// TIA Portal V20 export
// export: Created 2025-12-01T14:57:30.8490755Z, ExportSetting None, DisplayName Totally Integrated Automation Portal, DisplayVersion V20 Update 3, DisplayName TIA Portal Openness, DisplayVersion V20 Update 3, DisplayName TIA Portal Version Control Interface, DisplayVersion V20 Update 3, DisplayName STEP 7 Professional, DisplayVersion V20 Update 3, DisplayName STEP 7 Safety, DisplayVersion V20 Update 2, DisplayName WinCC Basic/Comfort/Advanced, DisplayVersion V20 Update 3, DisplayName WinCC Professional, DisplayVersion V20 Update 3, DisplayName WinCC Unified, DisplayVersion V20 Update 3
FUNCTION_BLOCK "FB271_FSS_Carga_Congelado"   // FB271, LAD
{ S7_Optimized_Access := 'FALSE' }
// NO sube los topes hasta
// stored: AutoNumber false, SetENOAutomatically false
   VAR_INPUT
      Mesa : UInt;   // Mesa de la FB
      Error_Tx : Bool;
      EnTension : Bool;   // Existe Tension en la Mesa
      Termico_Tx : Bool;
      pHsMx_1 : Bool;
      pHsMx_2 : Bool;
      EnMovimiento_Tx : Bool;
      Termico_TRx : Bool;
      Termico_TRxE : Bool;
      TRx_Arriba : Bool;
      TRx_Abajo { ExternalAccessible := 'False'; ExternalVisible := 'False'; ExternalWritable := 'False'} : Bool;
      EnMovimiento_TRx : Bool;
      EnMovimiento_TRxE : Bool;
      TP1_Arriba : Bool;
      TP1_Abajo { ExternalAccessible := 'False'; ExternalVisible := 'False'; ExternalWritable := 'False'} : Bool;
      TP2_Arriba : Bool;
      TP2_Abajo { ExternalAccessible := 'False'; ExternalVisible := 'False'; ExternalWritable := 'False'} : Bool;
      EnMovimiento_TP1 : Bool;
      EnMovimiento_TP2 : Bool;
      MAnt_E2_DesCarga_Act : Bool;
      AVTF_MAnt_E2_Mx : Bool;
      P_Mens_MAnt_E2_Mx : Bool;
      Arrival_S3 : Bool;
      Rotative_S3 : Bool;
      Complete_S3 : Bool;
      PTF_Mx_MSig_S4 : Bool;
      FTF_Mx_MSig_S4 : Bool;
      Mx_NoEntrar_E2 : Bool;
      Mx_Simul_E2S4 : Bool;
      F_EnvMens_PMx : Bool;
      F_EnvMens_AMx : Bool;
      OrdSal_S3 : Bool;
      OrdSal_S4 : Bool;
      MSig_Ocupada : Bool;
      IN_Bandeja_Peq_1 : Bool;
      IN_Bandeja_Peq_2 : Bool;
      IN_Bandeja_grande : Bool;
      V_SubirTP : Int := 20;
      V_CNT_pHsMx_E2 : Int := 500;
      V_CNT_pHsMx_FTF_E2 : Int := 0;
      V_CNTSeg_Pres : Int := 10;
      V_TIM_ApHsMx : Time := T#100ms;
      V_CNTSeg_Aus : Int := 10;
      V_TIM_VeloRapida_E2 : Time := T#1s;
      V_CNTSimul : Int := 999;
      V_Simul_Inicio : Int := 0;
      V_Simul_Fin : Int := 0;
      V_TOut_Entrada : Time := T#5s;
      V_TOut_TP : Time := T#2s;
      V_TOut_TR : Time := T#2s;
      V_TOut_Interlock : Time := T#10s;
      V_CNT_Perdida_pHs : Int := 10;
   END_VAR
   VAR_OUTPUT
      P_EnvMens_PMx : Bool;
      P_EnvMens_AMx : Bool;
      P_RecepOK_Mx : Bool;
      PTF_MAnt_E2_Mx : Bool;
      FTF_MAnt_E2_Mx : Bool;
      AVTF_Mx_MSig_S4 : Bool;
      P_Mens_Mx_MSig_S4 : Bool;
   END_VAR
   VAR
      TOut_Entrada_E2 { ExternalAccessible := 'False'; ExternalVisible := 'False'; ExternalWritable := 'False'; S7_SetPoint := 'True'} : TON_TIME;
      TOut_TP1 { ExternalAccessible := 'False'; ExternalVisible := 'False'; ExternalWritable := 'False'; S7_SetPoint := 'True'} : TON_TIME;
      TOut_TP2 { ExternalAccessible := 'False'; ExternalVisible := 'False'; ExternalWritable := 'False'; S7_SetPoint := 'True'} : TON_TIME;
      TOut_TRx { ExternalAccessible := 'False'; ExternalVisible := 'False'; ExternalWritable := 'False'; S7_SetPoint := 'True'} : TON_TIME;
      TOut_Interlock { S7_SetPoint := 'True'} : TON_TIME;
      CNTPerdida_pHs { ExternalAccessible := 'False'; ExternalVisible := 'False'; ExternalWritable := 'False'; S7_SetPoint := 'True'} : CTU_INT;
      TIM_VeloRapida_E2 { ExternalAccessible := 'False'; ExternalVisible := 'False'; ExternalWritable := 'False'; S7_SetPoint := 'True'} : TON_TIME;
      TIM_ApHsMx { S7_SetPoint := 'True'} : TON_TIME;
      CNT_pHsMx_E2 { ExternalAccessible := 'False'; ExternalVisible := 'False'; ExternalWritable := 'False'; S7_SetPoint := 'True'} : "FB910_CNT_UHS";
      CNTSeg_Pres { ExternalAccessible := 'False'; ExternalVisible := 'False'; ExternalWritable := 'False'; S7_SetPoint := 'True'} : CTU_INT;
      CNTSeg_Aus { ExternalAccessible := 'False'; ExternalVisible := 'False'; ExternalWritable := 'False'; S7_SetPoint := 'True'} : CTU_INT;
      CNTSimul { S7_SetPoint := 'True'} : CTD_INT;
      CNT_Inactividad { S7_SetPoint := 'True'} : "FB910_CNT_UHS";
      Tim_Marcha_Ina { S7_SetPoint := 'True'} : TON_TIME;
      CNTSimul_CV : Int;
      Simul_Mx_E2S4 : Bool;
      Protoc_Ini_Mx : Bool;
      FTF_Entrada_E2_OK : Bool;
      AVTF_Salida_S4_OK : Bool;
      MA_Avanzar_Tx : Bool;
      MA_Retroceder_Tx : Bool;
      MA_VeloRapida_Tx : Bool;
      MA_Subir_TP1 : Bool;
      MA_Bajar_TP1 : Bool;
      MA_Subir_TP2 : Bool;
      MA_Bajar_TP2 : Bool;
      MA_Avanzar_TRx : Bool;
      MA_Retroceder_TRx : Bool;
      MA_VeloRapida_TRx : Bool;
      MA_Subir_TRx : Bool;
      MA_Bajar_TRx : Bool;
      MA_PickUpOK_S3 : Bool;
      Selec_Entrada_E2 : Bool;
      Selec_Salida_S3 : Bool;
      Selec_Salida_S4 : Bool;
      Mx_ET00 : Bool;
      Mx_ET01 : Bool;
      Mx_ET02 : Bool;
      Mx_RES01 : Bool;
      Mx_RES02 : Bool;
      Mx_RES03 : Bool;
      Mx_RES09 : Bool;
      Mx_ET20 : Bool;
      Mx_ET21 : Bool;
      Mx_ET22 : Bool;
      Mx_ET23 : Bool;
      Mx_ET50 : Bool;
      Mx_ET51 : Bool;
      Mx_ET52 : Bool;
      Mx_ET60 : Bool;
      Mx_ET61 : Bool;
      Mx_ET90 : Bool;
      Mx_ET91 : Bool;
      Mx_ET120 : Bool;
      Mx_ET121 : Bool;
      Mx_ET150 : Bool;
      Mx_ET151 : Bool;
      Mx_ET160 : Bool;
      Mx_ET161 : Bool;
      Mx_ET250 : Bool;
      Mx_ET260 : Bool;
      STAT_EnvMens_PMx : Bool;
      STAT_EnvMens_AMx : Bool;
      STAT_FTF_MAnt_E2_Mx : Bool;
      STAT_AVTF_Mx_MSig_S4 : Bool;
   END_VAR
   VAR_TEMP
      EstadoZona : "EstadoZona";   // Estado de Zona de la Mesa
      EstadoVI : "EstadosMesa";   // Estado del Vehiculo Inteliguente de la Mesa
      ConfigFB : "UDT_ConfigFB";   // Configuracion de la FB de la Mesa
      BaseUnidades_ms : DInt;
      Aux_ET00 : Bool;
      FinCargaFSS_Auto_S3 : Bool;
      AutoArranque : Bool;
      EnResetPresMulti : Bool;
      EliminaErrores : Bool;
   END_VAR
BEGIN

REGION Network 1: INICIALIZAR - Recoger las Variables de Estado de la Mesa
   // Se recoge - Estado_CBx
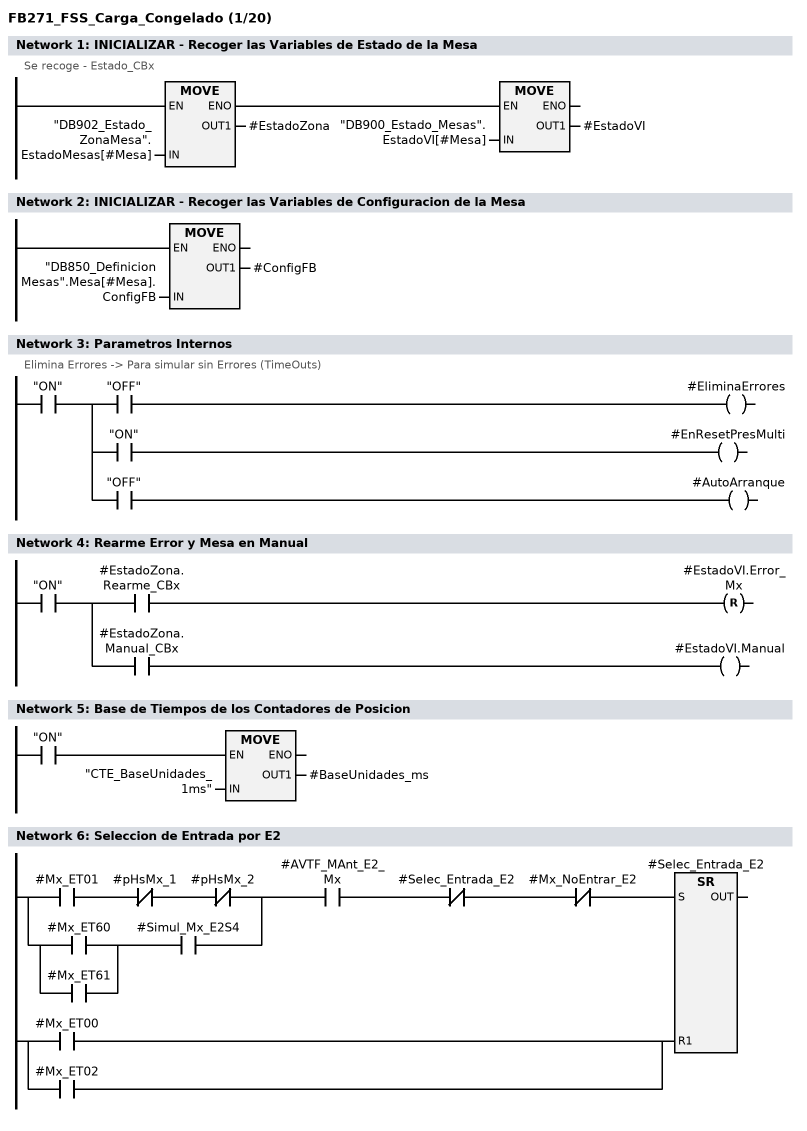
   RUNG wire#powerrail
      Move(in := "DB902_Estado_ZonaMesa".EstadoMesas[#Mesa], out1 => #EstadoZona)
      Move(in := "DB900_Estado_Mesas".EstadoVI[#Mesa], out1 => #EstadoVI)
   END_RUNG
   // the same network as SCL:
   #EstadoZona := "DB902_Estado_ZonaMesa".EstadoMesas[#Mesa];
   #EstadoVI := "DB900_Estado_Mesas".EstadoVI[#Mesa];
END_REGION

REGION Network 2: INICIALIZAR - Recoger las Variables de Configuracion de la Mesa
   RUNG wire#powerrail
      Move(in := "DB850_DefinicionMesas".Mesa[#Mesa].ConfigFB, out1 => #ConfigFB)
   END_RUNG
   // the same network as SCL:
   #ConfigFB := "DB850_DefinicionMesas".Mesa[#Mesa].ConfigFB;
END_REGION

REGION Network 3: Parametros Internos
   // Elimina Errores -> Para simular sin Errores (TimeOuts)
   RUNG wire#powerrail
      Contact( "ON" )
      wire#w1
      Contact( "OFF" )
      Coil( #EliminaErrores )
   END_RUNG
   RUNG wire#w1
      Contact( "ON" )
      Coil( #EnResetPresMulti )
   END_RUNG
   RUNG wire#w1
      Contact( "OFF" )
      Coil( #AutoArranque )
   END_RUNG
   // the same network as SCL:
   #EliminaErrores := "ON" AND "OFF";
   #EnResetPresMulti := "ON" AND "ON";
   #AutoArranque := "ON" AND "OFF";
END_REGION

REGION Network 4: Rearme Error y Mesa en Manual
   RUNG wire#powerrail
      Contact( "ON" )
      wire#w1
      Contact( #EstadoZona.Rearme_CBx )
      R_Coil( #EstadoVI.Error_Mx )
   END_RUNG
   RUNG wire#w1
      Contact( #EstadoZona.Manual_CBx )
      Coil( #EstadoVI.Manual )
   END_RUNG
   // the same network as SCL:
   IF "ON" AND #EstadoZona.Rearme_CBx THEN #EstadoVI.Error_Mx := FALSE; END_IF;
   #EstadoVI.Manual := "ON" AND #EstadoZona.Manual_CBx;
END_REGION

REGION Network 5: Base de Tiempos de los Contadores de Posicion
   RUNG wire#powerrail
      Contact( "ON" )
      Move(in := "CTE_BaseUnidades_1ms", out1 => #BaseUnidades_ms)
   END_RUNG
   // the same network as SCL:
   IF "ON" THEN #BaseUnidades_ms := "CTE_BaseUnidades_1ms"; END_IF;
END_REGION

REGION Network 6: Seleccion de Entrada por E2
   RUNG wire#powerrail
      Contact( #Mx_ET01 )
      I_Contact( #pHsMx_1 )
      I_Contact( #pHsMx_2 )
      wire#w1
      Contact( #AVTF_MAnt_E2_Mx )
      I_Contact( #Selec_Entrada_E2 )
      I_Contact( #Mx_NoEntrar_E2 )
      S_SR(operand := #Selec_Entrada_E2, r1 := wire#w3)
   END_RUNG
   RUNG wire#powerrail
      Contact( #Mx_ET60 )
      wire#w2
      Contact( #Simul_Mx_E2S4 )
   END_RUNG wire#w1
   RUNG wire#powerrail
      Contact( #Mx_ET61 )
   END_RUNG wire#w2
   RUNG wire#powerrail
      Contact( #Mx_ET00 )
   END_RUNG wire#w3
   RUNG wire#powerrail
      Contact( #Mx_ET02 )
   END_RUNG wire#w3
   // the same network as SCL:
   IF ((#Mx_ET01 AND NOT #pHsMx_1 AND NOT #pHsMx_2) OR ((#Mx_ET60 OR #Mx_ET61) AND #Simul_Mx_E2S4)) AND #AVTF_MAnt_E2_Mx AND NOT #Selec_Entrada_E2 AND NOT #Mx_NoEntrar_E2 THEN
       #Selec_Entrada_E2 := TRUE;   // SR flip-flop
   END_IF;
   IF #Mx_ET00 OR #Mx_ET02 THEN #Selec_Entrada_E2 := FALSE; END_IF;
END_REGION

REGION Network 7: Seleccion de Salida por S3 -Carga del FSS
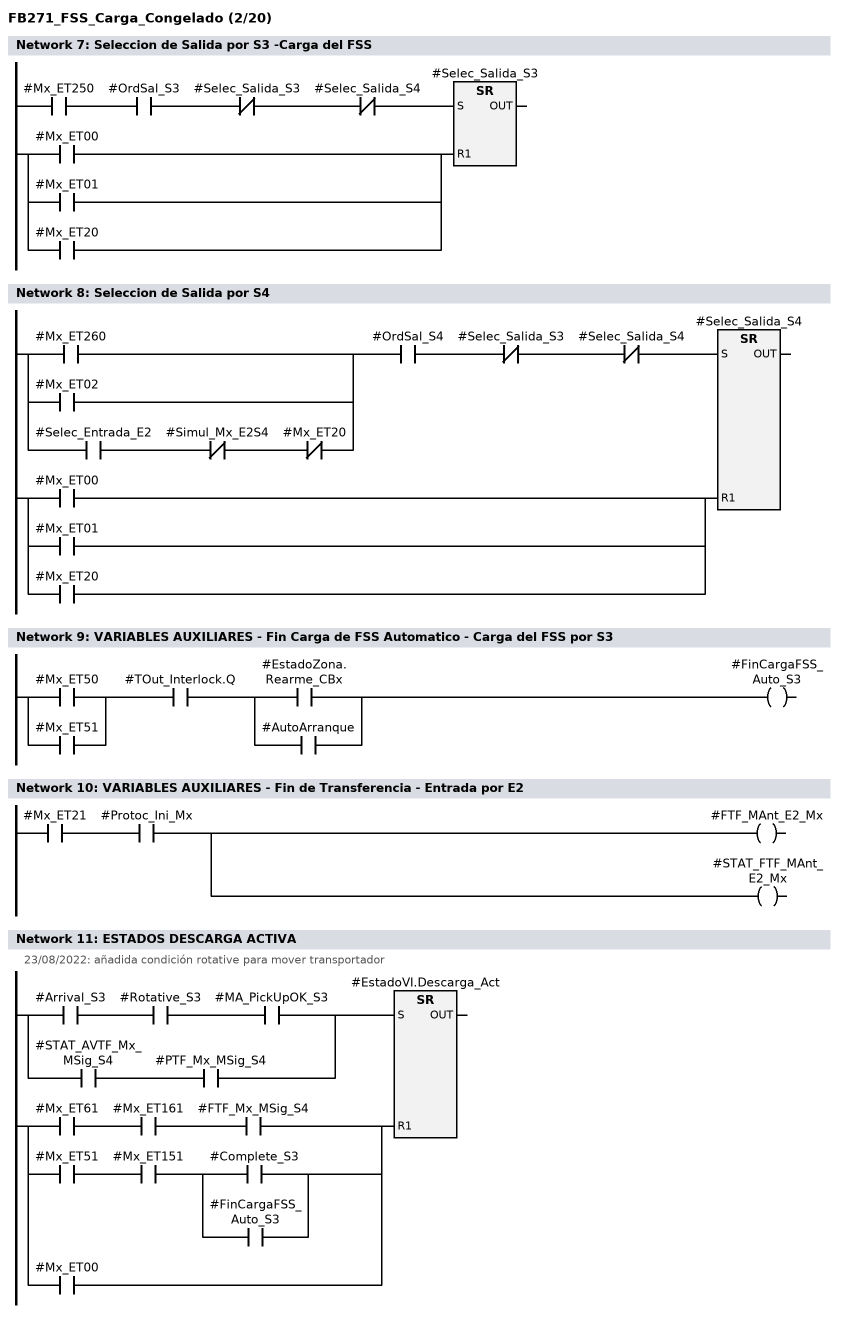
   RUNG wire#powerrail
      Contact( #Mx_ET250 )
      Contact( #OrdSal_S3 )
      I_Contact( #Selec_Salida_S3 )
      I_Contact( #Selec_Salida_S4 )
      S_SR(operand := #Selec_Salida_S3, r1 := wire#w1)
   END_RUNG
   RUNG wire#powerrail
      Contact( #Mx_ET00 )
   END_RUNG wire#w1
   RUNG wire#powerrail
      Contact( #Mx_ET01 )
   END_RUNG wire#w1
   RUNG wire#powerrail
      Contact( #Mx_ET20 )
   END_RUNG wire#w1
   // the same network as SCL:
   IF #Mx_ET250 AND #OrdSal_S3 AND NOT #Selec_Salida_S3 AND NOT #Selec_Salida_S4 THEN
       #Selec_Salida_S3 := TRUE;   // SR flip-flop
   END_IF;
   IF #Mx_ET00 OR #Mx_ET01 OR #Mx_ET20 THEN #Selec_Salida_S3 := FALSE; END_IF;
END_REGION

REGION Network 8: Seleccion de Salida por S4
   RUNG wire#powerrail
      Contact( #Mx_ET260 )
      wire#w1
      Contact( #OrdSal_S4 )
      I_Contact( #Selec_Salida_S3 )
      I_Contact( #Selec_Salida_S4 )
      S_SR(operand := #Selec_Salida_S4, r1 := wire#w2)
   END_RUNG
   RUNG wire#powerrail
      Contact( #Mx_ET02 )
   END_RUNG wire#w1
   RUNG wire#powerrail
      Contact( #Selec_Entrada_E2 )
      I_Contact( #Simul_Mx_E2S4 )
      I_Contact( #Mx_ET20 )
   END_RUNG wire#w1
   RUNG wire#powerrail
      Contact( #Mx_ET00 )
   END_RUNG wire#w2
   RUNG wire#powerrail
      Contact( #Mx_ET01 )
   END_RUNG wire#w2
   RUNG wire#powerrail
      Contact( #Mx_ET20 )
   END_RUNG wire#w2
   // the same network as SCL:
   IF (#Mx_ET260 OR #Mx_ET02 OR (#Selec_Entrada_E2 AND NOT #Simul_Mx_E2S4 AND NOT #Mx_ET20)) AND #OrdSal_S4 AND NOT #Selec_Salida_S3 AND NOT #Selec_Salida_S4 THEN
       #Selec_Salida_S4 := TRUE;   // SR flip-flop
   END_IF;
   IF #Mx_ET00 OR #Mx_ET01 OR #Mx_ET20 THEN #Selec_Salida_S4 := FALSE; END_IF;
END_REGION

REGION Network 9: VARIABLES AUXILIARES - Fin Carga de FSS Automatico - Carga del FSS por S3
   RUNG wire#powerrail
      Contact( #Mx_ET50 )
      wire#w1
      Contact( #TOut_Interlock.Q )
      wire#w2
      Contact( #EstadoZona.Rearme_CBx )
      wire#w3
      Coil( #FinCargaFSS_Auto_S3 )
   END_RUNG
   RUNG wire#powerrail
      Contact( #Mx_ET51 )
   END_RUNG wire#w1
   RUNG wire#w2
      Contact( #AutoArranque )
   END_RUNG wire#w3
   // the same network as SCL:
   #FinCargaFSS_Auto_S3 := (#Mx_ET50 OR #Mx_ET51) AND #TOut_Interlock.Q AND (#EstadoZona.Rearme_CBx OR #AutoArranque);
END_REGION

REGION Network 10: VARIABLES AUXILIARES - Fin de Transferencia - Entrada por E2
   RUNG wire#powerrail
      Contact( #Mx_ET21 )
      Contact( #Protoc_Ini_Mx )
      wire#w1
      Coil( #FTF_MAnt_E2_Mx )
   END_RUNG
   RUNG wire#w1
      Coil( #STAT_FTF_MAnt_E2_Mx )
   END_RUNG
   // the same network as SCL:
   #FTF_MAnt_E2_Mx := #Mx_ET21 AND #Protoc_Ini_Mx;
   #STAT_FTF_MAnt_E2_Mx := #FTF_MAnt_E2_Mx;
END_REGION

REGION Network 11: ESTADOS DESCARGA ACTIVA
   // 23/08/2022: añadida condición rotative para mover transportador
   RUNG wire#powerrail
      Contact( #Arrival_S3 )
      Contact( #Rotative_S3 )
      Contact( #MA_PickUpOK_S3 )
      wire#w1
      S_SR(operand := #EstadoVI.Descarga_Act, r1 := wire#w3)
   END_RUNG
   RUNG wire#powerrail
      Contact( #STAT_AVTF_Mx_MSig_S4 )
      Contact( #PTF_Mx_MSig_S4 )
   END_RUNG wire#w1
   RUNG wire#powerrail
      Contact( #Mx_ET61 )
      Contact( #Mx_ET161 )
      Contact( #FTF_Mx_MSig_S4 )
   END_RUNG wire#w3
   RUNG wire#powerrail
      Contact( #Mx_ET51 )
      Contact( #Mx_ET151 )
      wire#w2
      Contact( #Complete_S3 )
   END_RUNG wire#w3
   RUNG wire#w2
      Contact( #FinCargaFSS_Auto_S3 )
   END_RUNG wire#w3
   RUNG wire#powerrail
      Contact( #Mx_ET00 )
   END_RUNG wire#w3
   // the same network as SCL:
   IF (#Arrival_S3 AND #Rotative_S3 AND #MA_PickUpOK_S3) OR (#STAT_AVTF_Mx_MSig_S4 AND #PTF_Mx_MSig_S4) THEN
       #EstadoVI.Descarga_Act := TRUE;   // SR flip-flop
   END_IF;
   IF (#Mx_ET61 AND #Mx_ET161 AND #FTF_Mx_MSig_S4) OR (#Mx_ET51 AND #Mx_ET151 AND (#Complete_S3 OR #FinCargaFSS_Auto_S3)) OR #Mx_ET00 THEN
       #EstadoVI.Descarga_Act := FALSE;
   END_IF;
END_REGION

REGION Network 12: ET91
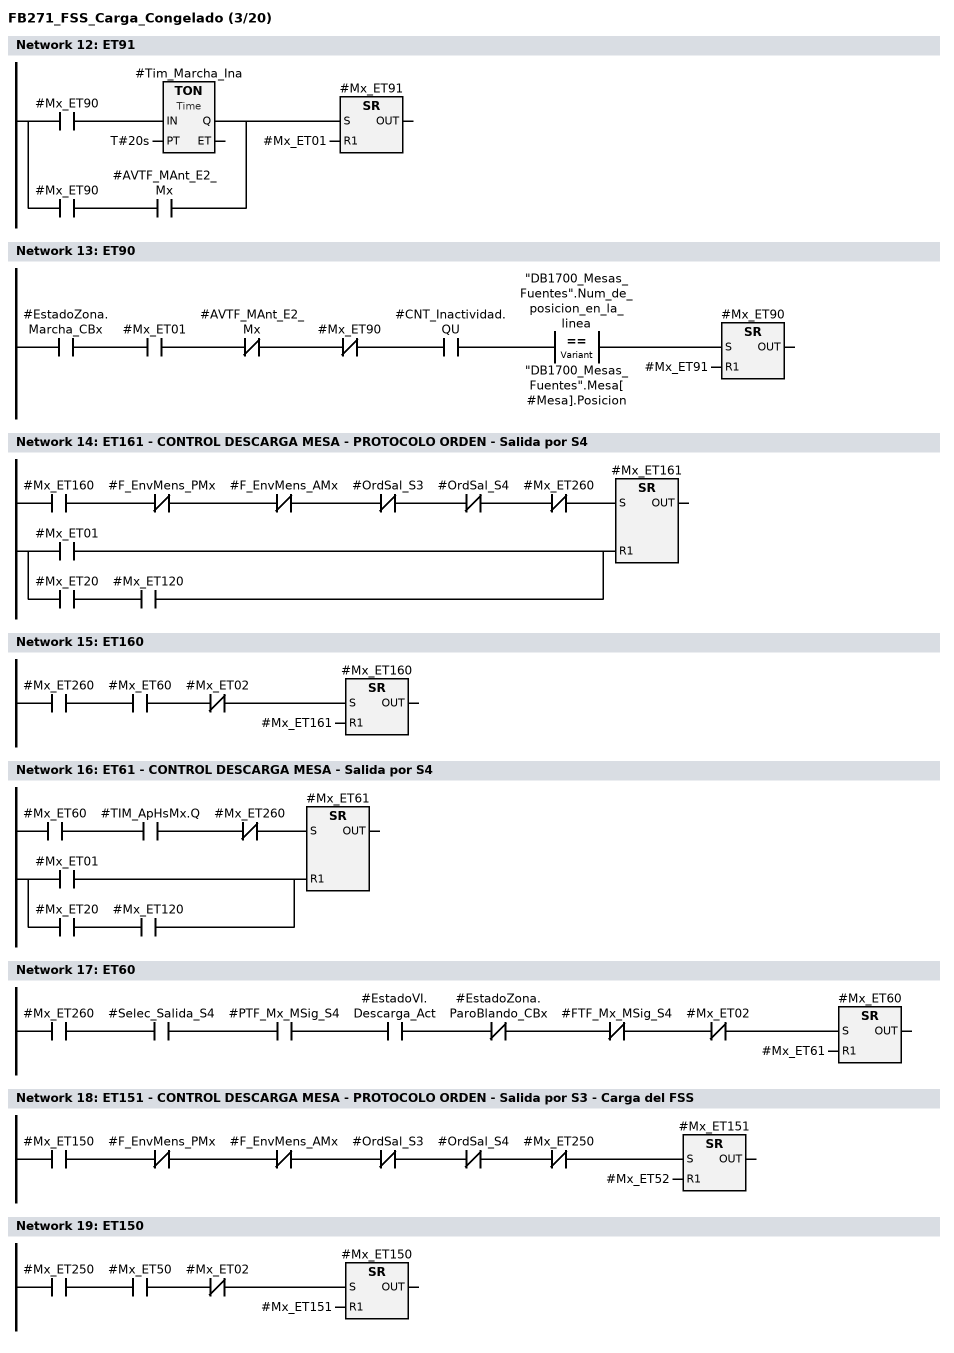
   RUNG wire#powerrail
      Contact( #Mx_ET90 )
      { S7_Templates := "time_type := Time" } #Tim_Marcha_Ina.TON(pt := T#20s, et =>)
      wire#w1
      S_SR(operand := #Mx_ET91, r1 := #Mx_ET01)
   END_RUNG
   RUNG wire#powerrail
      Contact( #Mx_ET90 )
      Contact( #AVTF_MAnt_E2_Mx )
   END_RUNG wire#w1
   // the same network as SCL:
   #Tim_Marcha_Ina(IN := #Mx_ET90, PT := T#20s);   // TON
   IF #Tim_Marcha_Ina.Q OR (#Mx_ET90 AND #AVTF_MAnt_E2_Mx) THEN
       #Mx_ET91 := TRUE;   // SR flip-flop
   END_IF;
   IF #Mx_ET01 THEN #Mx_ET91 := FALSE; END_IF;
END_REGION

REGION Network 13: ET90
   RUNG wire#powerrail
      Contact( #EstadoZona.Marcha_CBx )
      Contact( #Mx_ET01 )
      I_Contact( #AVTF_MAnt_E2_Mx )
      I_Contact( #Mx_ET90 )
      Contact( #CNT_Inactividad.QU )
      { S7_Templates := "SrcType := Variant" } EQ_Contact(in1 := "DB1700_Mesas_Fuentes".Num_de_posicion_en_la_linea, in2 := "DB1700_Mesas_Fuentes".Mesa[#Mesa].Posicion)
      S_SR(operand := #Mx_ET90, r1 := #Mx_ET91)
   END_RUNG
   // the same network as SCL:
   IF #EstadoZona.Marcha_CBx AND #Mx_ET01 AND NOT #AVTF_MAnt_E2_Mx AND NOT #Mx_ET90 AND #CNT_Inactividad.QU AND ("DB1700_Mesas_Fuentes".Num_de_posicion_en_la_linea = "DB1700_Mesas_Fuentes".Mesa[#Mesa].Posicion) THEN
       #Mx_ET90 := TRUE;   // SR flip-flop
   END_IF;
   IF #Mx_ET91 THEN #Mx_ET90 := FALSE; END_IF;
END_REGION

REGION Network 14: ET161 - CONTROL DESCARGA MESA - PROTOCOLO ORDEN - Salida por S4
   RUNG wire#powerrail
      Contact( #Mx_ET160 )
      I_Contact( #F_EnvMens_PMx )
      I_Contact( #F_EnvMens_AMx )
      I_Contact( #OrdSal_S3 )
      I_Contact( #OrdSal_S4 )
      I_Contact( #Mx_ET260 )
      S_SR(operand := #Mx_ET161, r1 := wire#w1)
   END_RUNG
   RUNG wire#powerrail
      Contact( #Mx_ET01 )
   END_RUNG wire#w1
   RUNG wire#powerrail
      Contact( #Mx_ET20 )
      Contact( #Mx_ET120 )
   END_RUNG wire#w1
   // the same network as SCL:
   IF #Mx_ET160 AND NOT #F_EnvMens_PMx AND NOT #F_EnvMens_AMx AND NOT #OrdSal_S3 AND NOT #OrdSal_S4 AND NOT #Mx_ET260 THEN
       #Mx_ET161 := TRUE;   // SR flip-flop
   END_IF;
   IF #Mx_ET01 OR (#Mx_ET20 AND #Mx_ET120) THEN #Mx_ET161 := FALSE; END_IF;
END_REGION

REGION Network 15: ET160
   RUNG wire#powerrail
      Contact( #Mx_ET260 )
      Contact( #Mx_ET60 )
      I_Contact( #Mx_ET02 )
      S_SR(operand := #Mx_ET160, r1 := #Mx_ET161)
   END_RUNG
   // the same network as SCL:
   IF #Mx_ET260 AND #Mx_ET60 AND NOT #Mx_ET02 THEN
       #Mx_ET160 := TRUE;   // SR flip-flop
   END_IF;
   IF #Mx_ET161 THEN #Mx_ET160 := FALSE; END_IF;
END_REGION

REGION Network 16: ET61 - CONTROL DESCARGA MESA - Salida por S4
   RUNG wire#powerrail
      Contact( #Mx_ET60 )
      Contact( #TIM_ApHsMx.Q )
      I_Contact( #Mx_ET260 )
      S_SR(operand := #Mx_ET61, r1 := wire#w1)
   END_RUNG
   RUNG wire#powerrail
      Contact( #Mx_ET01 )
   END_RUNG wire#w1
   RUNG wire#powerrail
      Contact( #Mx_ET20 )
      Contact( #Mx_ET120 )
   END_RUNG wire#w1
   // the same network as SCL:
   IF #Mx_ET60 AND #TIM_ApHsMx.Q AND NOT #Mx_ET260 THEN
       #Mx_ET61 := TRUE;   // SR flip-flop
   END_IF;
   IF #Mx_ET01 OR (#Mx_ET20 AND #Mx_ET120) THEN #Mx_ET61 := FALSE; END_IF;
END_REGION

REGION Network 17: ET60
   RUNG wire#powerrail
      Contact( #Mx_ET260 )
      Contact( #Selec_Salida_S4 )
      Contact( #PTF_Mx_MSig_S4 )
      Contact( #EstadoVI.Descarga_Act )
      I_Contact( #EstadoZona.ParoBlando_CBx )
      I_Contact( #FTF_Mx_MSig_S4 )
      I_Contact( #Mx_ET02 )
      S_SR(operand := #Mx_ET60, r1 := #Mx_ET61)
   END_RUNG
   // the same network as SCL:
   IF #Mx_ET260 AND #Selec_Salida_S4 AND #PTF_Mx_MSig_S4 AND #EstadoVI.Descarga_Act AND NOT #EstadoZona.ParoBlando_CBx AND NOT #FTF_Mx_MSig_S4 AND NOT #Mx_ET02 THEN
       #Mx_ET60 := TRUE;   // SR flip-flop
   END_IF;
   IF #Mx_ET61 THEN #Mx_ET60 := FALSE; END_IF;
END_REGION

REGION Network 18: ET151 - CONTROL DESCARGA MESA - PROTOCOLO ORDEN - Salida por S3 - Carga del FSS
   RUNG wire#powerrail
      Contact( #Mx_ET150 )
      I_Contact( #F_EnvMens_PMx )
      I_Contact( #F_EnvMens_AMx )
      I_Contact( #OrdSal_S3 )
      I_Contact( #OrdSal_S4 )
      I_Contact( #Mx_ET250 )
      S_SR(operand := #Mx_ET151, r1 := #Mx_ET52)
   END_RUNG
   // the same network as SCL:
   IF #Mx_ET150 AND NOT #F_EnvMens_PMx AND NOT #F_EnvMens_AMx AND NOT #OrdSal_S3 AND NOT #OrdSal_S4 AND NOT #Mx_ET250 THEN
       #Mx_ET151 := TRUE;   // SR flip-flop
   END_IF;
   IF #Mx_ET52 THEN #Mx_ET151 := FALSE; END_IF;
END_REGION

REGION Network 19: ET150
   RUNG wire#powerrail
      Contact( #Mx_ET250 )
      Contact( #Mx_ET50 )
      I_Contact( #Mx_ET02 )
      S_SR(operand := #Mx_ET150, r1 := #Mx_ET151)
   END_RUNG
   // the same network as SCL:
   IF #Mx_ET250 AND #Mx_ET50 AND NOT #Mx_ET02 THEN
       #Mx_ET150 := TRUE;   // SR flip-flop
   END_IF;
   IF #Mx_ET151 THEN #Mx_ET150 := FALSE; END_IF;
END_REGION

REGION Network 20: ET52 - CONTROL DESCARGA MESA - Salida por S3 - Carga del FSS
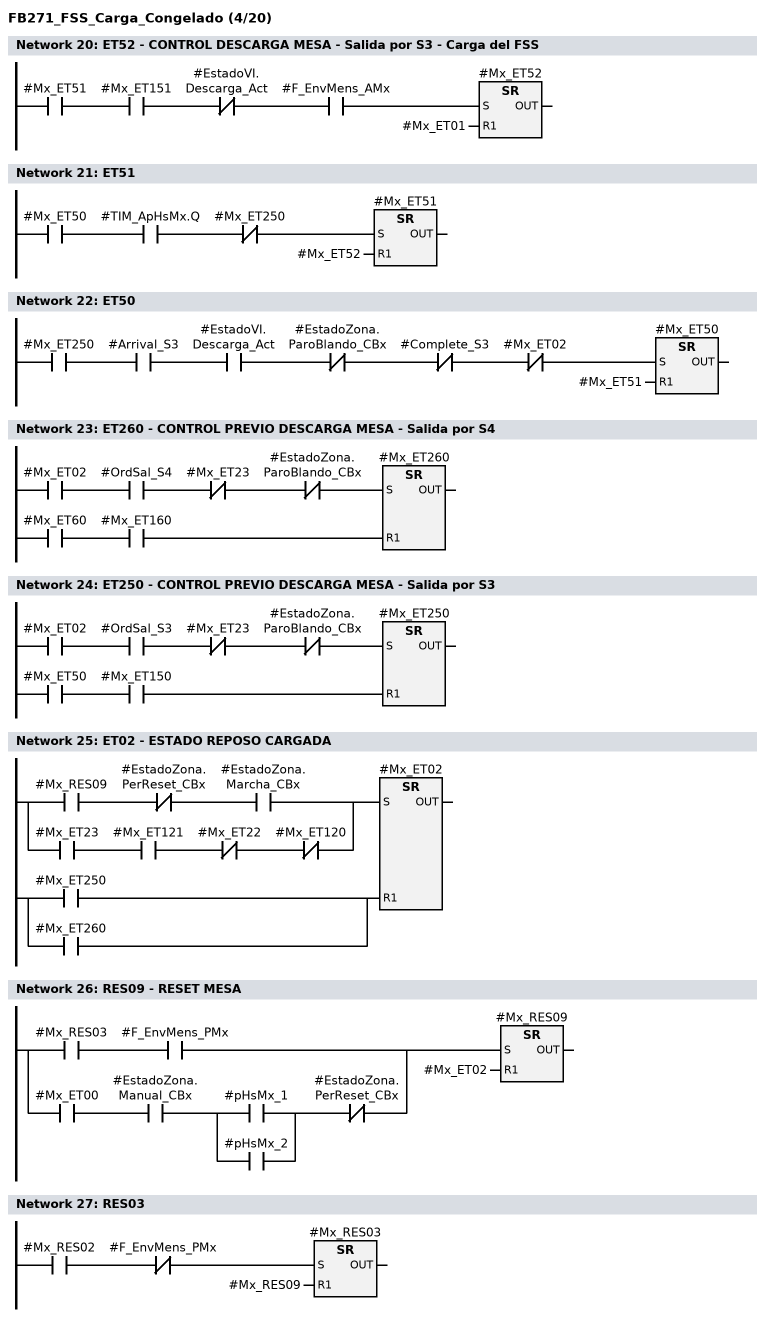
   RUNG wire#powerrail
      Contact( #Mx_ET51 )
      Contact( #Mx_ET151 )
      I_Contact( #EstadoVI.Descarga_Act )
      Contact( #F_EnvMens_AMx )
      S_SR(operand := #Mx_ET52, r1 := #Mx_ET01)
   END_RUNG
   // the same network as SCL:
   IF #Mx_ET51 AND #Mx_ET151 AND NOT #EstadoVI.Descarga_Act AND #F_EnvMens_AMx THEN
       #Mx_ET52 := TRUE;   // SR flip-flop
   END_IF;
   IF #Mx_ET01 THEN #Mx_ET52 := FALSE; END_IF;
END_REGION

REGION Network 21: ET51
   RUNG wire#powerrail
      Contact( #Mx_ET50 )
      Contact( #TIM_ApHsMx.Q )
      I_Contact( #Mx_ET250 )
      S_SR(operand := #Mx_ET51, r1 := #Mx_ET52)
   END_RUNG
   // the same network as SCL:
   IF #Mx_ET50 AND #TIM_ApHsMx.Q AND NOT #Mx_ET250 THEN
       #Mx_ET51 := TRUE;   // SR flip-flop
   END_IF;
   IF #Mx_ET52 THEN #Mx_ET51 := FALSE; END_IF;
END_REGION

REGION Network 22: ET50
   RUNG wire#powerrail
      Contact( #Mx_ET250 )
      Contact( #Arrival_S3 )
      Contact( #EstadoVI.Descarga_Act )
      I_Contact( #EstadoZona.ParoBlando_CBx )
      I_Contact( #Complete_S3 )
      I_Contact( #Mx_ET02 )
      S_SR(operand := #Mx_ET50, r1 := #Mx_ET51)
   END_RUNG
   // the same network as SCL:
   IF #Mx_ET250 AND #Arrival_S3 AND #EstadoVI.Descarga_Act AND NOT #EstadoZona.ParoBlando_CBx AND NOT #Complete_S3 AND NOT #Mx_ET02 THEN
       #Mx_ET50 := TRUE;   // SR flip-flop
   END_IF;
   IF #Mx_ET51 THEN #Mx_ET50 := FALSE; END_IF;
END_REGION

REGION Network 23: ET260 - CONTROL PREVIO DESCARGA MESA - Salida por S4
   RUNG wire#powerrail
      Contact( #Mx_ET02 )
      Contact( #OrdSal_S4 )
      I_Contact( #Mx_ET23 )
      I_Contact( #EstadoZona.ParoBlando_CBx )
      S_SR(operand := #Mx_ET260, r1 := wire#w1)
   END_RUNG
   RUNG wire#powerrail
      Contact( #Mx_ET60 )
      Contact( #Mx_ET160 )
   END_RUNG wire#w1
   // the same network as SCL:
   IF #Mx_ET02 AND #OrdSal_S4 AND NOT #Mx_ET23 AND NOT #EstadoZona.ParoBlando_CBx THEN
       #Mx_ET260 := TRUE;   // SR flip-flop
   END_IF;
   IF #Mx_ET60 AND #Mx_ET160 THEN #Mx_ET260 := FALSE; END_IF;
END_REGION

REGION Network 24: ET250 - CONTROL PREVIO DESCARGA MESA - Salida por S3
   RUNG wire#powerrail
      Contact( #Mx_ET02 )
      Contact( #OrdSal_S3 )
      I_Contact( #Mx_ET23 )
      I_Contact( #EstadoZona.ParoBlando_CBx )
      S_SR(operand := #Mx_ET250, r1 := wire#w1)
   END_RUNG
   RUNG wire#powerrail
      Contact( #Mx_ET50 )
      Contact( #Mx_ET150 )
   END_RUNG wire#w1
   // the same network as SCL:
   IF #Mx_ET02 AND #OrdSal_S3 AND NOT #Mx_ET23 AND NOT #EstadoZona.ParoBlando_CBx THEN
       #Mx_ET250 := TRUE;   // SR flip-flop
   END_IF;
   IF #Mx_ET50 AND #Mx_ET150 THEN #Mx_ET250 := FALSE; END_IF;
END_REGION

REGION Network 25: ET02 - ESTADO REPOSO CARGADA
   RUNG wire#powerrail
      Contact( #Mx_RES09 )
      I_Contact( #EstadoZona.PerReset_CBx )
      Contact( #EstadoZona.Marcha_CBx )
      wire#w1
      S_SR(operand := #Mx_ET02, r1 := wire#w2)
   END_RUNG
   RUNG wire#powerrail
      Contact( #Mx_ET23 )
      Contact( #Mx_ET121 )
      I_Contact( #Mx_ET22 )
      I_Contact( #Mx_ET120 )
   END_RUNG wire#w1
   RUNG wire#powerrail
      Contact( #Mx_ET250 )
   END_RUNG wire#w2
   RUNG wire#powerrail
      Contact( #Mx_ET260 )
   END_RUNG wire#w2
   // the same network as SCL:
   IF (#Mx_RES09 AND NOT #EstadoZona.PerReset_CBx AND #EstadoZona.Marcha_CBx) OR (#Mx_ET23 AND #Mx_ET121 AND NOT #Mx_ET22 AND NOT #Mx_ET120) THEN
       #Mx_ET02 := TRUE;   // SR flip-flop
   END_IF;
   IF #Mx_ET250 OR #Mx_ET260 THEN #Mx_ET02 := FALSE; END_IF;
END_REGION

REGION Network 26: RES09 - RESET MESA
   RUNG wire#powerrail
      Contact( #Mx_RES03 )
      Contact( #F_EnvMens_PMx )
      wire#w1
      S_SR(operand := #Mx_RES09, r1 := #Mx_ET02)
   END_RUNG
   RUNG wire#powerrail
      Contact( #Mx_ET00 )
      Contact( #EstadoZona.Manual_CBx )
      wire#w2
      Contact( #pHsMx_1 )
      wire#w3
      I_Contact( #EstadoZona.PerReset_CBx )
   END_RUNG wire#w1
   RUNG wire#w2
      Contact( #pHsMx_2 )
   END_RUNG wire#w3
   // the same network as SCL:
   IF (#Mx_RES03 AND #F_EnvMens_PMx) OR (#Mx_ET00 AND #EstadoZona.Manual_CBx AND (#pHsMx_1 OR #pHsMx_2) AND NOT #EstadoZona.PerReset_CBx) THEN
       #Mx_RES09 := TRUE;   // SR flip-flop
   END_IF;
   IF #Mx_ET02 THEN #Mx_RES09 := FALSE; END_IF;
END_REGION

REGION Network 27: RES03
   RUNG wire#powerrail
      Contact( #Mx_RES02 )
      I_Contact( #F_EnvMens_PMx )
      S_SR(operand := #Mx_RES03, r1 := #Mx_RES09)
   END_RUNG
   // the same network as SCL:
   IF #Mx_RES02 AND NOT #F_EnvMens_PMx THEN
       #Mx_RES03 := TRUE;   // SR flip-flop
   END_IF;
   IF #Mx_RES09 THEN #Mx_RES03 := FALSE; END_IF;
END_REGION

REGION Network 28: RES02
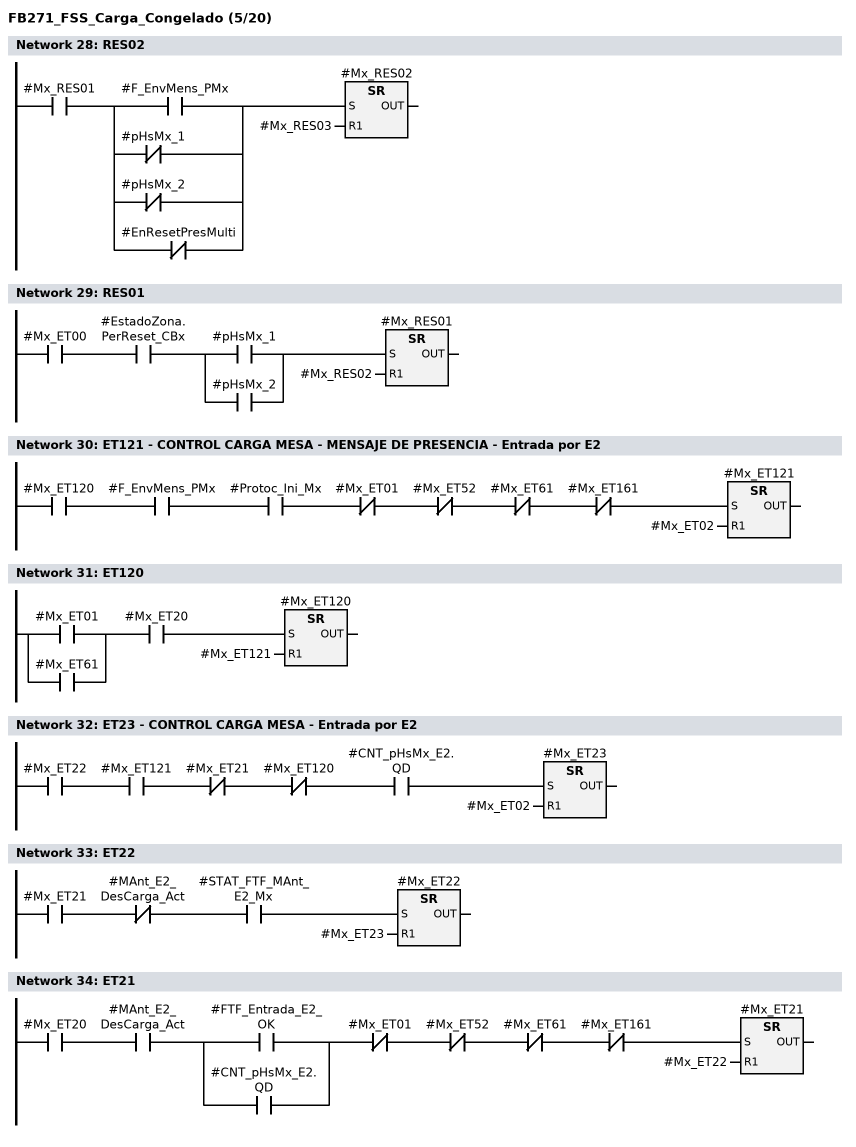
   RUNG wire#powerrail
      Contact( #Mx_RES01 )
      wire#w1
      Contact( #F_EnvMens_PMx )
      wire#w2
      S_SR(operand := #Mx_RES02, r1 := #Mx_RES03)
   END_RUNG
   RUNG wire#w1
      I_Contact( #pHsMx_1 )
   END_RUNG wire#w2
   RUNG wire#w1
      I_Contact( #pHsMx_2 )
   END_RUNG wire#w2
   RUNG wire#w1
      I_Contact( #EnResetPresMulti )
   END_RUNG wire#w2
   // the same network as SCL:
   IF #Mx_RES01 AND (#F_EnvMens_PMx OR NOT #pHsMx_1 OR NOT #pHsMx_2 OR NOT #EnResetPresMulti) THEN
       #Mx_RES02 := TRUE;   // SR flip-flop
   END_IF;
   IF #Mx_RES03 THEN #Mx_RES02 := FALSE; END_IF;
END_REGION

REGION Network 29: RES01
   RUNG wire#powerrail
      Contact( #Mx_ET00 )
      Contact( #EstadoZona.PerReset_CBx )
      wire#w1
      Contact( #pHsMx_1 )
      wire#w2
      S_SR(operand := #Mx_RES01, r1 := #Mx_RES02)
   END_RUNG
   RUNG wire#w1
      Contact( #pHsMx_2 )
   END_RUNG wire#w2
   // the same network as SCL:
   IF #Mx_ET00 AND #EstadoZona.PerReset_CBx AND (#pHsMx_1 OR #pHsMx_2) THEN
       #Mx_RES01 := TRUE;   // SR flip-flop
   END_IF;
   IF #Mx_RES02 THEN #Mx_RES01 := FALSE; END_IF;
END_REGION

REGION Network 30: ET121 - CONTROL CARGA MESA - MENSAJE DE PRESENCIA - Entrada por E2
   RUNG wire#powerrail
      Contact( #Mx_ET120 )
      Contact( #F_EnvMens_PMx )
      Contact( #Protoc_Ini_Mx )
      I_Contact( #Mx_ET01 )
      I_Contact( #Mx_ET52 )
      I_Contact( #Mx_ET61 )
      I_Contact( #Mx_ET161 )
      S_SR(operand := #Mx_ET121, r1 := #Mx_ET02)
   END_RUNG
   // the same network as SCL:
   IF #Mx_ET120 AND #F_EnvMens_PMx AND #Protoc_Ini_Mx AND NOT #Mx_ET01 AND NOT #Mx_ET52 AND NOT #Mx_ET61 AND NOT #Mx_ET161 THEN
       #Mx_ET121 := TRUE;   // SR flip-flop
   END_IF;
   IF #Mx_ET02 THEN #Mx_ET121 := FALSE; END_IF;
END_REGION

REGION Network 31: ET120
   RUNG wire#powerrail
      Contact( #Mx_ET01 )
      wire#w1
      Contact( #Mx_ET20 )
      S_SR(operand := #Mx_ET120, r1 := #Mx_ET121)
   END_RUNG
   RUNG wire#powerrail
      Contact( #Mx_ET61 )
   END_RUNG wire#w1
   // the same network as SCL:
   IF (#Mx_ET01 OR #Mx_ET61) AND #Mx_ET20 THEN
       #Mx_ET120 := TRUE;   // SR flip-flop
   END_IF;
   IF #Mx_ET121 THEN #Mx_ET120 := FALSE; END_IF;
END_REGION

REGION Network 32: ET23 - CONTROL CARGA MESA - Entrada por E2
   RUNG wire#powerrail
      Contact( #Mx_ET22 )
      Contact( #Mx_ET121 )
      I_Contact( #Mx_ET21 )
      I_Contact( #Mx_ET120 )
      Contact( #CNT_pHsMx_E2.QD )
      S_SR(operand := #Mx_ET23, r1 := #Mx_ET02)
   END_RUNG
   // the same network as SCL:
   IF #Mx_ET22 AND #Mx_ET121 AND NOT #Mx_ET21 AND NOT #Mx_ET120 AND #CNT_pHsMx_E2.QD THEN
       #Mx_ET23 := TRUE;   // SR flip-flop
   END_IF;
   IF #Mx_ET02 THEN #Mx_ET23 := FALSE; END_IF;
END_REGION

REGION Network 33: ET22
   RUNG wire#powerrail
      Contact( #Mx_ET21 )
      I_Contact( #MAnt_E2_DesCarga_Act )
      Contact( #STAT_FTF_MAnt_E2_Mx )
      S_SR(operand := #Mx_ET22, r1 := #Mx_ET23)
   END_RUNG
   // the same network as SCL:
   IF #Mx_ET21 AND NOT #MAnt_E2_DesCarga_Act AND #STAT_FTF_MAnt_E2_Mx THEN
       #Mx_ET22 := TRUE;   // SR flip-flop
   END_IF;
   IF #Mx_ET23 THEN #Mx_ET22 := FALSE; END_IF;
END_REGION

REGION Network 34: ET21
   RUNG wire#powerrail
      Contact( #Mx_ET20 )
      Contact( #MAnt_E2_DesCarga_Act )
      wire#w1
      Contact( #FTF_Entrada_E2_OK )
      wire#w2
      I_Contact( #Mx_ET01 )
      I_Contact( #Mx_ET52 )
      I_Contact( #Mx_ET61 )
      I_Contact( #Mx_ET161 )
      S_SR(operand := #Mx_ET21, r1 := #Mx_ET22)
   END_RUNG
   RUNG wire#w1
      Contact( #CNT_pHsMx_E2.QD )
   END_RUNG wire#w2
   // the same network as SCL:
   IF #Mx_ET20 AND #MAnt_E2_DesCarga_Act AND (#FTF_Entrada_E2_OK OR #CNT_pHsMx_E2.QD) AND NOT #Mx_ET01 AND NOT #Mx_ET52 AND NOT #Mx_ET61 AND NOT #Mx_ET161 THEN
       #Mx_ET21 := TRUE;   // SR flip-flop
   END_IF;
   IF #Mx_ET22 THEN #Mx_ET21 := FALSE; END_IF;
END_REGION

REGION Network 35: ET20
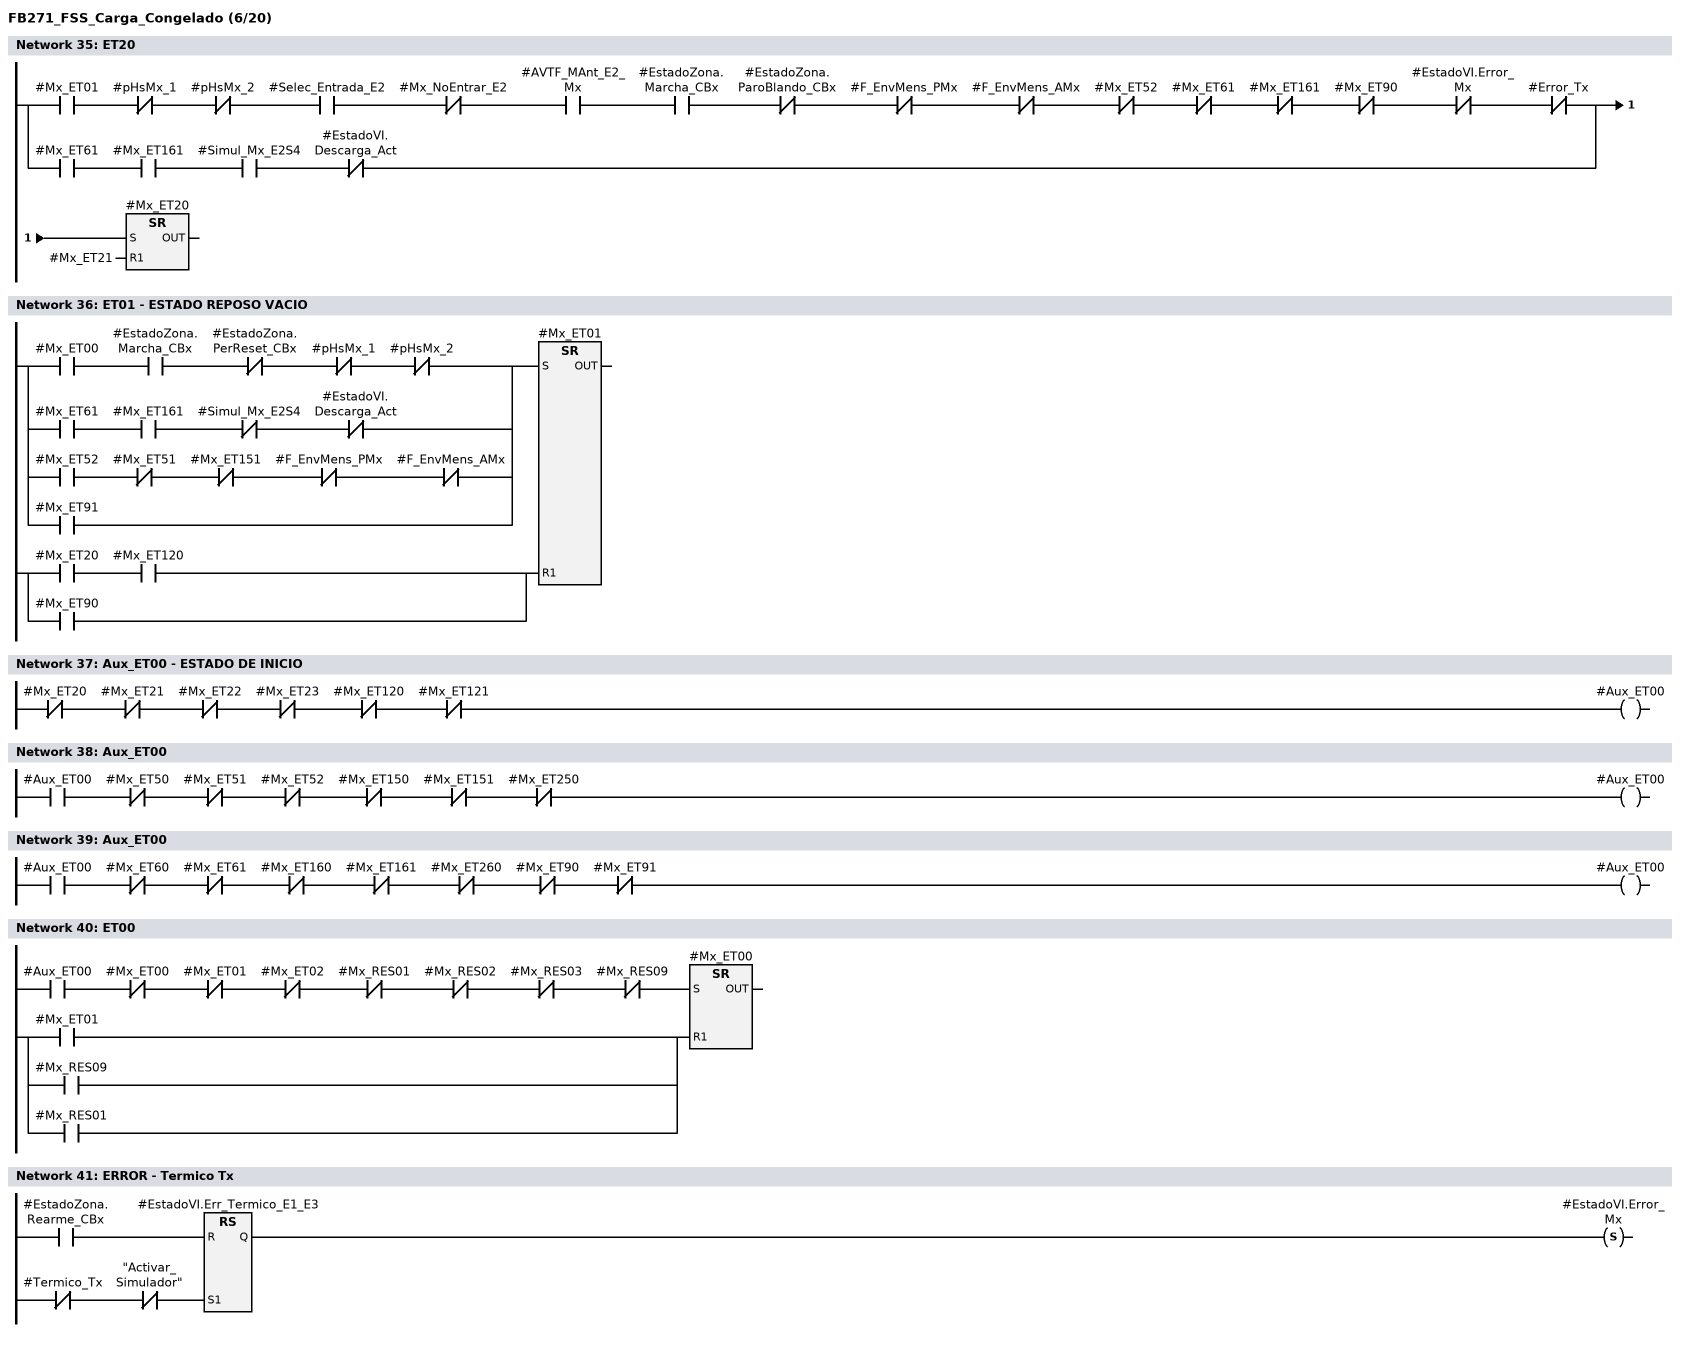
   RUNG wire#powerrail
      Contact( #Mx_ET01 )
      I_Contact( #pHsMx_1 )
      I_Contact( #pHsMx_2 )
      Contact( #Selec_Entrada_E2 )
      I_Contact( #Mx_NoEntrar_E2 )
      Contact( #AVTF_MAnt_E2_Mx )
      Contact( #EstadoZona.Marcha_CBx )
      I_Contact( #EstadoZona.ParoBlando_CBx )
      I_Contact( #F_EnvMens_PMx )
      I_Contact( #F_EnvMens_AMx )
      I_Contact( #Mx_ET52 )
      I_Contact( #Mx_ET61 )
      I_Contact( #Mx_ET161 )
      I_Contact( #Mx_ET90 )
      I_Contact( #EstadoVI.Error_Mx )
      I_Contact( #Error_Tx )
      wire#w1
      S_SR(operand := #Mx_ET20, r1 := #Mx_ET21)
   END_RUNG
   RUNG wire#powerrail
      Contact( #Mx_ET61 )
      Contact( #Mx_ET161 )
      Contact( #Simul_Mx_E2S4 )
      I_Contact( #EstadoVI.Descarga_Act )
   END_RUNG wire#w1
   // the same network as SCL:
   IF (#Mx_ET01 AND NOT #pHsMx_1 AND NOT #pHsMx_2 AND #Selec_Entrada_E2 AND NOT #Mx_NoEntrar_E2 AND #AVTF_MAnt_E2_Mx AND #EstadoZona.Marcha_CBx AND NOT #EstadoZona.ParoBlando_CBx AND NOT #F_EnvMens_PMx AND NOT #F_EnvMens_AMx AND NOT #Mx_ET52 AND NOT #Mx_ET61 AND NOT #Mx_ET161 AND NOT #Mx_ET90 AND NOT #EstadoVI.Error_Mx AND NOT #Error_Tx) OR (#Mx_ET61 AND #Mx_ET161 AND #Simul_Mx_E2S4 AND NOT #EstadoVI.Descarga_Act) THEN
       #Mx_ET20 := TRUE;   // SR flip-flop
   END_IF;
   IF #Mx_ET21 THEN #Mx_ET20 := FALSE; END_IF;
END_REGION

REGION Network 36: ET01 - ESTADO REPOSO VACIO
   RUNG wire#powerrail
      Contact( #Mx_ET00 )
      Contact( #EstadoZona.Marcha_CBx )
      I_Contact( #EstadoZona.PerReset_CBx )
      I_Contact( #pHsMx_1 )
      I_Contact( #pHsMx_2 )
      wire#w1
      S_SR(operand := #Mx_ET01, r1 := wire#w2)
   END_RUNG
   RUNG wire#powerrail
      Contact( #Mx_ET61 )
      Contact( #Mx_ET161 )
      I_Contact( #Simul_Mx_E2S4 )
      I_Contact( #EstadoVI.Descarga_Act )
   END_RUNG wire#w1
   RUNG wire#powerrail
      Contact( #Mx_ET52 )
      I_Contact( #Mx_ET51 )
      I_Contact( #Mx_ET151 )
      I_Contact( #F_EnvMens_PMx )
      I_Contact( #F_EnvMens_AMx )
   END_RUNG wire#w1
   RUNG wire#powerrail
      Contact( #Mx_ET91 )
   END_RUNG wire#w1
   RUNG wire#powerrail
      Contact( #Mx_ET20 )
      Contact( #Mx_ET120 )
   END_RUNG wire#w2
   RUNG wire#powerrail
      Contact( #Mx_ET90 )
   END_RUNG wire#w2
   // the same network as SCL:
   IF (#Mx_ET00 AND #EstadoZona.Marcha_CBx AND NOT #EstadoZona.PerReset_CBx AND NOT #pHsMx_1 AND NOT #pHsMx_2) OR (#Mx_ET61 AND #Mx_ET161 AND NOT #Simul_Mx_E2S4 AND NOT #EstadoVI.Descarga_Act) OR (#Mx_ET52 AND NOT #Mx_ET51 AND NOT #Mx_ET151 AND NOT #F_EnvMens_PMx AND NOT #F_EnvMens_AMx) OR #Mx_ET91 THEN
       #Mx_ET01 := TRUE;   // SR flip-flop
   END_IF;
   IF (#Mx_ET20 AND #Mx_ET120) OR #Mx_ET90 THEN #Mx_ET01 := FALSE; END_IF;
END_REGION

REGION Network 37: Aux_ET00 - ESTADO DE INICIO
   RUNG wire#powerrail
      I_Contact( #Mx_ET20 )
      I_Contact( #Mx_ET21 )
      I_Contact( #Mx_ET22 )
      I_Contact( #Mx_ET23 )
      I_Contact( #Mx_ET120 )
      I_Contact( #Mx_ET121 )
      Coil( #Aux_ET00 )
   END_RUNG
   // the same network as SCL:
   #Aux_ET00 := NOT #Mx_ET20 AND NOT #Mx_ET21 AND NOT #Mx_ET22 AND NOT #Mx_ET23 AND NOT #Mx_ET120 AND NOT #Mx_ET121;
END_REGION

REGION Network 38: Aux_ET00
   RUNG wire#powerrail
      Contact( #Aux_ET00 )
      I_Contact( #Mx_ET50 )
      I_Contact( #Mx_ET51 )
      I_Contact( #Mx_ET52 )
      I_Contact( #Mx_ET150 )
      I_Contact( #Mx_ET151 )
      I_Contact( #Mx_ET250 )
      Coil( #Aux_ET00 )
   END_RUNG
   // the same network as SCL:
   #Aux_ET00 := #Aux_ET00 AND NOT #Mx_ET50 AND NOT #Mx_ET51 AND NOT #Mx_ET52 AND NOT #Mx_ET150 AND NOT #Mx_ET151 AND NOT #Mx_ET250;
END_REGION

REGION Network 39: Aux_ET00
   RUNG wire#powerrail
      Contact( #Aux_ET00 )
      I_Contact( #Mx_ET60 )
      I_Contact( #Mx_ET61 )
      I_Contact( #Mx_ET160 )
      I_Contact( #Mx_ET161 )
      I_Contact( #Mx_ET260 )
      I_Contact( #Mx_ET90 )
      I_Contact( #Mx_ET91 )
      Coil( #Aux_ET00 )
   END_RUNG
   // the same network as SCL:
   #Aux_ET00 := #Aux_ET00 AND NOT #Mx_ET60 AND NOT #Mx_ET61 AND NOT #Mx_ET160 AND NOT #Mx_ET161 AND NOT #Mx_ET260 AND NOT #Mx_ET90 AND NOT #Mx_ET91;
END_REGION

REGION Network 40: ET00
   RUNG wire#powerrail
      Contact( #Aux_ET00 )
      I_Contact( #Mx_ET00 )
      I_Contact( #Mx_ET01 )
      I_Contact( #Mx_ET02 )
      I_Contact( #Mx_RES01 )
      I_Contact( #Mx_RES02 )
      I_Contact( #Mx_RES03 )
      I_Contact( #Mx_RES09 )
      S_SR(operand := #Mx_ET00, r1 := wire#w1)
   END_RUNG
   RUNG wire#powerrail
      Contact( #Mx_ET01 )
   END_RUNG wire#w1
   RUNG wire#powerrail
      Contact( #Mx_RES09 )
   END_RUNG wire#w1
   RUNG wire#powerrail
      Contact( #Mx_RES01 )
   END_RUNG wire#w1
   // the same network as SCL:
   IF #Aux_ET00 AND NOT #Mx_ET00 AND NOT #Mx_ET01 AND NOT #Mx_ET02 AND NOT #Mx_RES01 AND NOT #Mx_RES02 AND NOT #Mx_RES03 AND NOT #Mx_RES09 THEN
       #Mx_ET00 := TRUE;   // SR flip-flop
   END_IF;
   IF #Mx_ET01 OR #Mx_RES09 OR #Mx_RES01 THEN #Mx_ET00 := FALSE; END_IF;
END_REGION

REGION Network 41: ERROR - Termico Tx
   RUNG wire#powerrail
      Contact( #EstadoZona.Rearme_CBx )
      S_RS(operand := #EstadoVI.Err_Termico_E1_E3, s1 := wire#w1)
      S_Coil( #EstadoVI.Error_Mx )
   END_RUNG
   RUNG wire#powerrail
      I_Contact( #Termico_Tx )
      I_Contact( "Activar_Simulador" )
   END_RUNG wire#w1
   // the same network as SCL:
   IF #EstadoZona.Rearme_CBx THEN
       #EstadoVI.Err_Termico_E1_E3 := FALSE;   // RS flip-flop
   END_IF;
   IF NOT #Termico_Tx AND NOT "Activar_Simulador" THEN #EstadoVI.Err_Termico_E1_E3 := TRUE; END_IF;
   IF #EstadoVI.Err_Termico_E1_E3 THEN #EstadoVI.Error_Mx := TRUE; END_IF;
END_REGION

REGION Network 42: ERROR - Termico TRx
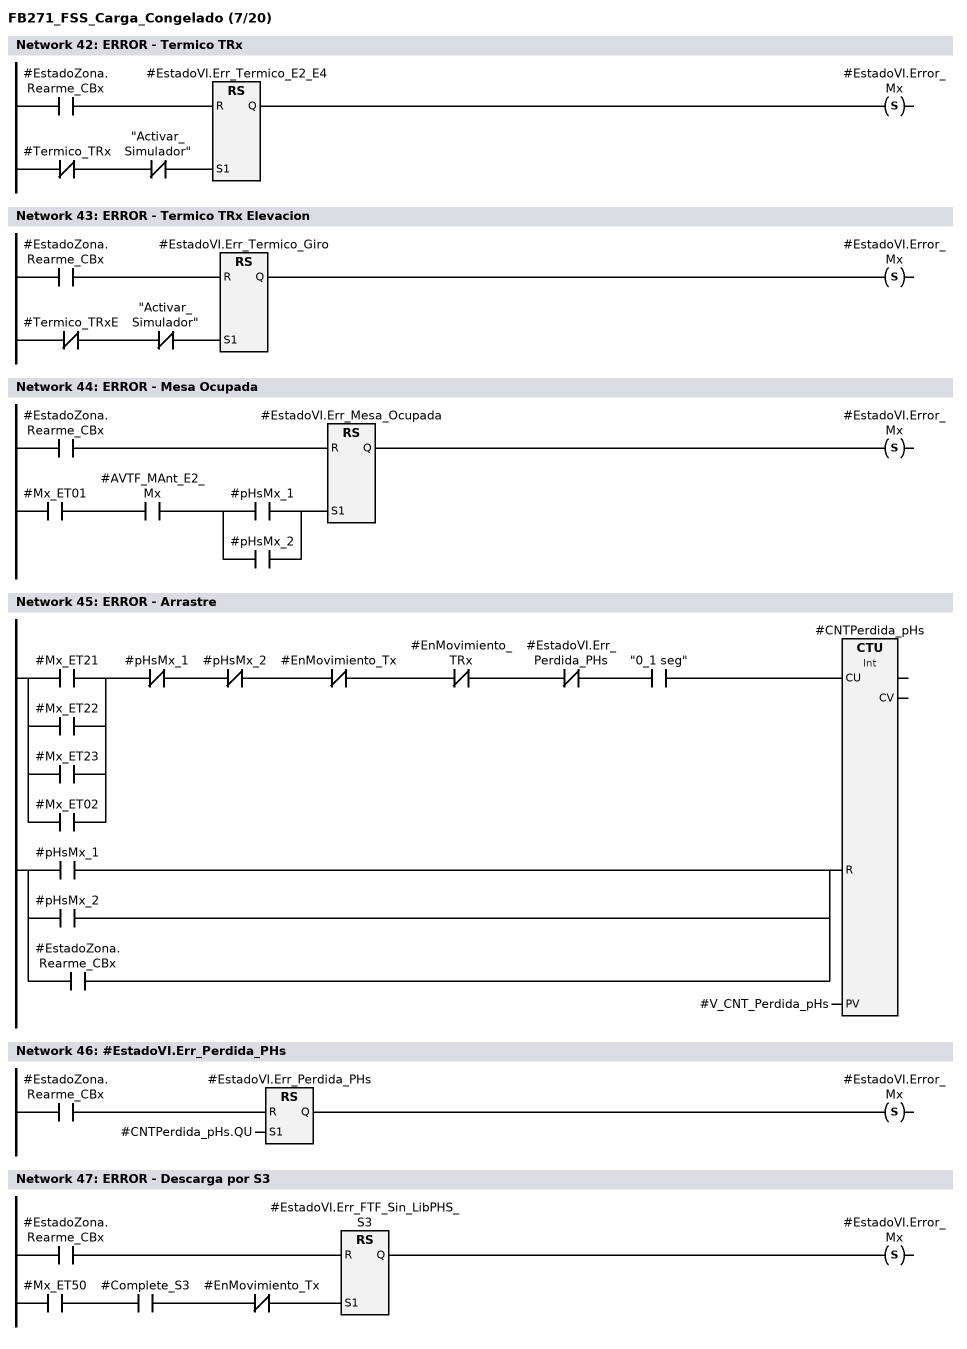
   RUNG wire#powerrail
      Contact( #EstadoZona.Rearme_CBx )
      S_RS(operand := #EstadoVI.Err_Termico_E2_E4, s1 := wire#w1)
      S_Coil( #EstadoVI.Error_Mx )
   END_RUNG
   RUNG wire#powerrail
      I_Contact( #Termico_TRx )
      I_Contact( "Activar_Simulador" )
   END_RUNG wire#w1
   // the same network as SCL:
   IF #EstadoZona.Rearme_CBx THEN
       #EstadoVI.Err_Termico_E2_E4 := FALSE;   // RS flip-flop
   END_IF;
   IF NOT #Termico_TRx AND NOT "Activar_Simulador" THEN #EstadoVI.Err_Termico_E2_E4 := TRUE; END_IF;
   IF #EstadoVI.Err_Termico_E2_E4 THEN #EstadoVI.Error_Mx := TRUE; END_IF;
END_REGION

REGION Network 43: ERROR - Termico TRx Elevacion
   RUNG wire#powerrail
      Contact( #EstadoZona.Rearme_CBx )
      S_RS(operand := #EstadoVI.Err_Termico_Giro, s1 := wire#w1)
      S_Coil( #EstadoVI.Error_Mx )
   END_RUNG
   RUNG wire#powerrail
      I_Contact( #Termico_TRxE )
      I_Contact( "Activar_Simulador" )
   END_RUNG wire#w1
   // the same network as SCL:
   IF #EstadoZona.Rearme_CBx THEN
       #EstadoVI.Err_Termico_Giro := FALSE;   // RS flip-flop
   END_IF;
   IF NOT #Termico_TRxE AND NOT "Activar_Simulador" THEN #EstadoVI.Err_Termico_Giro := TRUE; END_IF;
   IF #EstadoVI.Err_Termico_Giro THEN #EstadoVI.Error_Mx := TRUE; END_IF;
END_REGION

REGION Network 44: ERROR - Mesa Ocupada
   RUNG wire#powerrail
      Contact( #EstadoZona.Rearme_CBx )
      S_RS(operand := #EstadoVI.Err_Mesa_Ocupada, s1 := wire#w2)
      S_Coil( #EstadoVI.Error_Mx )
   END_RUNG
   RUNG wire#powerrail
      Contact( #Mx_ET01 )
      Contact( #AVTF_MAnt_E2_Mx )
      wire#w1
      Contact( #pHsMx_1 )
   END_RUNG wire#w2
   RUNG wire#w1
      Contact( #pHsMx_2 )
   END_RUNG wire#w2
   // the same network as SCL:
   IF #EstadoZona.Rearme_CBx THEN
       #EstadoVI.Err_Mesa_Ocupada := FALSE;   // RS flip-flop
   END_IF;
   IF #Mx_ET01 AND #AVTF_MAnt_E2_Mx AND (#pHsMx_1 OR #pHsMx_2) THEN
       #EstadoVI.Err_Mesa_Ocupada := TRUE;
   END_IF;
   IF #EstadoVI.Err_Mesa_Ocupada THEN #EstadoVI.Error_Mx := TRUE; END_IF;
END_REGION

REGION Network 45: ERROR - Arrastre
   RUNG wire#powerrail
      Contact( #Mx_ET21 )
      wire#w1
      I_Contact( #pHsMx_1 )
      I_Contact( #pHsMx_2 )
      I_Contact( #EnMovimiento_Tx )
      I_Contact( #EnMovimiento_TRx )
      I_Contact( #EstadoVI.Err_Perdida_PHs )
      Contact( "0_1 seg" )
      { S7_Templates := "value_type := Int" } #CNTPerdida_pHs.CTU(r := wire#w2, pv := #V_CNT_Perdida_pHs, cv =>)
   END_RUNG
   RUNG wire#powerrail
      Contact( #Mx_ET22 )
   END_RUNG wire#w1
   RUNG wire#powerrail
      Contact( #Mx_ET23 )
   END_RUNG wire#w1
   RUNG wire#powerrail
      Contact( #Mx_ET02 )
   END_RUNG wire#w1
   RUNG wire#powerrail
      Contact( #pHsMx_1 )
   END_RUNG wire#w2
   RUNG wire#powerrail
      Contact( #pHsMx_2 )
   END_RUNG wire#w2
   RUNG wire#powerrail
      Contact( #EstadoZona.Rearme_CBx )
   END_RUNG wire#w2
   // the same network as SCL:
   #CNTPerdida_pHs(CU := (#Mx_ET21 OR #Mx_ET22 OR #Mx_ET23 OR #Mx_ET02) AND NOT #pHsMx_1 AND NOT #pHsMx_2 AND NOT #EnMovimiento_Tx AND NOT #EnMovimiento_TRx AND NOT #EstadoVI.Err_Perdida_PHs AND "0_1 seg",   // CTU
                   R := #pHsMx_1 OR #pHsMx_2 OR #EstadoZona.Rearme_CBx,
                   PV := #V_CNT_Perdida_pHs);
END_REGION

REGION Network 46: #EstadoVI.Err_Perdida_PHs
   RUNG wire#powerrail
      Contact( #EstadoZona.Rearme_CBx )
      S_RS(operand := #EstadoVI.Err_Perdida_PHs, s1 := #CNTPerdida_pHs.QU)
      S_Coil( #EstadoVI.Error_Mx )
   END_RUNG
   // the same network as SCL:
   IF #EstadoZona.Rearme_CBx THEN
       #EstadoVI.Err_Perdida_PHs := FALSE;   // RS flip-flop
   END_IF;
   IF #CNTPerdida_pHs.QU THEN #EstadoVI.Err_Perdida_PHs := TRUE; END_IF;
   IF #EstadoVI.Err_Perdida_PHs THEN #EstadoVI.Error_Mx := TRUE; END_IF;
END_REGION

REGION Network 47: ERROR - Descarga por S3
   RUNG wire#powerrail
      Contact( #EstadoZona.Rearme_CBx )
      S_RS(operand := #EstadoVI.Err_FTF_Sin_LibPHS_S3, s1 := wire#w1)
      S_Coil( #EstadoVI.Error_Mx )
   END_RUNG
   RUNG wire#powerrail
      Contact( #Mx_ET50 )
      Contact( #Complete_S3 )
      I_Contact( #EnMovimiento_Tx )
   END_RUNG wire#w1
   // the same network as SCL:
   IF #EstadoZona.Rearme_CBx THEN
       #EstadoVI.Err_FTF_Sin_LibPHS_S3 := FALSE;   // RS flip-flop
   END_IF;
   IF #Mx_ET50 AND #Complete_S3 AND NOT #EnMovimiento_Tx THEN
       #EstadoVI.Err_FTF_Sin_LibPHS_S3 := TRUE;
   END_IF;
   IF #EstadoVI.Err_FTF_Sin_LibPHS_S3 THEN #EstadoVI.Error_Mx := TRUE; END_IF;
END_REGION

REGION Network 48: ERROR - Descarga por S4
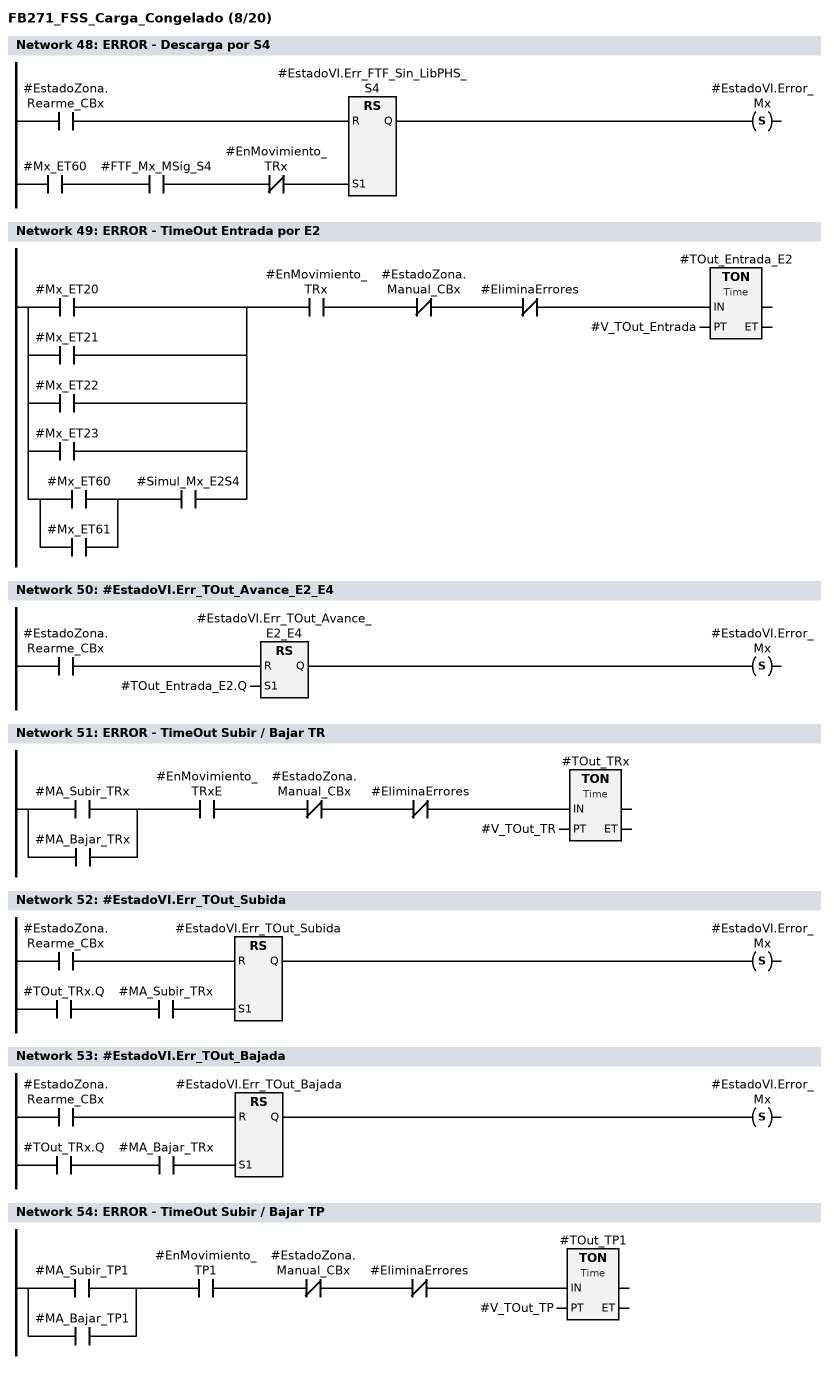
   RUNG wire#powerrail
      Contact( #EstadoZona.Rearme_CBx )
      S_RS(operand := #EstadoVI.Err_FTF_Sin_LibPHS_S4, s1 := wire#w1)
      S_Coil( #EstadoVI.Error_Mx )
   END_RUNG
   RUNG wire#powerrail
      Contact( #Mx_ET60 )
      Contact( #FTF_Mx_MSig_S4 )
      I_Contact( #EnMovimiento_TRx )
   END_RUNG wire#w1
   // the same network as SCL:
   IF #EstadoZona.Rearme_CBx THEN
       #EstadoVI.Err_FTF_Sin_LibPHS_S4 := FALSE;   // RS flip-flop
   END_IF;
   IF #Mx_ET60 AND #FTF_Mx_MSig_S4 AND NOT #EnMovimiento_TRx THEN
       #EstadoVI.Err_FTF_Sin_LibPHS_S4 := TRUE;
   END_IF;
   IF #EstadoVI.Err_FTF_Sin_LibPHS_S4 THEN #EstadoVI.Error_Mx := TRUE; END_IF;
END_REGION

REGION Network 49: ERROR - TimeOut Entrada por E2
   RUNG wire#powerrail
      Contact( #Mx_ET20 )
      wire#w1
      Contact( #EnMovimiento_TRx )
      I_Contact( #EstadoZona.Manual_CBx )
      I_Contact( #EliminaErrores )
      { S7_Templates := "time_type := Time" } #TOut_Entrada_E2.TON(pt := #V_TOut_Entrada, et =>)
   END_RUNG
   RUNG wire#powerrail
      Contact( #Mx_ET21 )
   END_RUNG wire#w1
   RUNG wire#powerrail
      Contact( #Mx_ET22 )
   END_RUNG wire#w1
   RUNG wire#powerrail
      Contact( #Mx_ET23 )
   END_RUNG wire#w1
   RUNG wire#powerrail
      Contact( #Mx_ET60 )
      wire#w2
      Contact( #Simul_Mx_E2S4 )
   END_RUNG wire#w1
   RUNG wire#powerrail
      Contact( #Mx_ET61 )
   END_RUNG wire#w2
   // the same network as SCL:
   #TOut_Entrada_E2(IN := (#Mx_ET20 OR #Mx_ET21 OR #Mx_ET22 OR #Mx_ET23 OR ((#Mx_ET60 OR #Mx_ET61) AND #Simul_Mx_E2S4)) AND #EnMovimiento_TRx AND NOT #EstadoZona.Manual_CBx AND NOT #EliminaErrores,   // TON
                    PT := #V_TOut_Entrada);
END_REGION

REGION Network 50: #EstadoVI.Err_TOut_Avance_E2_E4
   RUNG wire#powerrail
      Contact( #EstadoZona.Rearme_CBx )
      S_RS(operand := #EstadoVI.Err_TOut_Avance_E2_E4, s1 := #TOut_Entrada_E2.Q)
      S_Coil( #EstadoVI.Error_Mx )
   END_RUNG
   // the same network as SCL:
   IF #EstadoZona.Rearme_CBx THEN
       #EstadoVI.Err_TOut_Avance_E2_E4 := FALSE;   // RS flip-flop
   END_IF;
   IF #TOut_Entrada_E2.Q THEN #EstadoVI.Err_TOut_Avance_E2_E4 := TRUE; END_IF;
   IF #EstadoVI.Err_TOut_Avance_E2_E4 THEN #EstadoVI.Error_Mx := TRUE; END_IF;
END_REGION

REGION Network 51: ERROR - TimeOut Subir / Bajar TR
   RUNG wire#powerrail
      Contact( #MA_Subir_TRx )
      wire#w1
      Contact( #EnMovimiento_TRxE )
      I_Contact( #EstadoZona.Manual_CBx )
      I_Contact( #EliminaErrores )
      { S7_Templates := "time_type := Time" } #TOut_TRx.TON(pt := #V_TOut_TR, et =>)
   END_RUNG
   RUNG wire#powerrail
      Contact( #MA_Bajar_TRx )
   END_RUNG wire#w1
   // the same network as SCL:
   #TOut_TRx(IN := (#MA_Subir_TRx OR #MA_Bajar_TRx) AND #EnMovimiento_TRxE AND NOT #EstadoZona.Manual_CBx AND NOT #EliminaErrores,   // TON
             PT := #V_TOut_TR);
END_REGION

REGION Network 52: #EstadoVI.Err_TOut_Subida
   RUNG wire#powerrail
      Contact( #EstadoZona.Rearme_CBx )
      S_RS(operand := #EstadoVI.Err_TOut_Subida, s1 := wire#w1)
      S_Coil( #EstadoVI.Error_Mx )
   END_RUNG
   RUNG wire#powerrail
      Contact( #TOut_TRx.Q )
      Contact( #MA_Subir_TRx )
   END_RUNG wire#w1
   // the same network as SCL:
   IF #EstadoZona.Rearme_CBx THEN
       #EstadoVI.Err_TOut_Subida := FALSE;   // RS flip-flop
   END_IF;
   IF #TOut_TRx.Q AND #MA_Subir_TRx THEN #EstadoVI.Err_TOut_Subida := TRUE; END_IF;
   IF #EstadoVI.Err_TOut_Subida THEN #EstadoVI.Error_Mx := TRUE; END_IF;
END_REGION

REGION Network 53: #EstadoVI.Err_TOut_Bajada
   RUNG wire#powerrail
      Contact( #EstadoZona.Rearme_CBx )
      S_RS(operand := #EstadoVI.Err_TOut_Bajada, s1 := wire#w1)
      S_Coil( #EstadoVI.Error_Mx )
   END_RUNG
   RUNG wire#powerrail
      Contact( #TOut_TRx.Q )
      Contact( #MA_Bajar_TRx )
   END_RUNG wire#w1
   // the same network as SCL:
   IF #EstadoZona.Rearme_CBx THEN
       #EstadoVI.Err_TOut_Bajada := FALSE;   // RS flip-flop
   END_IF;
   IF #TOut_TRx.Q AND #MA_Bajar_TRx THEN #EstadoVI.Err_TOut_Bajada := TRUE; END_IF;
   IF #EstadoVI.Err_TOut_Bajada THEN #EstadoVI.Error_Mx := TRUE; END_IF;
END_REGION

REGION Network 54: ERROR - TimeOut Subir / Bajar TP
   RUNG wire#powerrail
      Contact( #MA_Subir_TP1 )
      wire#w1
      Contact( #EnMovimiento_TP1 )
      I_Contact( #EstadoZona.Manual_CBx )
      I_Contact( #EliminaErrores )
      { S7_Templates := "time_type := Time" } #TOut_TP1.TON(pt := #V_TOut_TP, et =>)
   END_RUNG
   RUNG wire#powerrail
      Contact( #MA_Bajar_TP1 )
   END_RUNG wire#w1
   // the same network as SCL:
   #TOut_TP1(IN := (#MA_Subir_TP1 OR #MA_Bajar_TP1) AND #EnMovimiento_TP1 AND NOT #EstadoZona.Manual_CBx AND NOT #EliminaErrores,   // TON
             PT := #V_TOut_TP);
END_REGION

REGION Network 55: #TOut_TP2
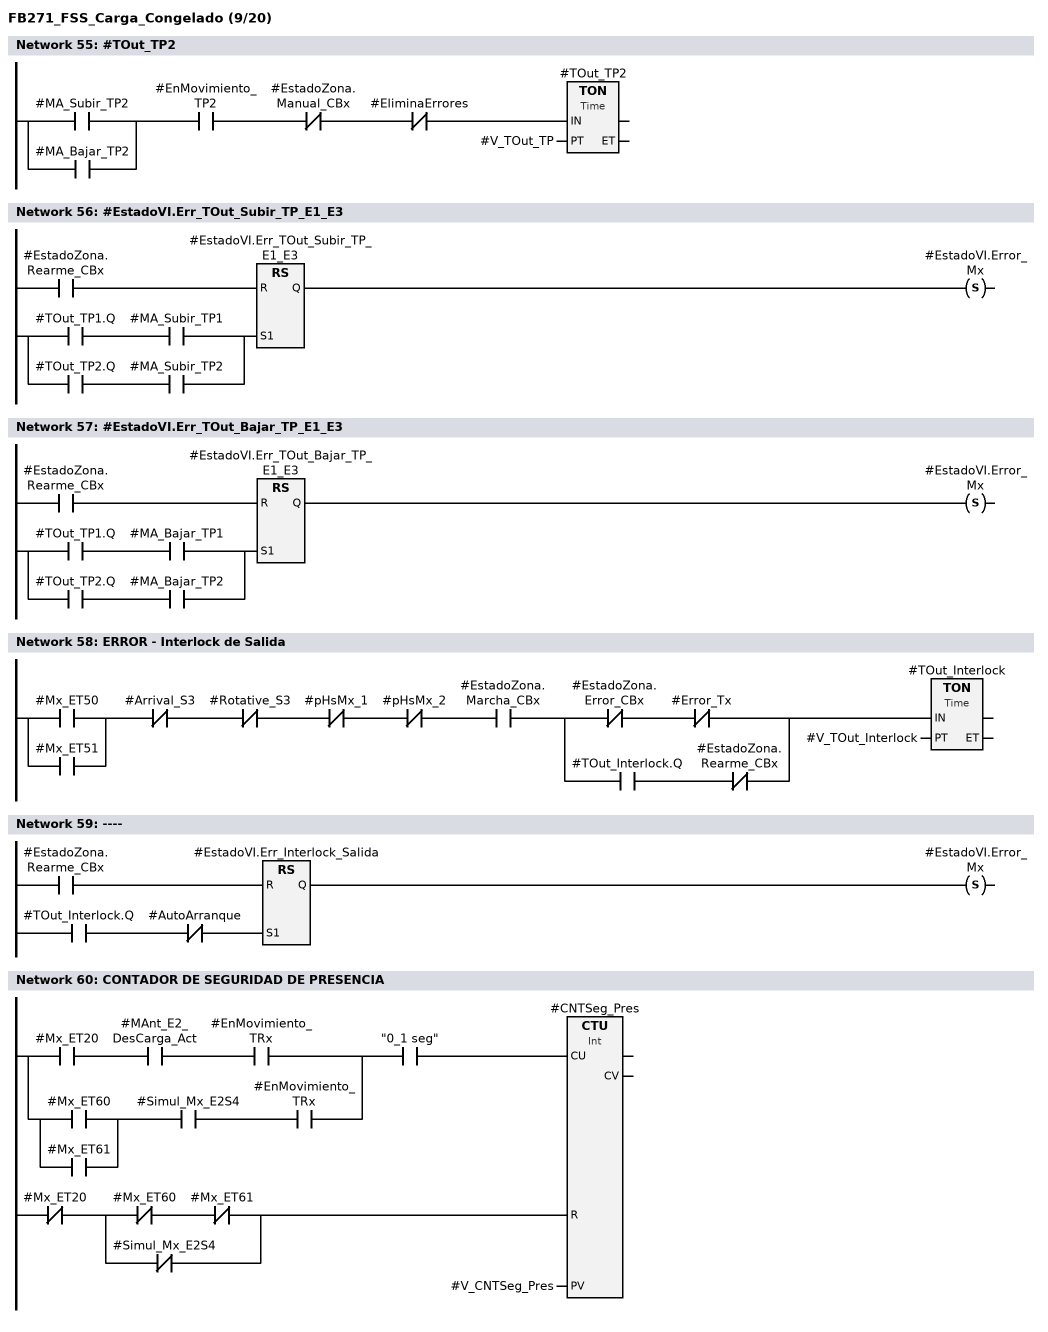
   RUNG wire#powerrail
      Contact( #MA_Subir_TP2 )
      wire#w1
      Contact( #EnMovimiento_TP2 )
      I_Contact( #EstadoZona.Manual_CBx )
      I_Contact( #EliminaErrores )
      { S7_Templates := "time_type := Time" } #TOut_TP2.TON(pt := #V_TOut_TP, et =>)
   END_RUNG
   RUNG wire#powerrail
      Contact( #MA_Bajar_TP2 )
   END_RUNG wire#w1
   // the same network as SCL:
   #TOut_TP2(IN := (#MA_Subir_TP2 OR #MA_Bajar_TP2) AND #EnMovimiento_TP2 AND NOT #EstadoZona.Manual_CBx AND NOT #EliminaErrores,   // TON
             PT := #V_TOut_TP);
END_REGION

REGION Network 56: #EstadoVI.Err_TOut_Subir_TP_E1_E3
   RUNG wire#powerrail
      Contact( #EstadoZona.Rearme_CBx )
      S_RS(operand := #EstadoVI.Err_TOut_Subir_TP_E1_E3, s1 := wire#w1)
      S_Coil( #EstadoVI.Error_Mx )
   END_RUNG
   RUNG wire#powerrail
      Contact( #TOut_TP1.Q )
      Contact( #MA_Subir_TP1 )
   END_RUNG wire#w1
   RUNG wire#powerrail
      Contact( #TOut_TP2.Q )
      Contact( #MA_Subir_TP2 )
   END_RUNG wire#w1
   // the same network as SCL:
   IF #EstadoZona.Rearme_CBx THEN
       #EstadoVI.Err_TOut_Subir_TP_E1_E3 := FALSE;   // RS flip-flop
   END_IF;
   IF (#TOut_TP1.Q AND #MA_Subir_TP1) OR (#TOut_TP2.Q AND #MA_Subir_TP2) THEN
       #EstadoVI.Err_TOut_Subir_TP_E1_E3 := TRUE;
   END_IF;
   IF #EstadoVI.Err_TOut_Subir_TP_E1_E3 THEN #EstadoVI.Error_Mx := TRUE; END_IF;
END_REGION

REGION Network 57: #EstadoVI.Err_TOut_Bajar_TP_E1_E3
   RUNG wire#powerrail
      Contact( #EstadoZona.Rearme_CBx )
      S_RS(operand := #EstadoVI.Err_TOut_Bajar_TP_E1_E3, s1 := wire#w1)
      S_Coil( #EstadoVI.Error_Mx )
   END_RUNG
   RUNG wire#powerrail
      Contact( #TOut_TP1.Q )
      Contact( #MA_Bajar_TP1 )
   END_RUNG wire#w1
   RUNG wire#powerrail
      Contact( #TOut_TP2.Q )
      Contact( #MA_Bajar_TP2 )
   END_RUNG wire#w1
   // the same network as SCL:
   IF #EstadoZona.Rearme_CBx THEN
       #EstadoVI.Err_TOut_Bajar_TP_E1_E3 := FALSE;   // RS flip-flop
   END_IF;
   IF (#TOut_TP1.Q AND #MA_Bajar_TP1) OR (#TOut_TP2.Q AND #MA_Bajar_TP2) THEN
       #EstadoVI.Err_TOut_Bajar_TP_E1_E3 := TRUE;
   END_IF;
   IF #EstadoVI.Err_TOut_Bajar_TP_E1_E3 THEN #EstadoVI.Error_Mx := TRUE; END_IF;
END_REGION

REGION Network 58: ERROR - Interlock de Salida
   RUNG wire#powerrail
      Contact( #Mx_ET50 )
      wire#w1
      I_Contact( #Arrival_S3 )
      I_Contact( #Rotative_S3 )
      I_Contact( #pHsMx_1 )
      I_Contact( #pHsMx_2 )
      Contact( #EstadoZona.Marcha_CBx )
      wire#w2
      I_Contact( #EstadoZona.Error_CBx )
      I_Contact( #Error_Tx )
      wire#w3
      { S7_Templates := "time_type := Time" } #TOut_Interlock.TON(pt := #V_TOut_Interlock, et =>)
   END_RUNG
   RUNG wire#powerrail
      Contact( #Mx_ET51 )
   END_RUNG wire#w1
   RUNG wire#w2
      Contact( #TOut_Interlock.Q )
      I_Contact( #EstadoZona.Rearme_CBx )
   END_RUNG wire#w3
   // the same network as SCL:
   #TOut_Interlock(IN := (#Mx_ET50 OR #Mx_ET51) AND NOT #Arrival_S3 AND NOT #Rotative_S3 AND NOT #pHsMx_1 AND NOT #pHsMx_2 AND #EstadoZona.Marcha_CBx AND ((NOT #EstadoZona.Error_CBx AND NOT #Error_Tx) OR (#TOut_Interlock.Q AND NOT #EstadoZona.Rearme_CBx)),   // TON
                   PT := #V_TOut_Interlock);
END_REGION

REGION Network 59: ----
   RUNG wire#powerrail
      Contact( #EstadoZona.Rearme_CBx )
      S_RS(operand := #EstadoVI.Err_Interlock_Salida, s1 := wire#w1)
      S_Coil( #EstadoVI.Error_Mx )
   END_RUNG
   RUNG wire#powerrail
      Contact( #TOut_Interlock.Q )
      I_Contact( #AutoArranque )
   END_RUNG wire#w1
   // the same network as SCL:
   IF #EstadoZona.Rearme_CBx THEN
       #EstadoVI.Err_Interlock_Salida := FALSE;   // RS flip-flop
   END_IF;
   IF #TOut_Interlock.Q AND NOT #AutoArranque THEN #EstadoVI.Err_Interlock_Salida := TRUE; END_IF;
   IF #EstadoVI.Err_Interlock_Salida THEN #EstadoVI.Error_Mx := TRUE; END_IF;
END_REGION

REGION Network 60: CONTADOR DE SEGURIDAD DE PRESENCIA
   RUNG wire#powerrail
      Contact( #Mx_ET20 )
      Contact( #MAnt_E2_DesCarga_Act )
      Contact( #EnMovimiento_TRx )
      wire#w1
      Contact( "0_1 seg" )
      { S7_Templates := "value_type := Int" } #CNTSeg_Pres.CTU(r := wire#w4, pv := #V_CNTSeg_Pres, cv =>)
   END_RUNG
   RUNG wire#powerrail
      Contact( #Mx_ET60 )
      wire#w2
      Contact( #Simul_Mx_E2S4 )
      Contact( #EnMovimiento_TRx )
   END_RUNG wire#w1
   RUNG wire#powerrail
      Contact( #Mx_ET61 )
   END_RUNG wire#w2
   RUNG wire#powerrail
      I_Contact( #Mx_ET20 )
      wire#w3
      I_Contact( #Mx_ET60 )
      I_Contact( #Mx_ET61 )
   END_RUNG wire#w4
   RUNG wire#w3
      I_Contact( #Simul_Mx_E2S4 )
   END_RUNG wire#w4
   // the same network as SCL:
   #CNTSeg_Pres(CU := ((#Mx_ET20 AND #MAnt_E2_DesCarga_Act AND #EnMovimiento_TRx) OR ((#Mx_ET60 OR #Mx_ET61) AND #Simul_Mx_E2S4 AND #EnMovimiento_TRx)) AND "0_1 seg",   // CTU
                R := NOT #Mx_ET20 AND ((NOT #Mx_ET60 AND NOT #Mx_ET61) OR NOT #Simul_Mx_E2S4),
                PV := #V_CNTSeg_Pres);
END_REGION

REGION Network 61: CONTADOR DE PRESENCIA - Entrada por E2
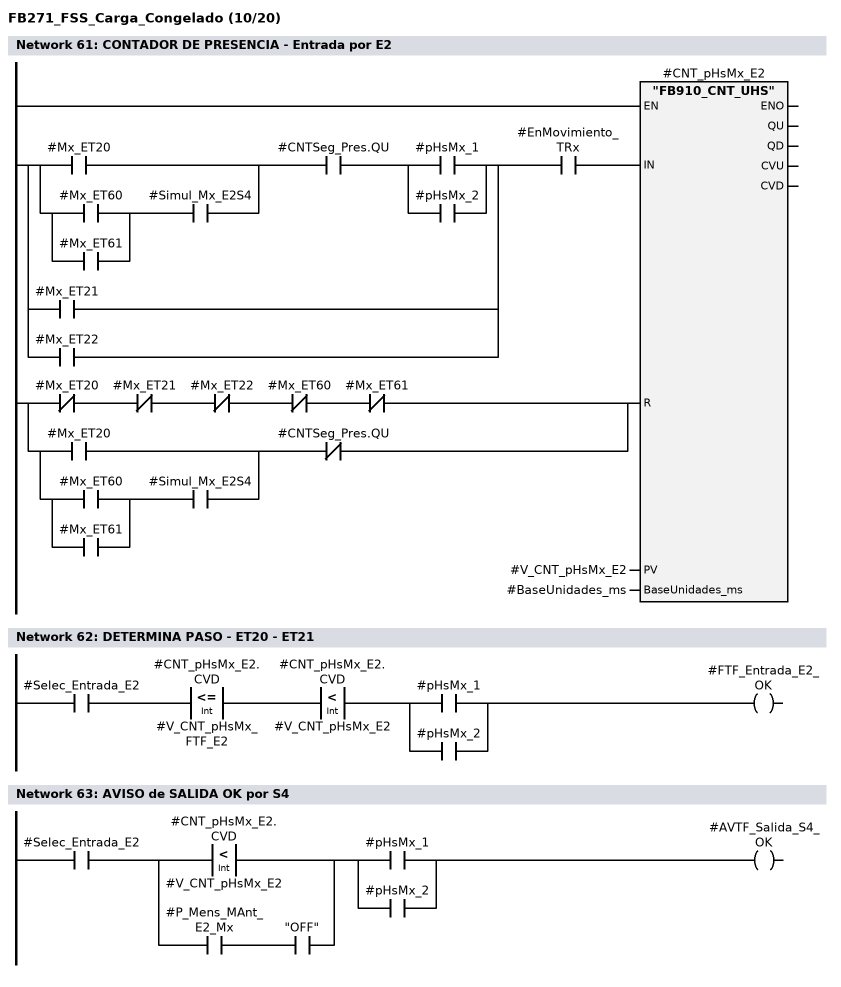
   RUNG wire#powerrail
      #CNT_pHsMx_E2(IN := wire#w5, R := wire#w8, PV := #V_CNT_pHsMx_E2, BaseUnidades_ms := #BaseUnidades_ms, QU =>, QD =>, CVU =>, CVD =>)
   END_RUNG
   RUNG wire#powerrail
      Contact( #Mx_ET20 )
      wire#w1
      Contact( #CNTSeg_Pres.QU )
      wire#w3
      Contact( #pHsMx_1 )
      wire#w4
      Contact( #EnMovimiento_TRx )
   END_RUNG wire#w5
   RUNG wire#powerrail
      Contact( #Mx_ET60 )
      wire#w2
      Contact( #Simul_Mx_E2S4 )
   END_RUNG wire#w1
   RUNG wire#powerrail
      Contact( #Mx_ET61 )
   END_RUNG wire#w2
   RUNG wire#w3
      Contact( #pHsMx_2 )
   END_RUNG wire#w4
   RUNG wire#powerrail
      Contact( #Mx_ET21 )
   END_RUNG wire#w4
   RUNG wire#powerrail
      Contact( #Mx_ET22 )
   END_RUNG wire#w4
   RUNG wire#powerrail
      I_Contact( #Mx_ET20 )
      I_Contact( #Mx_ET21 )
      I_Contact( #Mx_ET22 )
      I_Contact( #Mx_ET60 )
      I_Contact( #Mx_ET61 )
   END_RUNG wire#w8
   RUNG wire#powerrail
      Contact( #Mx_ET20 )
      wire#w6
      I_Contact( #CNTSeg_Pres.QU )
   END_RUNG wire#w8
   RUNG wire#powerrail
      Contact( #Mx_ET60 )
      wire#w7
      Contact( #Simul_Mx_E2S4 )
   END_RUNG wire#w6
   RUNG wire#powerrail
      Contact( #Mx_ET61 )
   END_RUNG wire#w7
   // the same network as SCL:
   #CNT_pHsMx_E2(IN := (((#Mx_ET20 OR ((#Mx_ET60 OR #Mx_ET61) AND #Simul_Mx_E2S4)) AND #CNTSeg_Pres.QU AND (#pHsMx_1 OR #pHsMx_2)) OR #Mx_ET21 OR #Mx_ET22) AND #EnMovimiento_TRx,   // "FB910_CNT_UHS"
                 R := (NOT #Mx_ET20 AND NOT #Mx_ET21 AND NOT #Mx_ET22 AND NOT #Mx_ET60 AND NOT #Mx_ET61) OR ((#Mx_ET20 OR ((#Mx_ET60 OR #Mx_ET61) AND #Simul_Mx_E2S4)) AND NOT #CNTSeg_Pres.QU),
                 PV := #V_CNT_pHsMx_E2,
                 BaseUnidades_ms := #BaseUnidades_ms);
END_REGION

REGION Network 62: DETERMINA PASO - ET20 - ET21
   RUNG wire#powerrail
      Contact( #Selec_Entrada_E2 )
      { S7_Templates := "SrcType := Int" } LE_Contact(in1 := #CNT_pHsMx_E2.CVD, in2 := #V_CNT_pHsMx_FTF_E2)
      { S7_Templates := "SrcType := Int" } LT_Contact(in1 := #CNT_pHsMx_E2.CVD, in2 := #V_CNT_pHsMx_E2)
      wire#w1
      Contact( #pHsMx_1 )
      wire#w2
      Coil( #FTF_Entrada_E2_OK )
   END_RUNG
   RUNG wire#w1
      Contact( #pHsMx_2 )
   END_RUNG wire#w2
   // the same network as SCL:
   #FTF_Entrada_E2_OK := #Selec_Entrada_E2 AND (#CNT_pHsMx_E2.CVD <= #V_CNT_pHsMx_FTF_E2) AND (#CNT_pHsMx_E2.CVD < #V_CNT_pHsMx_E2) AND (#pHsMx_1 OR #pHsMx_2);
END_REGION

REGION Network 63: AVISO de SALIDA OK por S4
   RUNG wire#powerrail
      Contact( #Selec_Entrada_E2 )
      wire#w1
      { S7_Templates := "SrcType := Int" } LT_Contact(in1 := #CNT_pHsMx_E2.CVD, in2 := #V_CNT_pHsMx_E2)
      wire#w2
      Contact( #pHsMx_1 )
      wire#w3
      Coil( #AVTF_Salida_S4_OK )
   END_RUNG
   RUNG wire#w1
      Contact( #P_Mens_MAnt_E2_Mx )
      Contact( "OFF" )
   END_RUNG wire#w2
   RUNG wire#w2
      Contact( #pHsMx_2 )
   END_RUNG wire#w3
   // the same network as SCL:
   #AVTF_Salida_S4_OK := #Selec_Entrada_E2 AND ((#CNT_pHsMx_E2.CVD < #V_CNT_pHsMx_E2) OR (#P_Mens_MAnt_E2_Mx AND "OFF")) AND (#pHsMx_1 OR #pHsMx_2);
END_REGION

REGION Network 64: CONTADORES SEGURIDAD DE AUSENCIA
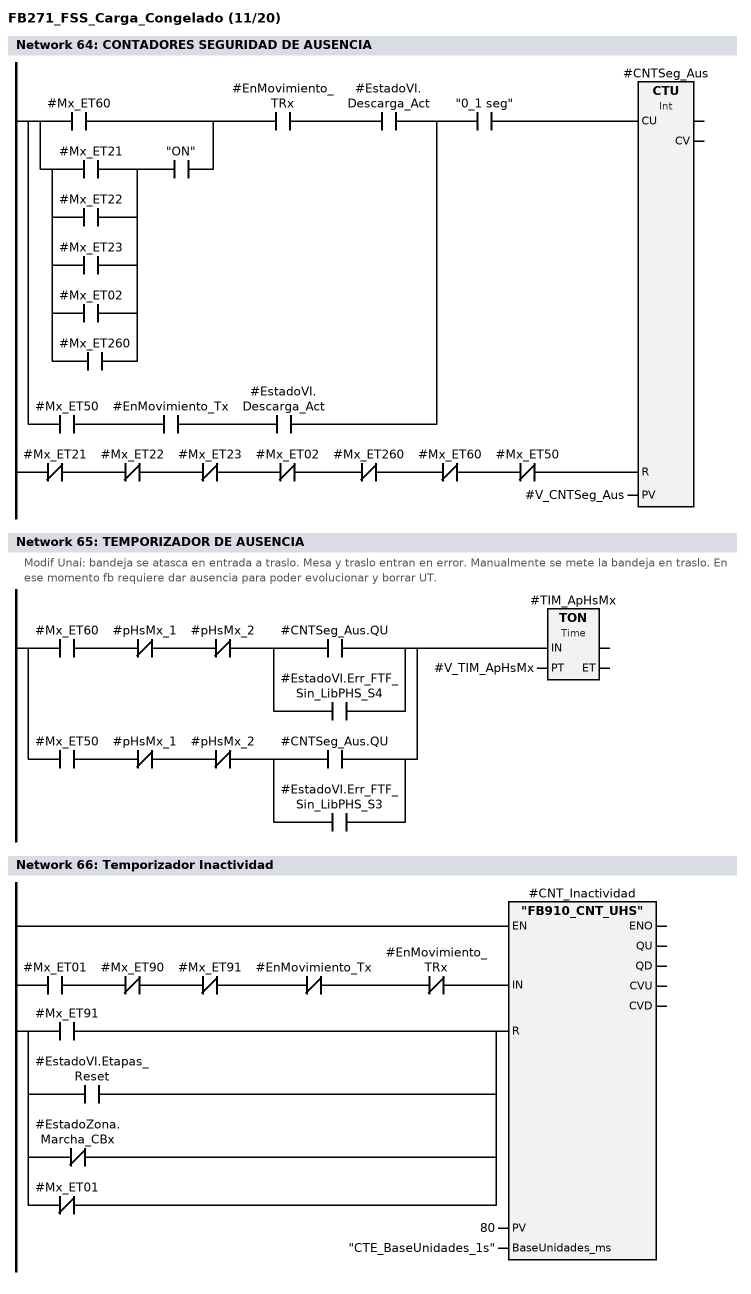
   RUNG wire#powerrail
      Contact( #Mx_ET60 )
      wire#w1
      Contact( #EnMovimiento_TRx )
      Contact( #EstadoVI.Descarga_Act )
      wire#w3
      Contact( "0_1 seg" )
      { S7_Templates := "value_type := Int" } #CNTSeg_Aus.CTU(r := wire#w4, pv := #V_CNTSeg_Aus, cv =>)
   END_RUNG
   RUNG wire#powerrail
      Contact( #Mx_ET21 )
      wire#w2
      Contact( "ON" )
   END_RUNG wire#w1
   RUNG wire#powerrail
      Contact( #Mx_ET22 )
   END_RUNG wire#w2
   RUNG wire#powerrail
      Contact( #Mx_ET23 )
   END_RUNG wire#w2
   RUNG wire#powerrail
      Contact( #Mx_ET02 )
   END_RUNG wire#w2
   RUNG wire#powerrail
      Contact( #Mx_ET260 )
   END_RUNG wire#w2
   RUNG wire#powerrail
      Contact( #Mx_ET50 )
      Contact( #EnMovimiento_Tx )
      Contact( #EstadoVI.Descarga_Act )
   END_RUNG wire#w3
   RUNG wire#powerrail
      I_Contact( #Mx_ET21 )
      I_Contact( #Mx_ET22 )
      I_Contact( #Mx_ET23 )
      I_Contact( #Mx_ET02 )
      I_Contact( #Mx_ET260 )
      I_Contact( #Mx_ET60 )
      I_Contact( #Mx_ET50 )
   END_RUNG wire#w4
   // the same network as SCL:
   #CNTSeg_Aus(CU := (((#Mx_ET60 OR ((#Mx_ET21 OR #Mx_ET22 OR #Mx_ET23 OR #Mx_ET02 OR #Mx_ET260) AND "ON")) AND #EnMovimiento_TRx AND #EstadoVI.Descarga_Act) OR (#Mx_ET50 AND #EnMovimiento_Tx AND #EstadoVI.Descarga_Act)) AND "0_1 seg",   // CTU
               R := NOT #Mx_ET21 AND NOT #Mx_ET22 AND NOT #Mx_ET23 AND NOT #Mx_ET02 AND NOT #Mx_ET260 AND NOT #Mx_ET60 AND NOT #Mx_ET50,
               PV := #V_CNTSeg_Aus);
END_REGION

REGION Network 65: TEMPORIZADOR DE AUSENCIA
   // Modif Unai: bandeja se atasca en entrada a traslo. Mesa y traslo entran en error. Manualmente se mete la bandeja en traslo. En ese momento fb requiere dar ausencia para poder evolucionar y borrar UT.
   RUNG wire#powerrail
      Contact( #Mx_ET60 )
      I_Contact( #pHsMx_1 )
      I_Contact( #pHsMx_2 )
      wire#w1
      Contact( #CNTSeg_Aus.QU )
      wire#w2
      { S7_Templates := "time_type := Time" } #TIM_ApHsMx.TON(pt := #V_TIM_ApHsMx, et =>)
   END_RUNG
   RUNG wire#w1
      Contact( #EstadoVI.Err_FTF_Sin_LibPHS_S4 )
   END_RUNG wire#w2
   RUNG wire#powerrail
      Contact( #Mx_ET50 )
      I_Contact( #pHsMx_1 )
      I_Contact( #pHsMx_2 )
      wire#w3
      Contact( #CNTSeg_Aus.QU )
   END_RUNG wire#w2
   RUNG wire#w3
      Contact( #EstadoVI.Err_FTF_Sin_LibPHS_S3 )
   END_RUNG wire#w2
   // the same network as SCL:
   #TIM_ApHsMx(IN := (#Mx_ET60 AND NOT #pHsMx_1 AND NOT #pHsMx_2 AND (#CNTSeg_Aus.QU OR #EstadoVI.Err_FTF_Sin_LibPHS_S4)) OR (#Mx_ET50 AND NOT #pHsMx_1 AND NOT #pHsMx_2 AND (#CNTSeg_Aus.QU OR #EstadoVI.Err_FTF_Sin_LibPHS_S3)),   // TON
               PT := #V_TIM_ApHsMx);
END_REGION

REGION Network 66: Temporizador Inactividad
   RUNG wire#powerrail
      #CNT_Inactividad(IN := wire#w1, R := wire#w2, PV := 80, BaseUnidades_ms := "CTE_BaseUnidades_1s", QU =>, QD =>, CVU =>, CVD =>)
   END_RUNG
   RUNG wire#powerrail
      Contact( #Mx_ET01 )
      I_Contact( #Mx_ET90 )
      I_Contact( #Mx_ET91 )
      I_Contact( #EnMovimiento_Tx )
      I_Contact( #EnMovimiento_TRx )
   END_RUNG wire#w1
   RUNG wire#powerrail
      Contact( #Mx_ET91 )
   END_RUNG wire#w2
   RUNG wire#powerrail
      Contact( #EstadoVI.Etapas_Reset )
   END_RUNG wire#w2
   RUNG wire#powerrail
      I_Contact( #EstadoZona.Marcha_CBx )
   END_RUNG wire#w2
   RUNG wire#powerrail
      I_Contact( #Mx_ET01 )
   END_RUNG wire#w2
   // the same network as SCL:
   #CNT_Inactividad(IN := #Mx_ET01 AND NOT #Mx_ET90 AND NOT #Mx_ET91 AND NOT #EnMovimiento_Tx AND NOT #EnMovimiento_TRx,   // "FB910_CNT_UHS"
                    R := #Mx_ET91 OR #EstadoVI.Etapas_Reset OR NOT #EstadoZona.Marcha_CBx OR NOT #Mx_ET01,
                    PV := 80,
                    BaseUnidades_ms := "CTE_BaseUnidades_1s");
END_REGION

REGION Network 67: VARIABLES AUXILIARES - Fin de Reset
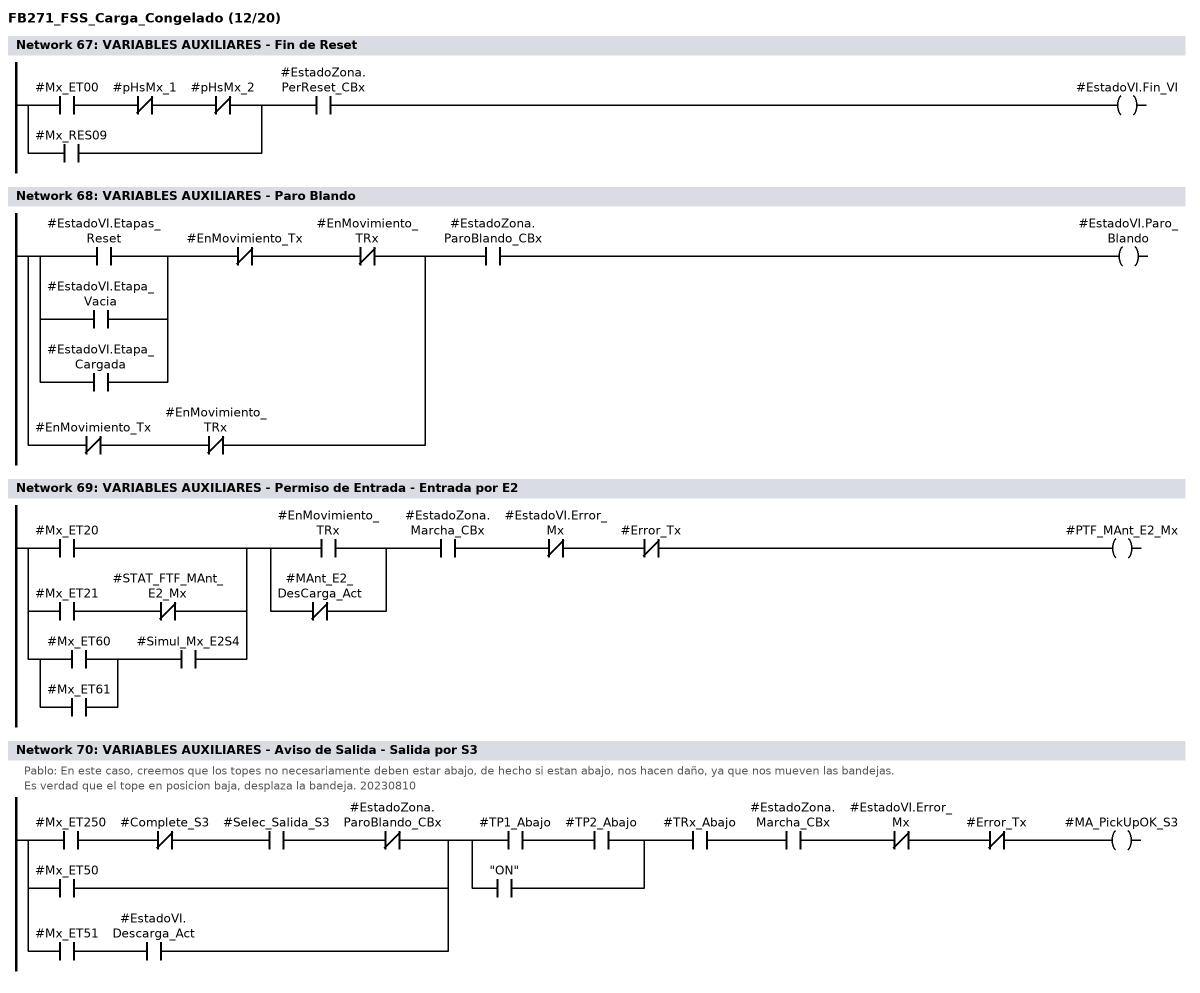
   RUNG wire#powerrail
      Contact( #Mx_ET00 )
      I_Contact( #pHsMx_1 )
      I_Contact( #pHsMx_2 )
      wire#w1
      Contact( #EstadoZona.PerReset_CBx )
      Coil( #EstadoVI.Fin_VI )
   END_RUNG
   RUNG wire#powerrail
      Contact( #Mx_RES09 )
   END_RUNG wire#w1
   // the same network as SCL:
   #EstadoVI.Fin_VI := ((#Mx_ET00 AND NOT #pHsMx_1 AND NOT #pHsMx_2) OR #Mx_RES09) AND #EstadoZona.PerReset_CBx;
END_REGION

REGION Network 68: VARIABLES AUXILIARES - Paro Blando
   RUNG wire#powerrail
      Contact( #EstadoVI.Etapas_Reset )
      wire#w1
      I_Contact( #EnMovimiento_Tx )
      I_Contact( #EnMovimiento_TRx )
      wire#w2
      Contact( #EstadoZona.ParoBlando_CBx )
      Coil( #EstadoVI.Paro_Blando )
   END_RUNG
   RUNG wire#powerrail
      Contact( #EstadoVI.Etapa_Vacia )
   END_RUNG wire#w1
   RUNG wire#powerrail
      Contact( #EstadoVI.Etapa_Cargada )
   END_RUNG wire#w1
   RUNG wire#powerrail
      I_Contact( #EnMovimiento_Tx )
      I_Contact( #EnMovimiento_TRx )
   END_RUNG wire#w2
   // the same network as SCL:
   #EstadoVI.Paro_Blando := (((#EstadoVI.Etapas_Reset OR #EstadoVI.Etapa_Vacia OR #EstadoVI.Etapa_Cargada) AND NOT #EnMovimiento_Tx AND NOT #EnMovimiento_TRx) OR (NOT #EnMovimiento_Tx AND NOT #EnMovimiento_TRx)) AND #EstadoZona.ParoBlando_CBx;
END_REGION

REGION Network 69: VARIABLES AUXILIARES - Permiso de Entrada - Entrada por E2
   RUNG wire#powerrail
      Contact( #Mx_ET20 )
      wire#w1
      Contact( #EnMovimiento_TRx )
      wire#w3
      Contact( #EstadoZona.Marcha_CBx )
      I_Contact( #EstadoVI.Error_Mx )
      I_Contact( #Error_Tx )
      Coil( #PTF_MAnt_E2_Mx )
   END_RUNG
   RUNG wire#powerrail
      Contact( #Mx_ET21 )
      I_Contact( #STAT_FTF_MAnt_E2_Mx )
   END_RUNG wire#w1
   RUNG wire#powerrail
      Contact( #Mx_ET60 )
      wire#w2
      Contact( #Simul_Mx_E2S4 )
   END_RUNG wire#w1
   RUNG wire#powerrail
      Contact( #Mx_ET61 )
   END_RUNG wire#w2
   RUNG wire#w1
      I_Contact( #MAnt_E2_DesCarga_Act )
   END_RUNG wire#w3
   // the same network as SCL:
   #PTF_MAnt_E2_Mx := (#Mx_ET20 OR (#Mx_ET21 AND NOT #STAT_FTF_MAnt_E2_Mx) OR ((#Mx_ET60 OR #Mx_ET61) AND #Simul_Mx_E2S4)) AND (#EnMovimiento_TRx OR NOT #MAnt_E2_DesCarga_Act) AND #EstadoZona.Marcha_CBx AND NOT #EstadoVI.Error_Mx AND NOT #Error_Tx;
END_REGION

REGION Network 70: VARIABLES AUXILIARES - Aviso de Salida - Salida por S3
   // Pablo: En este caso, creemos que los topes no necesariamente deben estar abajo, de hecho si estan abajo, nos hacen daño, ya que nos mueven las bandejas. 
   // Es verdad que el tope en posicion baja, desplaza la bandeja. 20230810
   RUNG wire#powerrail
      Contact( #Mx_ET250 )
      I_Contact( #Complete_S3 )
      Contact( #Selec_Salida_S3 )
      I_Contact( #EstadoZona.ParoBlando_CBx )
      wire#w1
      Contact( #TP1_Abajo )
      Contact( #TP2_Abajo )
      wire#w2
      Contact( #TRx_Abajo )
      Contact( #EstadoZona.Marcha_CBx )
      I_Contact( #EstadoVI.Error_Mx )
      I_Contact( #Error_Tx )
      Coil( #MA_PickUpOK_S3 )
   END_RUNG
   RUNG wire#powerrail
      Contact( #Mx_ET50 )
   END_RUNG wire#w1
   RUNG wire#powerrail
      Contact( #Mx_ET51 )
      Contact( #EstadoVI.Descarga_Act )
   END_RUNG wire#w1
   RUNG wire#w1
      Contact( "ON" )
   END_RUNG wire#w2
   // the same network as SCL:
   #MA_PickUpOK_S3 := ((#Mx_ET250 AND NOT #Complete_S3 AND #Selec_Salida_S3 AND NOT #EstadoZona.ParoBlando_CBx) OR #Mx_ET50 OR (#Mx_ET51 AND #EstadoVI.Descarga_Act)) AND ((#TP1_Abajo AND #TP2_Abajo) OR "ON") AND #TRx_Abajo AND #EstadoZona.Marcha_CBx AND NOT #EstadoVI.Error_Mx AND NOT #Error_Tx;
END_REGION

REGION Network 71: VARIABLES AUXILIARES - Aviso de Salida - Salida por S4
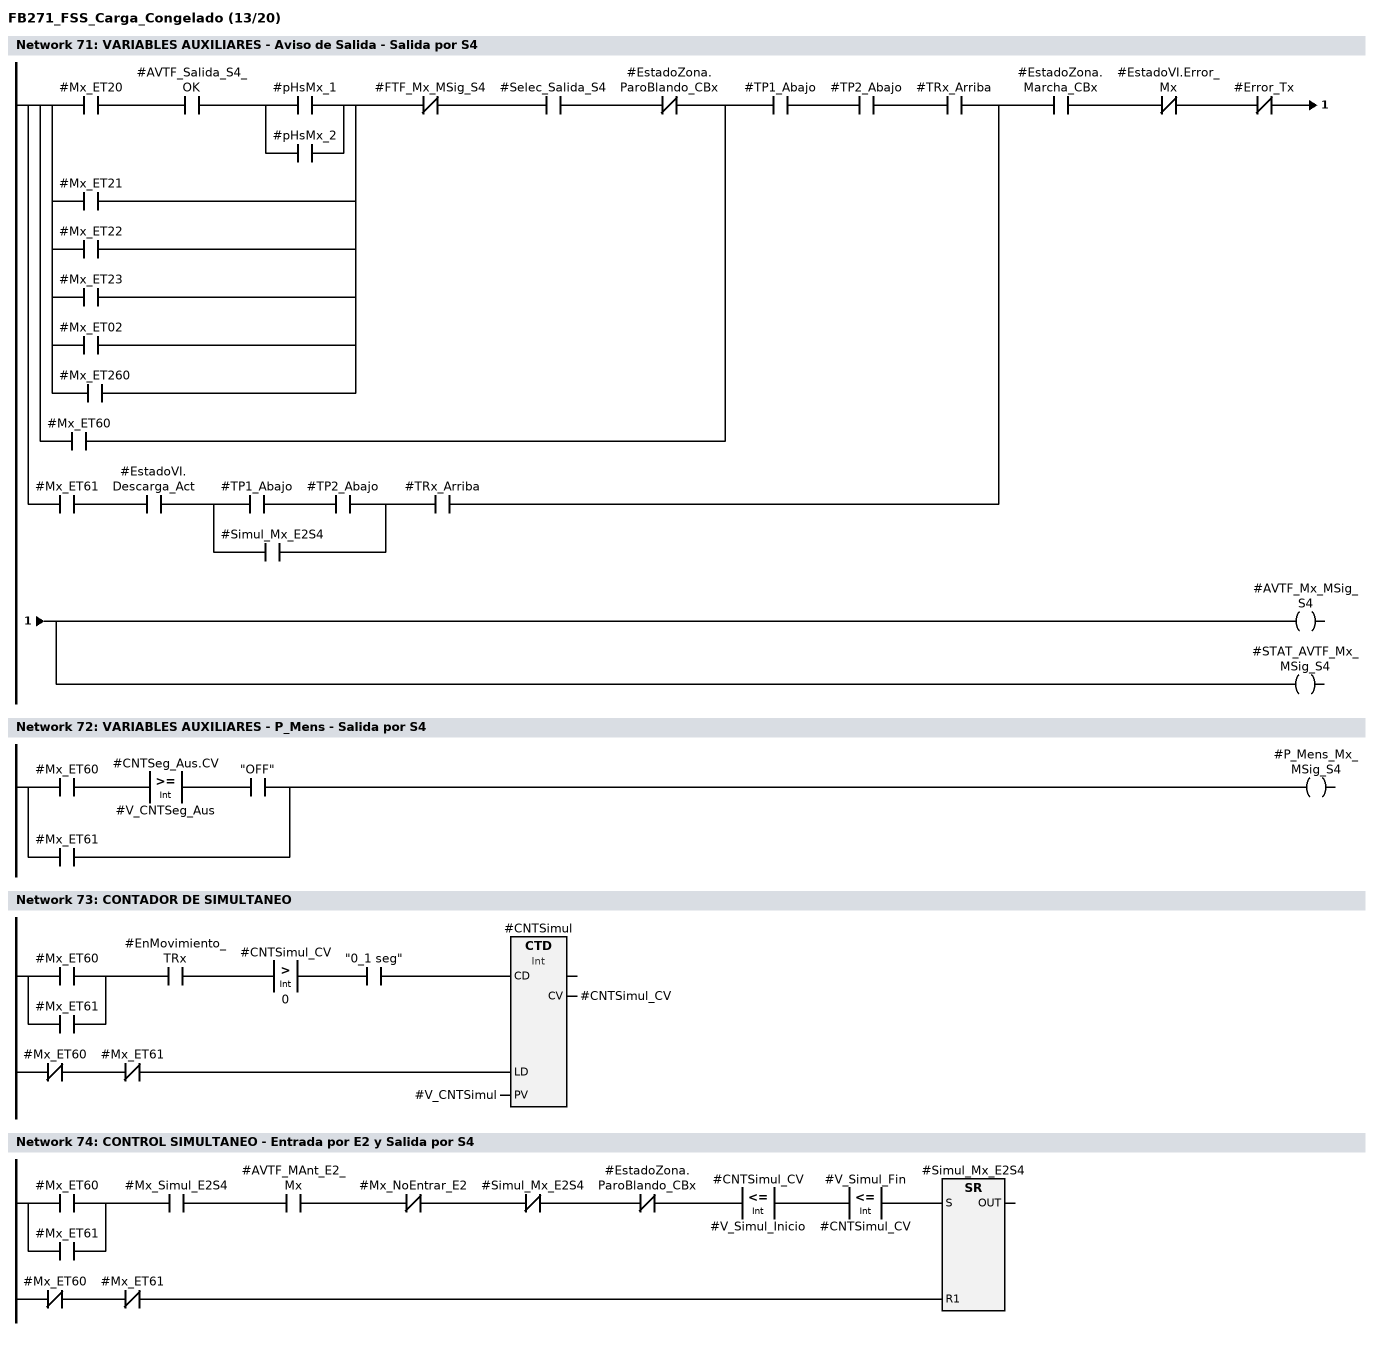
   RUNG wire#powerrail
      Contact( #Mx_ET20 )
      Contact( #AVTF_Salida_S4_OK )
      wire#w1
      Contact( #pHsMx_1 )
      wire#w2
      I_Contact( #FTF_Mx_MSig_S4 )
      Contact( #Selec_Salida_S4 )
      I_Contact( #EstadoZona.ParoBlando_CBx )
      wire#w3
      Contact( #TP1_Abajo )
      Contact( #TP2_Abajo )
      Contact( #TRx_Arriba )
      wire#w4
      Contact( #EstadoZona.Marcha_CBx )
      I_Contact( #EstadoVI.Error_Mx )
      I_Contact( #Error_Tx )
      wire#w7
      Coil( #AVTF_Mx_MSig_S4 )
   END_RUNG
   RUNG wire#w1
      Contact( #pHsMx_2 )
   END_RUNG wire#w2
   RUNG wire#powerrail
      Contact( #Mx_ET21 )
   END_RUNG wire#w2
   RUNG wire#powerrail
      Contact( #Mx_ET22 )
   END_RUNG wire#w2
   RUNG wire#powerrail
      Contact( #Mx_ET23 )
   END_RUNG wire#w2
   RUNG wire#powerrail
      Contact( #Mx_ET02 )
   END_RUNG wire#w2
   RUNG wire#powerrail
      Contact( #Mx_ET260 )
   END_RUNG wire#w2
   RUNG wire#powerrail
      Contact( #Mx_ET60 )
   END_RUNG wire#w3
   RUNG wire#powerrail
      Contact( #Mx_ET61 )
      Contact( #EstadoVI.Descarga_Act )
      wire#w5
      Contact( #TP1_Abajo )
      Contact( #TP2_Abajo )
      wire#w6
      Contact( #TRx_Arriba )
   END_RUNG wire#w4
   RUNG wire#w5
      Contact( #Simul_Mx_E2S4 )
   END_RUNG wire#w6
   RUNG wire#w7
      Coil( #STAT_AVTF_Mx_MSig_S4 )
   END_RUNG
   // the same network as SCL:
   #AVTF_Mx_MSig_S4 := ((((((#Mx_ET20 AND #AVTF_Salida_S4_OK AND (#pHsMx_1 OR #pHsMx_2)) OR #Mx_ET21 OR #Mx_ET22 OR #Mx_ET23 OR #Mx_ET02 OR #Mx_ET260) AND NOT #FTF_Mx_MSig_S4 AND #Selec_Salida_S4 AND NOT #EstadoZona.ParoBlando_CBx) OR #Mx_ET60) AND #TP1_Abajo AND #TP2_Abajo AND #TRx_Arriba) OR (#Mx_ET61 AND #EstadoVI.Descarga_Act AND ((#TP1_Abajo AND #TP2_Abajo) OR #Simul_Mx_E2S4) AND #TRx_Arriba)) AND #EstadoZona.Marcha_CBx AND NOT #EstadoVI.Error_Mx AND NOT #Error_Tx;
   #STAT_AVTF_Mx_MSig_S4 := #AVTF_Mx_MSig_S4;
END_REGION

REGION Network 72: VARIABLES AUXILIARES - P_Mens - Salida por S4
   RUNG wire#powerrail
      Contact( #Mx_ET60 )
      { S7_Templates := "SrcType := Int" } GE_Contact(in1 := #CNTSeg_Aus.CV, in2 := #V_CNTSeg_Aus)
      Contact( "OFF" )
      wire#w1
      Coil( #P_Mens_Mx_MSig_S4 )
   END_RUNG
   RUNG wire#powerrail
      Contact( #Mx_ET61 )
   END_RUNG wire#w1
   // the same network as SCL:
   #P_Mens_Mx_MSig_S4 := (#Mx_ET60 AND (#CNTSeg_Aus.CV >= #V_CNTSeg_Aus) AND "OFF") OR #Mx_ET61;
END_REGION

REGION Network 73: CONTADOR DE SIMULTANEO
   RUNG wire#powerrail
      Contact( #Mx_ET60 )
      wire#w1
      Contact( #EnMovimiento_TRx )
      { S7_Templates := "SrcType := Int" } GT_Contact(in1 := #CNTSimul_CV, in2 := 0)
      Contact( "0_1 seg" )
      { S7_Templates := "value_type := Int" } #CNTSimul.CTD(ld := wire#w2, pv := #V_CNTSimul, cv => #CNTSimul_CV)
   END_RUNG
   RUNG wire#powerrail
      Contact( #Mx_ET61 )
   END_RUNG wire#w1
   RUNG wire#powerrail
      I_Contact( #Mx_ET60 )
      I_Contact( #Mx_ET61 )
   END_RUNG wire#w2
   // the same network as SCL:
   #CNTSimul(CD := (#Mx_ET60 OR #Mx_ET61) AND #EnMovimiento_TRx AND (#CNTSimul_CV > 0) AND "0_1 seg",   // CTD
             LD := NOT #Mx_ET60 AND NOT #Mx_ET61,
             PV := #V_CNTSimul,
             CV => #CNTSimul_CV);
END_REGION

REGION Network 74: CONTROL SIMULTANEO - Entrada por E2 y Salida por S4
   RUNG wire#powerrail
      Contact( #Mx_ET60 )
      wire#w1
      Contact( #Mx_Simul_E2S4 )
      Contact( #AVTF_MAnt_E2_Mx )
      I_Contact( #Mx_NoEntrar_E2 )
      I_Contact( #Simul_Mx_E2S4 )
      I_Contact( #EstadoZona.ParoBlando_CBx )
      { S7_Templates := "SrcType := Int" } LE_Contact(in1 := #CNTSimul_CV, in2 := #V_Simul_Inicio)
      { S7_Templates := "SrcType := Int" } LE_Contact(in1 := #V_Simul_Fin, in2 := #CNTSimul_CV)
      S_SR(operand := #Simul_Mx_E2S4, r1 := wire#w2)
   END_RUNG
   RUNG wire#powerrail
      Contact( #Mx_ET61 )
   END_RUNG wire#w1
   RUNG wire#powerrail
      I_Contact( #Mx_ET60 )
      I_Contact( #Mx_ET61 )
   END_RUNG wire#w2
   // the same network as SCL:
   IF (#Mx_ET60 OR #Mx_ET61) AND #Mx_Simul_E2S4 AND #AVTF_MAnt_E2_Mx AND NOT #Mx_NoEntrar_E2 AND NOT #Simul_Mx_E2S4 AND NOT #EstadoZona.ParoBlando_CBx AND (#CNTSimul_CV <= #V_Simul_Inicio) AND (#V_Simul_Fin <= #CNTSimul_CV) THEN
       #Simul_Mx_E2S4 := TRUE;   // SR flip-flop
   END_IF;
   IF NOT #Mx_ET60 AND NOT #Mx_ET61 THEN #Simul_Mx_E2S4 := FALSE; END_IF;
END_REGION

REGION Network 75: MENSAJES - PRESENCIA
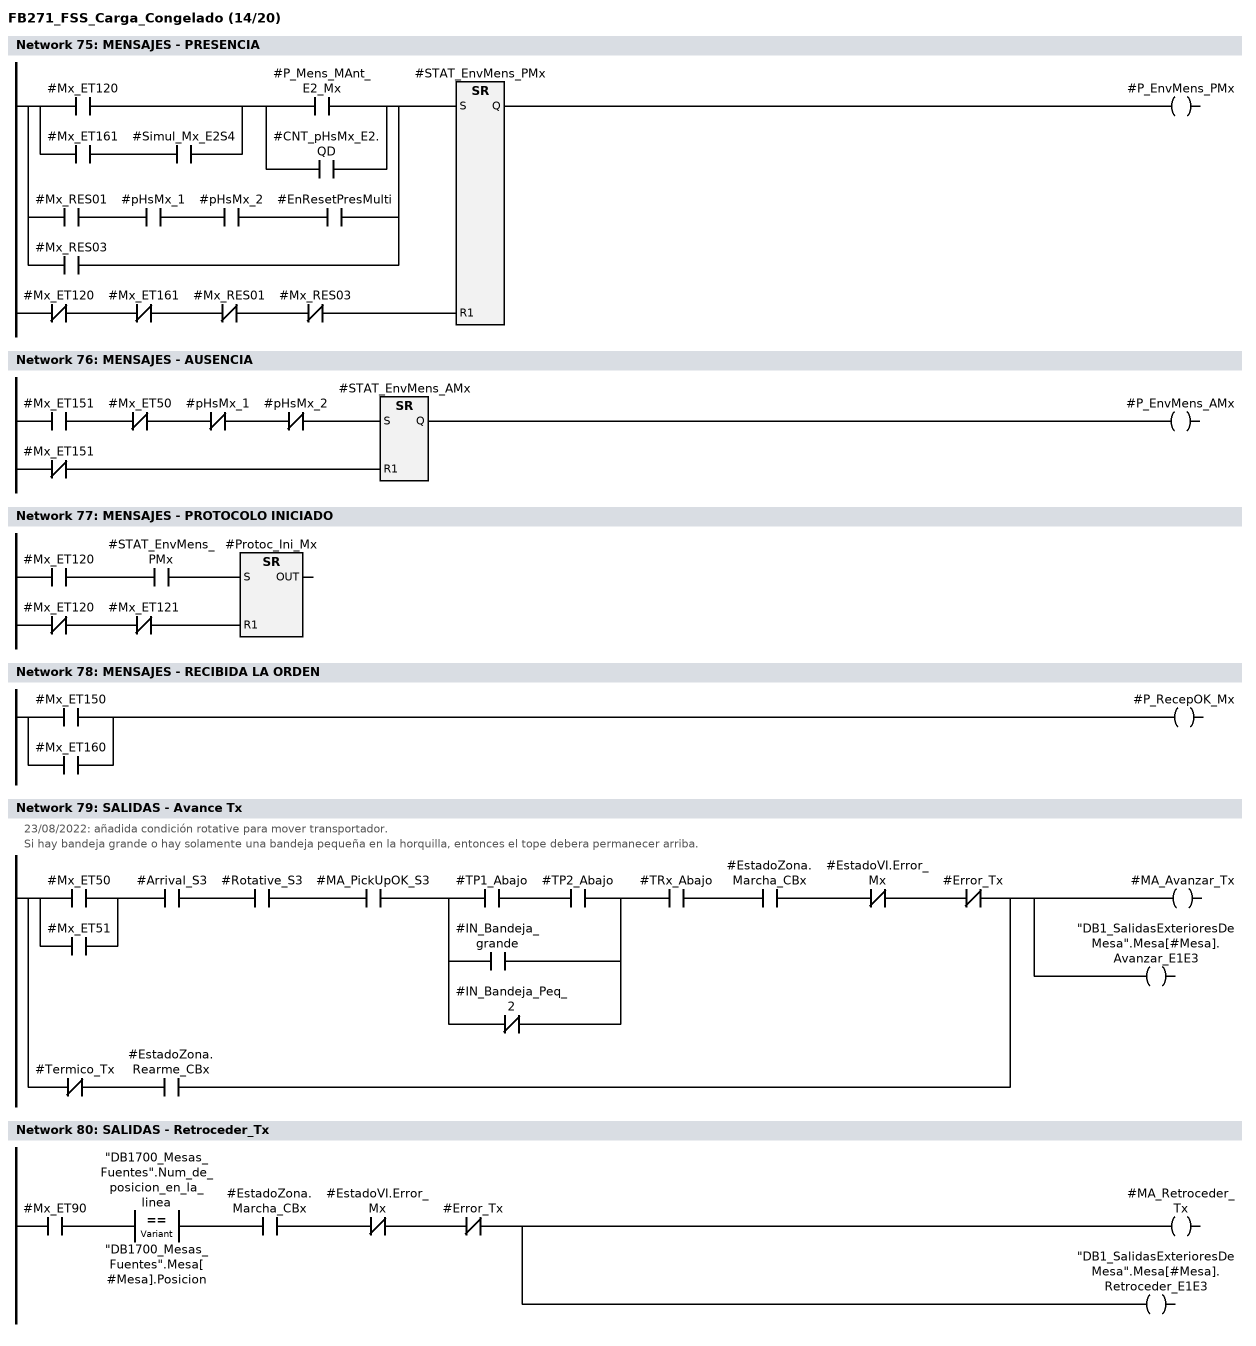
   RUNG wire#powerrail
      Contact( #Mx_ET120 )
      wire#w1
      Contact( #P_Mens_MAnt_E2_Mx )
      wire#w2
      S_SR(operand := #STAT_EnvMens_PMx, r1 := wire#w3)
      Coil( #P_EnvMens_PMx )
   END_RUNG
   RUNG wire#powerrail
      Contact( #Mx_ET161 )
      Contact( #Simul_Mx_E2S4 )
   END_RUNG wire#w1
   RUNG wire#w1
      Contact( #CNT_pHsMx_E2.QD )
   END_RUNG wire#w2
   RUNG wire#powerrail
      Contact( #Mx_RES01 )
      Contact( #pHsMx_1 )
      Contact( #pHsMx_2 )
      Contact( #EnResetPresMulti )
   END_RUNG wire#w2
   RUNG wire#powerrail
      Contact( #Mx_RES03 )
   END_RUNG wire#w2
   RUNG wire#powerrail
      I_Contact( #Mx_ET120 )
      I_Contact( #Mx_ET161 )
      I_Contact( #Mx_RES01 )
      I_Contact( #Mx_RES03 )
   END_RUNG wire#w3
   // the same network as SCL:
   IF ((#Mx_ET120 OR (#Mx_ET161 AND #Simul_Mx_E2S4)) AND (#P_Mens_MAnt_E2_Mx OR #CNT_pHsMx_E2.QD)) OR (#Mx_RES01 AND #pHsMx_1 AND #pHsMx_2 AND #EnResetPresMulti) OR #Mx_RES03 THEN
       #STAT_EnvMens_PMx := TRUE;   // SR flip-flop
   END_IF;
   IF NOT #Mx_ET120 AND NOT #Mx_ET161 AND NOT #Mx_RES01 AND NOT #Mx_RES03 THEN
       #STAT_EnvMens_PMx := FALSE;
   END_IF;
   #P_EnvMens_PMx := #STAT_EnvMens_PMx;
END_REGION

REGION Network 76: MENSAJES - AUSENCIA
   RUNG wire#powerrail
      Contact( #Mx_ET151 )
      I_Contact( #Mx_ET50 )
      I_Contact( #pHsMx_1 )
      I_Contact( #pHsMx_2 )
      S_SR(operand := #STAT_EnvMens_AMx, r1 := wire#w1)
      Coil( #P_EnvMens_AMx )
   END_RUNG
   RUNG wire#powerrail
      I_Contact( #Mx_ET151 )
   END_RUNG wire#w1
   // the same network as SCL:
   IF #Mx_ET151 AND NOT #Mx_ET50 AND NOT #pHsMx_1 AND NOT #pHsMx_2 THEN
       #STAT_EnvMens_AMx := TRUE;   // SR flip-flop
   END_IF;
   IF NOT #Mx_ET151 THEN #STAT_EnvMens_AMx := FALSE; END_IF;
   #P_EnvMens_AMx := #STAT_EnvMens_AMx;
END_REGION

REGION Network 77: MENSAJES - PROTOCOLO INICIADO
   RUNG wire#powerrail
      Contact( #Mx_ET120 )
      Contact( #STAT_EnvMens_PMx )
      S_SR(operand := #Protoc_Ini_Mx, r1 := wire#w1)
   END_RUNG
   RUNG wire#powerrail
      I_Contact( #Mx_ET120 )
      I_Contact( #Mx_ET121 )
   END_RUNG wire#w1
   // the same network as SCL:
   IF #Mx_ET120 AND #STAT_EnvMens_PMx THEN
       #Protoc_Ini_Mx := TRUE;   // SR flip-flop
   END_IF;
   IF NOT #Mx_ET120 AND NOT #Mx_ET121 THEN #Protoc_Ini_Mx := FALSE; END_IF;
END_REGION

REGION Network 78: MENSAJES - RECIBIDA LA ORDEN
   RUNG wire#powerrail
      Contact( #Mx_ET150 )
      wire#w1
      Coil( #P_RecepOK_Mx )
   END_RUNG
   RUNG wire#powerrail
      Contact( #Mx_ET160 )
   END_RUNG wire#w1
   // the same network as SCL:
   #P_RecepOK_Mx := #Mx_ET150 OR #Mx_ET160;
END_REGION

REGION Network 79: SALIDAS - Avance Tx
   // 23/08/2022: añadida condición rotative para mover transportador. 
   // Si hay bandeja grande o hay solamente una bandeja pequeña en la horquilla, entonces el tope debera permanecer arriba.
   RUNG wire#powerrail
      Contact( #Mx_ET50 )
      wire#w1
      Contact( #Arrival_S3 )
      Contact( #Rotative_S3 )
      Contact( #MA_PickUpOK_S3 )
      wire#w2
      Contact( #TP1_Abajo )
      Contact( #TP2_Abajo )
      wire#w3
      Contact( #TRx_Abajo )
      Contact( #EstadoZona.Marcha_CBx )
      I_Contact( #EstadoVI.Error_Mx )
      I_Contact( #Error_Tx )
      wire#w4
      Coil( #MA_Avanzar_Tx )
   END_RUNG
   RUNG wire#powerrail
      Contact( #Mx_ET51 )
   END_RUNG wire#w1
   RUNG wire#w2
      Contact( #IN_Bandeja_grande )
   END_RUNG wire#w3
   RUNG wire#w2
      I_Contact( #IN_Bandeja_Peq_2 )
   END_RUNG wire#w3
   RUNG wire#powerrail
      I_Contact( #Termico_Tx )
      Contact( #EstadoZona.Rearme_CBx )
   END_RUNG wire#w4
   RUNG wire#w4
      Coil( "DB1_SalidasExterioresDeMesa".Mesa[#Mesa].Avanzar_E1E3 )
   END_RUNG
   // the same network as SCL:
   #MA_Avanzar_Tx := ((#Mx_ET50 OR #Mx_ET51) AND #Arrival_S3 AND #Rotative_S3 AND #MA_PickUpOK_S3 AND ((#TP1_Abajo AND #TP2_Abajo) OR #IN_Bandeja_grande OR NOT #IN_Bandeja_Peq_2) AND #TRx_Abajo AND #EstadoZona.Marcha_CBx AND NOT #EstadoVI.Error_Mx AND NOT #Error_Tx) OR (NOT #Termico_Tx AND #EstadoZona.Rearme_CBx);
   "DB1_SalidasExterioresDeMesa".Mesa[#Mesa].Avanzar_E1E3 := #MA_Avanzar_Tx;
END_REGION

REGION Network 80: SALIDAS - Retroceder_Tx
   RUNG wire#powerrail
      Contact( #Mx_ET90 )
      { S7_Templates := "SrcType := Variant" } EQ_Contact(in1 := "DB1700_Mesas_Fuentes".Num_de_posicion_en_la_linea, in2 := "DB1700_Mesas_Fuentes".Mesa[#Mesa].Posicion)
      Contact( #EstadoZona.Marcha_CBx )
      I_Contact( #EstadoVI.Error_Mx )
      I_Contact( #Error_Tx )
      wire#w1
      Coil( #MA_Retroceder_Tx )
   END_RUNG
   RUNG wire#w1
      Coil( "DB1_SalidasExterioresDeMesa".Mesa[#Mesa].Retroceder_E1E3 )
   END_RUNG
   // the same network as SCL:
   #MA_Retroceder_Tx := #Mx_ET90 AND ("DB1700_Mesas_Fuentes".Num_de_posicion_en_la_linea = "DB1700_Mesas_Fuentes".Mesa[#Mesa].Posicion) AND #EstadoZona.Marcha_CBx AND NOT #EstadoVI.Error_Mx AND NOT #Error_Tx;
   "DB1_SalidasExterioresDeMesa".Mesa[#Mesa].Retroceder_E1E3 := #MA_Retroceder_Tx;
END_REGION

REGION Network 81: SALIDAS - Velocidad Rapida Tx
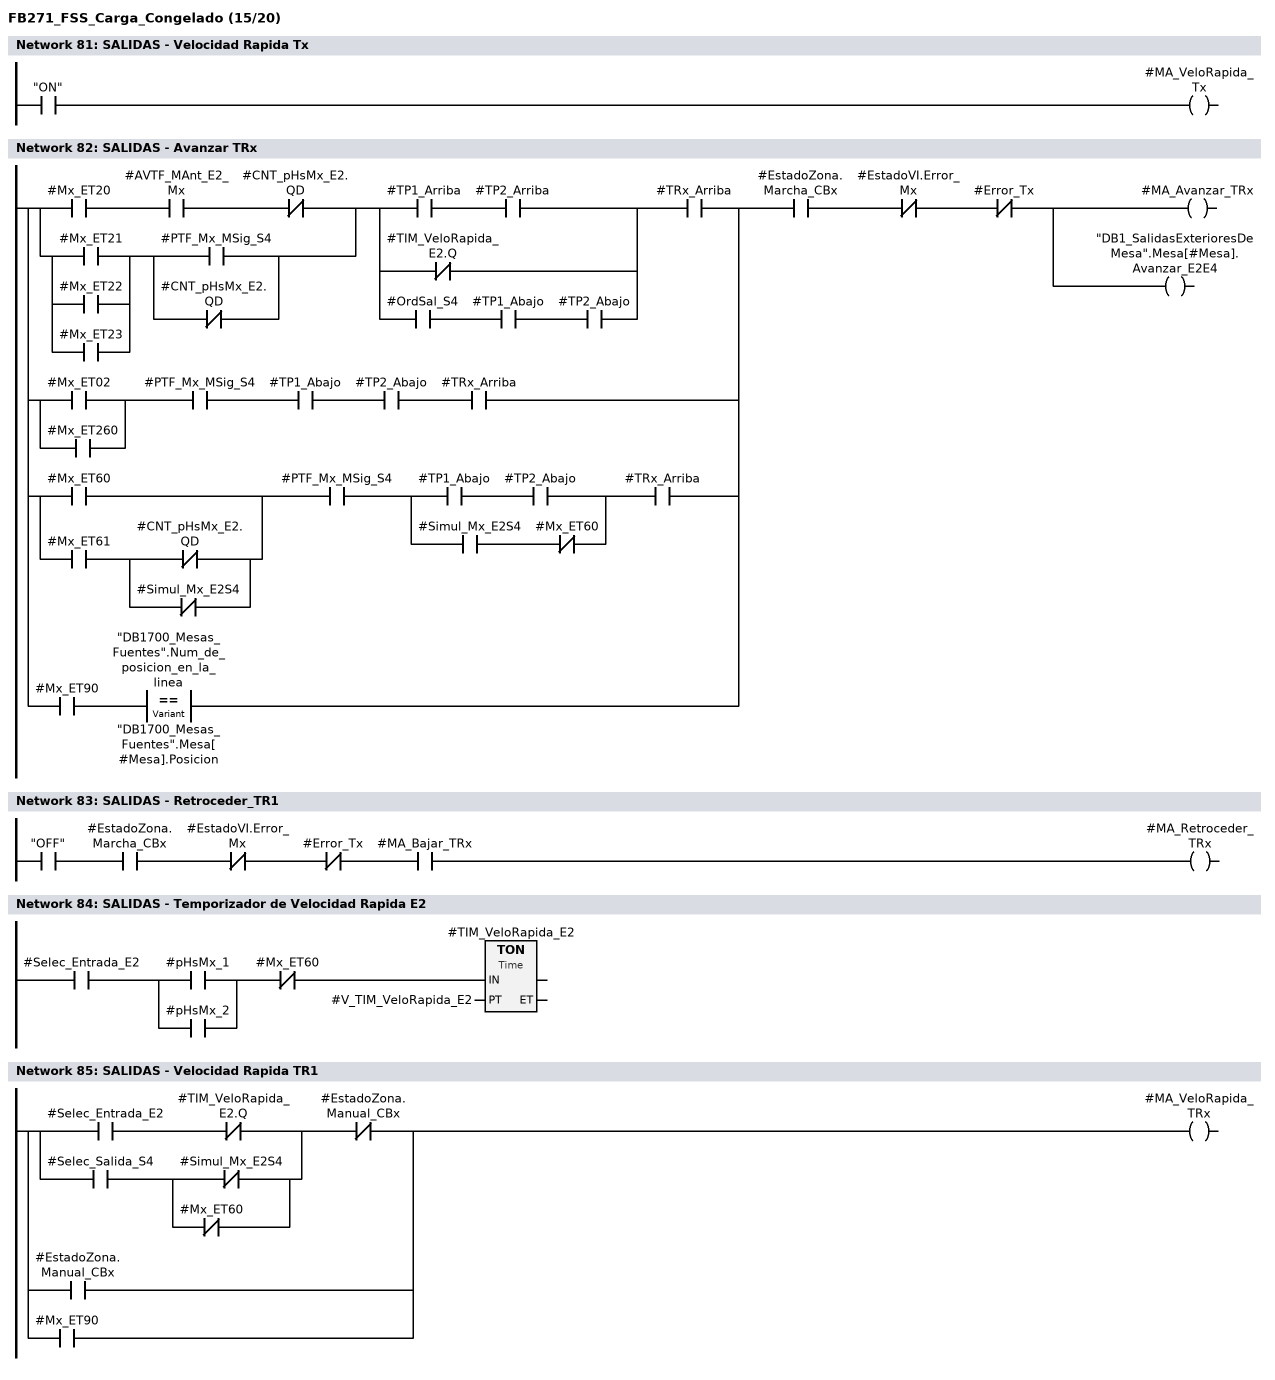
   RUNG wire#powerrail
      Contact( "ON" )
      Coil( #MA_VeloRapida_Tx )
   END_RUNG
   // the same network as SCL:
   #MA_VeloRapida_Tx := "ON";
END_REGION

REGION Network 82: SALIDAS - Avanzar TRx
   RUNG wire#powerrail
      Contact( #Mx_ET20 )
      Contact( #AVTF_MAnt_E2_Mx )
      I_Contact( #CNT_pHsMx_E2.QD )
      wire#w1
      Contact( #TP1_Arriba )
      Contact( #TP2_Arriba )
      wire#w3
      Contact( #TRx_Arriba )
      wire#w4
      Contact( #EstadoZona.Marcha_CBx )
      I_Contact( #EstadoVI.Error_Mx )
      I_Contact( #Error_Tx )
      wire#w10
      Coil( #MA_Avanzar_TRx )
   END_RUNG
   RUNG wire#powerrail
      Contact( #Mx_ET21 )
      wire#w2
      Contact( #PTF_Mx_MSig_S4 )
   END_RUNG wire#w1
   RUNG wire#powerrail
      Contact( #Mx_ET22 )
   END_RUNG wire#w2
   RUNG wire#powerrail
      Contact( #Mx_ET23 )
   END_RUNG wire#w2
   RUNG wire#w2
      I_Contact( #CNT_pHsMx_E2.QD )
   END_RUNG wire#w1
   RUNG wire#w1
      I_Contact( #TIM_VeloRapida_E2.Q )
   END_RUNG wire#w3
   RUNG wire#w1
      Contact( #OrdSal_S4 )
      Contact( #TP1_Abajo )
      Contact( #TP2_Abajo )
   END_RUNG wire#w3
   RUNG wire#powerrail
      Contact( #Mx_ET02 )
      wire#w5
      Contact( #PTF_Mx_MSig_S4 )
      Contact( #TP1_Abajo )
      Contact( #TP2_Abajo )
      Contact( #TRx_Arriba )
   END_RUNG wire#w4
   RUNG wire#powerrail
      Contact( #Mx_ET260 )
   END_RUNG wire#w5
   RUNG wire#powerrail
      Contact( #Mx_ET60 )
      wire#w6
      Contact( #PTF_Mx_MSig_S4 )
      wire#w8
      Contact( #TP1_Abajo )
      Contact( #TP2_Abajo )
      wire#w9
      Contact( #TRx_Arriba )
   END_RUNG wire#w4
   RUNG wire#powerrail
      Contact( #Mx_ET61 )
      wire#w7
      I_Contact( #CNT_pHsMx_E2.QD )
   END_RUNG wire#w6
   RUNG wire#w7
      I_Contact( #Simul_Mx_E2S4 )
   END_RUNG wire#w6
   RUNG wire#w8
      Contact( #Simul_Mx_E2S4 )
      I_Contact( #Mx_ET60 )
   END_RUNG wire#w9
   RUNG wire#powerrail
      Contact( #Mx_ET90 )
      { S7_Templates := "SrcType := Variant" } EQ_Contact(in1 := "DB1700_Mesas_Fuentes".Num_de_posicion_en_la_linea, in2 := "DB1700_Mesas_Fuentes".Mesa[#Mesa].Posicion)
   END_RUNG wire#w4
   RUNG wire#w10
      Coil( "DB1_SalidasExterioresDeMesa".Mesa[#Mesa].Avanzar_E2E4 )
   END_RUNG
   // the same network as SCL:
   #MA_Avanzar_TRx := ((((#Mx_ET20 AND #AVTF_MAnt_E2_Mx AND NOT #CNT_pHsMx_E2.QD) OR ((#Mx_ET21 OR #Mx_ET22 OR #Mx_ET23) AND (#PTF_Mx_MSig_S4 OR NOT #CNT_pHsMx_E2.QD))) AND ((#TP1_Arriba AND #TP2_Arriba) OR NOT #TIM_VeloRapida_E2.Q OR (#OrdSal_S4 AND #TP1_Abajo AND #TP2_Abajo)) AND #TRx_Arriba) OR ((#Mx_ET02 OR #Mx_ET260) AND #PTF_Mx_MSig_S4 AND #TP1_Abajo AND #TP2_Abajo AND #TRx_Arriba) OR ((#Mx_ET60 OR (#Mx_ET61 AND (NOT #CNT_pHsMx_E2.QD OR NOT #Simul_Mx_E2S4))) AND #PTF_Mx_MSig_S4 AND ((#TP1_Abajo AND #TP2_Abajo) OR (#Simul_Mx_E2S4 AND NOT #Mx_ET60)) AND #TRx_Arriba) OR (#Mx_ET90 AND ("DB1700_Mesas_Fuentes".Num_de_posicion_en_la_linea = "DB1700_Mesas_Fuentes".Mesa[#Mesa].Posicion))) AND #EstadoZona.Marcha_CBx AND NOT #EstadoVI.Error_Mx AND NOT #Error_Tx;
   "DB1_SalidasExterioresDeMesa".Mesa[#Mesa].Avanzar_E2E4 := #MA_Avanzar_TRx;
END_REGION

REGION Network 83: SALIDAS - Retroceder_TR1
   RUNG wire#powerrail
      Contact( "OFF" )
      Contact( #EstadoZona.Marcha_CBx )
      I_Contact( #EstadoVI.Error_Mx )
      I_Contact( #Error_Tx )
      Contact( #MA_Bajar_TRx )
      Coil( #MA_Retroceder_TRx )
   END_RUNG
   // the same network as SCL:
   #MA_Retroceder_TRx := "OFF" AND #EstadoZona.Marcha_CBx AND NOT #EstadoVI.Error_Mx AND NOT #Error_Tx AND #MA_Bajar_TRx;
END_REGION

REGION Network 84: SALIDAS - Temporizador de Velocidad Rapida E2
   RUNG wire#powerrail
      Contact( #Selec_Entrada_E2 )
      wire#w1
      Contact( #pHsMx_1 )
      wire#w2
      I_Contact( #Mx_ET60 )
      { S7_Templates := "time_type := Time" } #TIM_VeloRapida_E2.TON(pt := #V_TIM_VeloRapida_E2, et =>)
   END_RUNG
   RUNG wire#w1
      Contact( #pHsMx_2 )
   END_RUNG wire#w2
   // the same network as SCL:
   #TIM_VeloRapida_E2(IN := #Selec_Entrada_E2 AND (#pHsMx_1 OR #pHsMx_2) AND NOT #Mx_ET60,   // TON
                      PT := #V_TIM_VeloRapida_E2);
END_REGION

REGION Network 85: SALIDAS - Velocidad Rapida TR1
   RUNG wire#powerrail
      Contact( #Selec_Entrada_E2 )
      I_Contact( #TIM_VeloRapida_E2.Q )
      wire#w1
      I_Contact( #EstadoZona.Manual_CBx )
      wire#w3
      Coil( #MA_VeloRapida_TRx )
   END_RUNG
   RUNG wire#powerrail
      Contact( #Selec_Salida_S4 )
      wire#w2
      I_Contact( #Simul_Mx_E2S4 )
   END_RUNG wire#w1
   RUNG wire#w2
      I_Contact( #Mx_ET60 )
   END_RUNG wire#w1
   RUNG wire#powerrail
      Contact( #EstadoZona.Manual_CBx )
   END_RUNG wire#w3
   RUNG wire#powerrail
      Contact( #Mx_ET90 )
   END_RUNG wire#w3
   // the same network as SCL:
   #MA_VeloRapida_TRx := (((#Selec_Entrada_E2 AND NOT #TIM_VeloRapida_E2.Q) OR (#Selec_Salida_S4 AND (NOT #Simul_Mx_E2S4 OR NOT #Mx_ET60))) AND NOT #EstadoZona.Manual_CBx) OR #EstadoZona.Manual_CBx OR #Mx_ET90;
END_REGION

REGION Network 86: SALIDAS - Subir TP1
   // No subir Tope al ver sensores
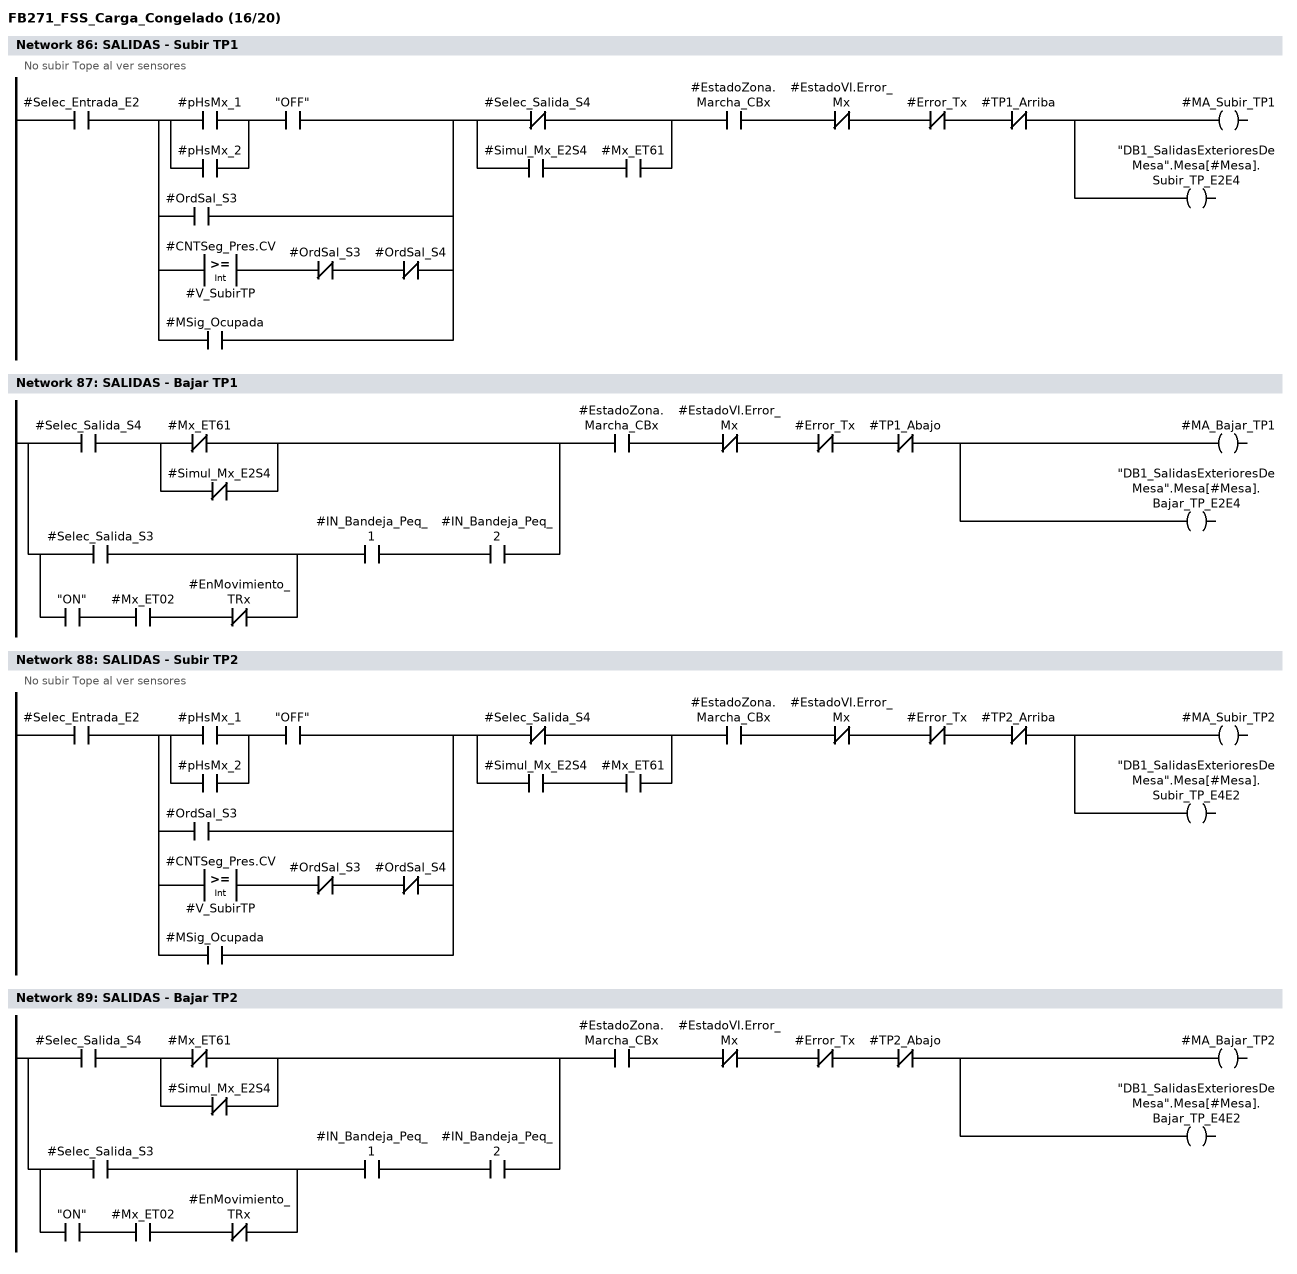
   RUNG wire#powerrail
      Contact( #Selec_Entrada_E2 )
      wire#w1
      Contact( #pHsMx_1 )
      wire#w2
      Contact( "OFF" )
      wire#w3
      I_Contact( #Selec_Salida_S4 )
      wire#w4
      Contact( #EstadoZona.Marcha_CBx )
      I_Contact( #EstadoVI.Error_Mx )
      I_Contact( #Error_Tx )
      I_Contact( #TP1_Arriba )
      wire#w5
      Coil( #MA_Subir_TP1 )
   END_RUNG
   RUNG wire#w1
      Contact( #pHsMx_2 )
   END_RUNG wire#w2
   RUNG wire#w1
      Contact( #OrdSal_S3 )
   END_RUNG wire#w3
   RUNG wire#w1
      { S7_Templates := "SrcType := Int" } GE_Contact(in1 := #CNTSeg_Pres.CV, in2 := #V_SubirTP)
      I_Contact( #OrdSal_S3 )
      I_Contact( #OrdSal_S4 )
   END_RUNG wire#w3
   RUNG wire#w1
      Contact( #MSig_Ocupada )
   END_RUNG wire#w3
   RUNG wire#w3
      Contact( #Simul_Mx_E2S4 )
      Contact( #Mx_ET61 )
   END_RUNG wire#w4
   RUNG wire#w5
      Coil( "DB1_SalidasExterioresDeMesa".Mesa[#Mesa].Subir_TP_E2E4 )
   END_RUNG
   // the same network as SCL:
   #MA_Subir_TP1 := #Selec_Entrada_E2 AND (((#pHsMx_1 OR #pHsMx_2) AND "OFF") OR #OrdSal_S3 OR ((#CNTSeg_Pres.CV >= #V_SubirTP) AND NOT #OrdSal_S3 AND NOT #OrdSal_S4) OR #MSig_Ocupada) AND (NOT #Selec_Salida_S4 OR (#Simul_Mx_E2S4 AND #Mx_ET61)) AND #EstadoZona.Marcha_CBx AND NOT #EstadoVI.Error_Mx AND NOT #Error_Tx AND NOT #TP1_Arriba;
   "DB1_SalidasExterioresDeMesa".Mesa[#Mesa].Subir_TP_E2E4 := #MA_Subir_TP1;
END_REGION

REGION Network 87: SALIDAS - Bajar TP1
   RUNG wire#powerrail
      Contact( #Selec_Salida_S4 )
      wire#w1
      I_Contact( #Mx_ET61 )
      wire#w2
      Contact( #EstadoZona.Marcha_CBx )
      I_Contact( #EstadoVI.Error_Mx )
      I_Contact( #Error_Tx )
      I_Contact( #TP1_Abajo )
      wire#w4
      Coil( #MA_Bajar_TP1 )
   END_RUNG
   RUNG wire#w1
      I_Contact( #Simul_Mx_E2S4 )
   END_RUNG wire#w2
   RUNG wire#powerrail
      Contact( #Selec_Salida_S3 )
      wire#w3
      Contact( #IN_Bandeja_Peq_1 )
      Contact( #IN_Bandeja_Peq_2 )
   END_RUNG wire#w2
   RUNG wire#powerrail
      Contact( "ON" )
      Contact( #Mx_ET02 )
      I_Contact( #EnMovimiento_TRx )
   END_RUNG wire#w3
   RUNG wire#w4
      Coil( "DB1_SalidasExterioresDeMesa".Mesa[#Mesa].Bajar_TP_E2E4 )
   END_RUNG
   // the same network as SCL:
   #MA_Bajar_TP1 := ((#Selec_Salida_S4 AND (NOT #Mx_ET61 OR NOT #Simul_Mx_E2S4)) OR ((#Selec_Salida_S3 OR ("ON" AND #Mx_ET02 AND NOT #EnMovimiento_TRx)) AND #IN_Bandeja_Peq_1 AND #IN_Bandeja_Peq_2)) AND #EstadoZona.Marcha_CBx AND NOT #EstadoVI.Error_Mx AND NOT #Error_Tx AND NOT #TP1_Abajo;
   "DB1_SalidasExterioresDeMesa".Mesa[#Mesa].Bajar_TP_E2E4 := #MA_Bajar_TP1;
END_REGION

REGION Network 88: SALIDAS - Subir TP2
   // No subir Tope al ver sensores
   RUNG wire#powerrail
      Contact( #Selec_Entrada_E2 )
      wire#w1
      Contact( #pHsMx_1 )
      wire#w2
      Contact( "OFF" )
      wire#w3
      I_Contact( #Selec_Salida_S4 )
      wire#w4
      Contact( #EstadoZona.Marcha_CBx )
      I_Contact( #EstadoVI.Error_Mx )
      I_Contact( #Error_Tx )
      I_Contact( #TP2_Arriba )
      wire#w5
      Coil( #MA_Subir_TP2 )
   END_RUNG
   RUNG wire#w1
      Contact( #pHsMx_2 )
   END_RUNG wire#w2
   RUNG wire#w1
      Contact( #OrdSal_S3 )
   END_RUNG wire#w3
   RUNG wire#w1
      { S7_Templates := "SrcType := Int" } GE_Contact(in1 := #CNTSeg_Pres.CV, in2 := #V_SubirTP)
      I_Contact( #OrdSal_S3 )
      I_Contact( #OrdSal_S4 )
   END_RUNG wire#w3
   RUNG wire#w1
      Contact( #MSig_Ocupada )
   END_RUNG wire#w3
   RUNG wire#w3
      Contact( #Simul_Mx_E2S4 )
      Contact( #Mx_ET61 )
   END_RUNG wire#w4
   RUNG wire#w5
      Coil( "DB1_SalidasExterioresDeMesa".Mesa[#Mesa].Subir_TP_E4E2 )
   END_RUNG
   // the same network as SCL:
   #MA_Subir_TP2 := #Selec_Entrada_E2 AND (((#pHsMx_1 OR #pHsMx_2) AND "OFF") OR #OrdSal_S3 OR ((#CNTSeg_Pres.CV >= #V_SubirTP) AND NOT #OrdSal_S3 AND NOT #OrdSal_S4) OR #MSig_Ocupada) AND (NOT #Selec_Salida_S4 OR (#Simul_Mx_E2S4 AND #Mx_ET61)) AND #EstadoZona.Marcha_CBx AND NOT #EstadoVI.Error_Mx AND NOT #Error_Tx AND NOT #TP2_Arriba;
   "DB1_SalidasExterioresDeMesa".Mesa[#Mesa].Subir_TP_E4E2 := #MA_Subir_TP2;
END_REGION

REGION Network 89: SALIDAS - Bajar TP2
   RUNG wire#powerrail
      Contact( #Selec_Salida_S4 )
      wire#w1
      I_Contact( #Mx_ET61 )
      wire#w2
      Contact( #EstadoZona.Marcha_CBx )
      I_Contact( #EstadoVI.Error_Mx )
      I_Contact( #Error_Tx )
      I_Contact( #TP2_Abajo )
      wire#w4
      Coil( #MA_Bajar_TP2 )
   END_RUNG
   RUNG wire#w1
      I_Contact( #Simul_Mx_E2S4 )
   END_RUNG wire#w2
   RUNG wire#powerrail
      Contact( #Selec_Salida_S3 )
      wire#w3
      Contact( #IN_Bandeja_Peq_1 )
      Contact( #IN_Bandeja_Peq_2 )
   END_RUNG wire#w2
   RUNG wire#powerrail
      Contact( "ON" )
      Contact( #Mx_ET02 )
      I_Contact( #EnMovimiento_TRx )
   END_RUNG wire#w3
   RUNG wire#w4
      Coil( "DB1_SalidasExterioresDeMesa".Mesa[#Mesa].Bajar_TP_E4E2 )
   END_RUNG
   // the same network as SCL:
   #MA_Bajar_TP2 := ((#Selec_Salida_S4 AND (NOT #Mx_ET61 OR NOT #Simul_Mx_E2S4)) OR ((#Selec_Salida_S3 OR ("ON" AND #Mx_ET02 AND NOT #EnMovimiento_TRx)) AND #IN_Bandeja_Peq_1 AND #IN_Bandeja_Peq_2)) AND #EstadoZona.Marcha_CBx AND NOT #EstadoVI.Error_Mx AND NOT #Error_Tx AND NOT #TP2_Abajo;
   "DB1_SalidasExterioresDeMesa".Mesa[#Mesa].Bajar_TP_E4E2 := #MA_Bajar_TP2;
END_REGION

REGION Network 90: SALIDAS - Subir_TR1
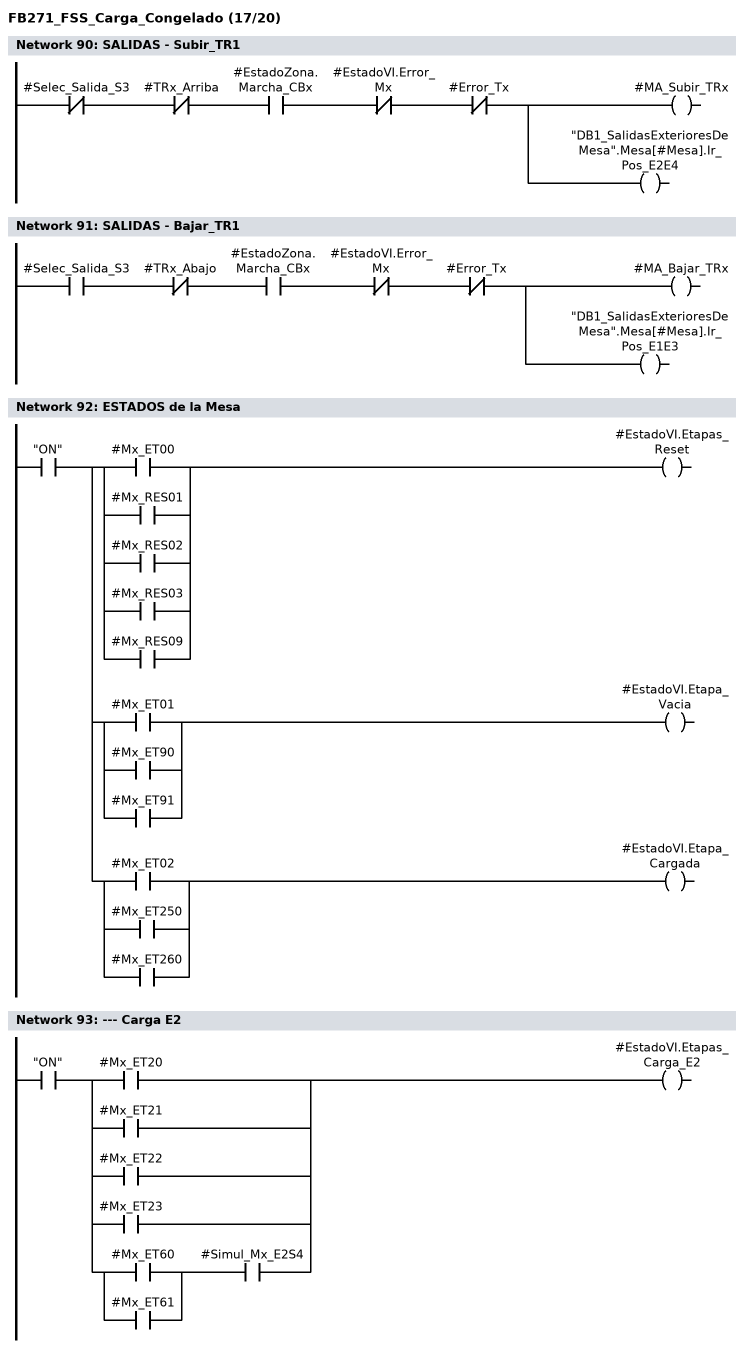
   RUNG wire#powerrail
      I_Contact( #Selec_Salida_S3 )
      I_Contact( #TRx_Arriba )
      Contact( #EstadoZona.Marcha_CBx )
      I_Contact( #EstadoVI.Error_Mx )
      I_Contact( #Error_Tx )
      wire#w1
      Coil( #MA_Subir_TRx )
   END_RUNG
   RUNG wire#w1
      Coil( "DB1_SalidasExterioresDeMesa".Mesa[#Mesa].Ir_Pos_E2E4 )
   END_RUNG
   // the same network as SCL:
   #MA_Subir_TRx := NOT #Selec_Salida_S3 AND NOT #TRx_Arriba AND #EstadoZona.Marcha_CBx AND NOT #EstadoVI.Error_Mx AND NOT #Error_Tx;
   "DB1_SalidasExterioresDeMesa".Mesa[#Mesa].Ir_Pos_E2E4 := #MA_Subir_TRx;
END_REGION

REGION Network 91: SALIDAS - Bajar_TR1
   RUNG wire#powerrail
      Contact( #Selec_Salida_S3 )
      I_Contact( #TRx_Abajo )
      Contact( #EstadoZona.Marcha_CBx )
      I_Contact( #EstadoVI.Error_Mx )
      I_Contact( #Error_Tx )
      wire#w1
      Coil( #MA_Bajar_TRx )
   END_RUNG
   RUNG wire#w1
      Coil( "DB1_SalidasExterioresDeMesa".Mesa[#Mesa].Ir_Pos_E1E3 )
   END_RUNG
   // the same network as SCL:
   #MA_Bajar_TRx := #Selec_Salida_S3 AND NOT #TRx_Abajo AND #EstadoZona.Marcha_CBx AND NOT #EstadoVI.Error_Mx AND NOT #Error_Tx;
   "DB1_SalidasExterioresDeMesa".Mesa[#Mesa].Ir_Pos_E1E3 := #MA_Bajar_TRx;
END_REGION

REGION Network 92: ESTADOS de la Mesa
   RUNG wire#powerrail
      Contact( "ON" )
      wire#w1
      Contact( #Mx_ET00 )
      wire#w2
      Coil( #EstadoVI.Etapas_Reset )
   END_RUNG
   RUNG wire#w1
      Contact( #Mx_RES01 )
   END_RUNG wire#w2
   RUNG wire#w1
      Contact( #Mx_RES02 )
   END_RUNG wire#w2
   RUNG wire#w1
      Contact( #Mx_RES03 )
   END_RUNG wire#w2
   RUNG wire#w1
      Contact( #Mx_RES09 )
   END_RUNG wire#w2
   RUNG wire#w1
      Contact( #Mx_ET01 )
      wire#w3
      Coil( #EstadoVI.Etapa_Vacia )
   END_RUNG
   RUNG wire#w1
      Contact( #Mx_ET90 )
   END_RUNG wire#w3
   RUNG wire#w1
      Contact( #Mx_ET91 )
   END_RUNG wire#w3
   RUNG wire#w1
      Contact( #Mx_ET02 )
      wire#w4
      Coil( #EstadoVI.Etapa_Cargada )
   END_RUNG
   RUNG wire#w1
      Contact( #Mx_ET250 )
   END_RUNG wire#w4
   RUNG wire#w1
      Contact( #Mx_ET260 )
   END_RUNG wire#w4
   // the same network as SCL:
   #EstadoVI.Etapas_Reset := "ON" AND (#Mx_ET00 OR #Mx_RES01 OR #Mx_RES02 OR #Mx_RES03 OR #Mx_RES09);
   #EstadoVI.Etapa_Vacia := "ON" AND (#Mx_ET01 OR #Mx_ET90 OR #Mx_ET91);
   #EstadoVI.Etapa_Cargada := "ON" AND (#Mx_ET02 OR #Mx_ET250 OR #Mx_ET260);
END_REGION

REGION Network 93: --- Carga E2
   RUNG wire#powerrail
      Contact( "ON" )
      wire#w1
      Contact( #Mx_ET20 )
      wire#w2
      Coil( #EstadoVI.Etapas_Carga_E2 )
   END_RUNG
   RUNG wire#w1
      Contact( #Mx_ET21 )
   END_RUNG wire#w2
   RUNG wire#w1
      Contact( #Mx_ET22 )
   END_RUNG wire#w2
   RUNG wire#w1
      Contact( #Mx_ET23 )
   END_RUNG wire#w2
   RUNG wire#w1
      Contact( #Mx_ET60 )
      wire#w3
      Contact( #Simul_Mx_E2S4 )
   END_RUNG wire#w2
   RUNG wire#w1
      Contact( #Mx_ET61 )
   END_RUNG wire#w3
   // the same network as SCL:
   #EstadoVI.Etapas_Carga_E2 := "ON" AND (#Mx_ET20 OR #Mx_ET21 OR #Mx_ET22 OR #Mx_ET23 OR ((#Mx_ET60 OR #Mx_ET61) AND #Simul_Mx_E2S4));
END_REGION

REGION Network 94: --- DesCarga S3
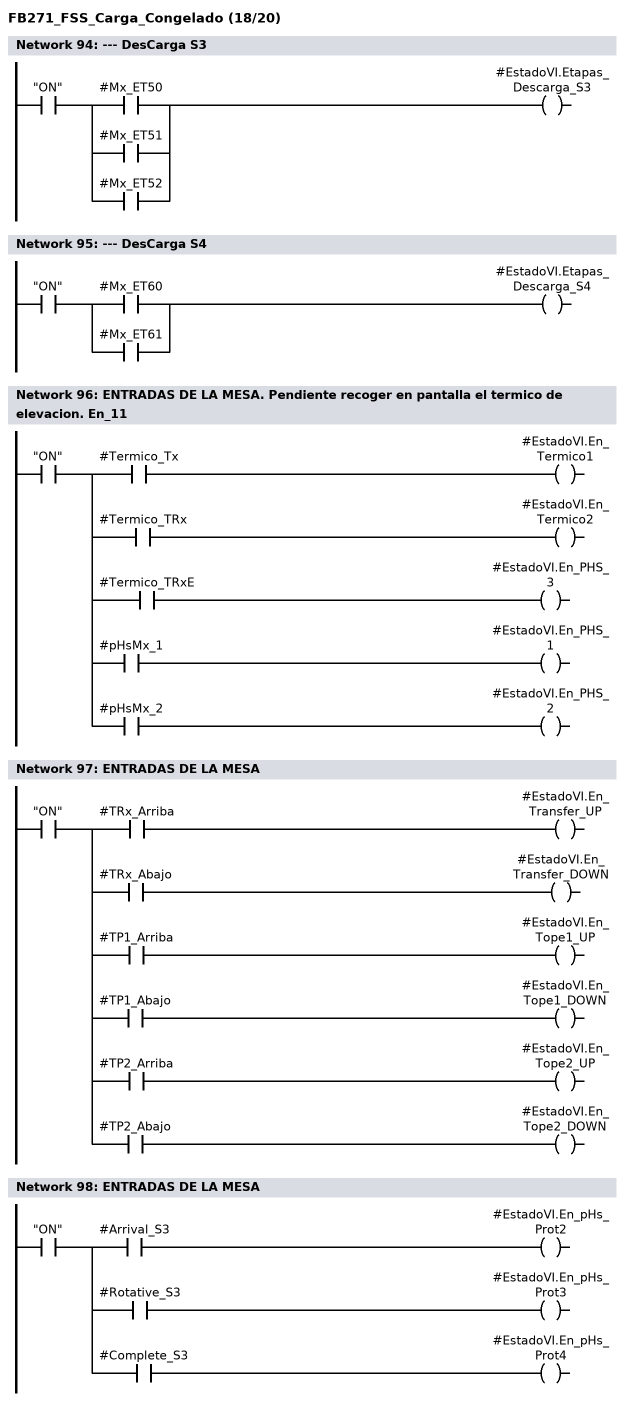
   RUNG wire#powerrail
      Contact( "ON" )
      wire#w1
      Contact( #Mx_ET50 )
      wire#w2
      Coil( #EstadoVI.Etapas_Descarga_S3 )
   END_RUNG
   RUNG wire#w1
      Contact( #Mx_ET51 )
   END_RUNG wire#w2
   RUNG wire#w1
      Contact( #Mx_ET52 )
   END_RUNG wire#w2
   // the same network as SCL:
   #EstadoVI.Etapas_Descarga_S3 := "ON" AND (#Mx_ET50 OR #Mx_ET51 OR #Mx_ET52);
END_REGION

REGION Network 95: --- DesCarga S4
   RUNG wire#powerrail
      Contact( "ON" )
      wire#w1
      Contact( #Mx_ET60 )
      wire#w2
      Coil( #EstadoVI.Etapas_Descarga_S4 )
   END_RUNG
   RUNG wire#w1
      Contact( #Mx_ET61 )
   END_RUNG wire#w2
   // the same network as SCL:
   #EstadoVI.Etapas_Descarga_S4 := "ON" AND (#Mx_ET60 OR #Mx_ET61);
END_REGION

REGION Network 96: ENTRADAS DE LA MESA. Pendiente recoger en pantalla el termico de elevacion. En_11
   RUNG wire#powerrail
      Contact( "ON" )
      wire#w1
      Contact( #Termico_Tx )
      Coil( #EstadoVI.En_Termico1 )
   END_RUNG
   RUNG wire#w1
      Contact( #Termico_TRx )
      Coil( #EstadoVI.En_Termico2 )
   END_RUNG
   RUNG wire#w1
      Contact( #Termico_TRxE )
      Coil( #EstadoVI.En_PHS_3 )
   END_RUNG
   RUNG wire#w1
      Contact( #pHsMx_1 )
      Coil( #EstadoVI.En_PHS_1 )
   END_RUNG
   RUNG wire#w1
      Contact( #pHsMx_2 )
      Coil( #EstadoVI.En_PHS_2 )
   END_RUNG
   // the same network as SCL:
   #EstadoVI.En_Termico1 := "ON" AND #Termico_Tx;
   #EstadoVI.En_Termico2 := "ON" AND #Termico_TRx;
   #EstadoVI.En_PHS_3 := "ON" AND #Termico_TRxE;
   #EstadoVI.En_PHS_1 := "ON" AND #pHsMx_1;
   #EstadoVI.En_PHS_2 := "ON" AND #pHsMx_2;
END_REGION

REGION Network 97: ENTRADAS DE LA MESA
   RUNG wire#powerrail
      Contact( "ON" )
      wire#w1
      Contact( #TRx_Arriba )
      Coil( #EstadoVI.En_Transfer_UP )
   END_RUNG
   RUNG wire#w1
      Contact( #TRx_Abajo )
      Coil( #EstadoVI.En_Transfer_DOWN )
   END_RUNG
   RUNG wire#w1
      Contact( #TP1_Arriba )
      Coil( #EstadoVI.En_Tope1_UP )
   END_RUNG
   RUNG wire#w1
      Contact( #TP1_Abajo )
      Coil( #EstadoVI.En_Tope1_DOWN )
   END_RUNG
   RUNG wire#w1
      Contact( #TP2_Arriba )
      Coil( #EstadoVI.En_Tope2_UP )
   END_RUNG
   RUNG wire#w1
      Contact( #TP2_Abajo )
      Coil( #EstadoVI.En_Tope2_DOWN )
   END_RUNG
   // the same network as SCL:
   #EstadoVI.En_Transfer_UP := "ON" AND #TRx_Arriba;
   #EstadoVI.En_Transfer_DOWN := "ON" AND #TRx_Abajo;
   #EstadoVI.En_Tope1_UP := "ON" AND #TP1_Arriba;
   #EstadoVI.En_Tope1_DOWN := "ON" AND #TP1_Abajo;
   #EstadoVI.En_Tope2_UP := "ON" AND #TP2_Arriba;
   #EstadoVI.En_Tope2_DOWN := "ON" AND #TP2_Abajo;
END_REGION

REGION Network 98: ENTRADAS DE LA MESA
   RUNG wire#powerrail
      Contact( "ON" )
      wire#w1
      Contact( #Arrival_S3 )
      Coil( #EstadoVI.En_pHs_Prot2 )
   END_RUNG
   RUNG wire#w1
      Contact( #Rotative_S3 )
      Coil( #EstadoVI.En_pHs_Prot3 )
   END_RUNG
   RUNG wire#w1
      Contact( #Complete_S3 )
      Coil( #EstadoVI.En_pHs_Prot4 )
   END_RUNG
   // the same network as SCL:
   #EstadoVI.En_pHs_Prot2 := "ON" AND #Arrival_S3;
   #EstadoVI.En_pHs_Prot3 := "ON" AND #Rotative_S3;
   #EstadoVI.En_pHs_Prot4 := "ON" AND #Complete_S3;
END_REGION

REGION Network 99: SALIDAS DE LA MESA
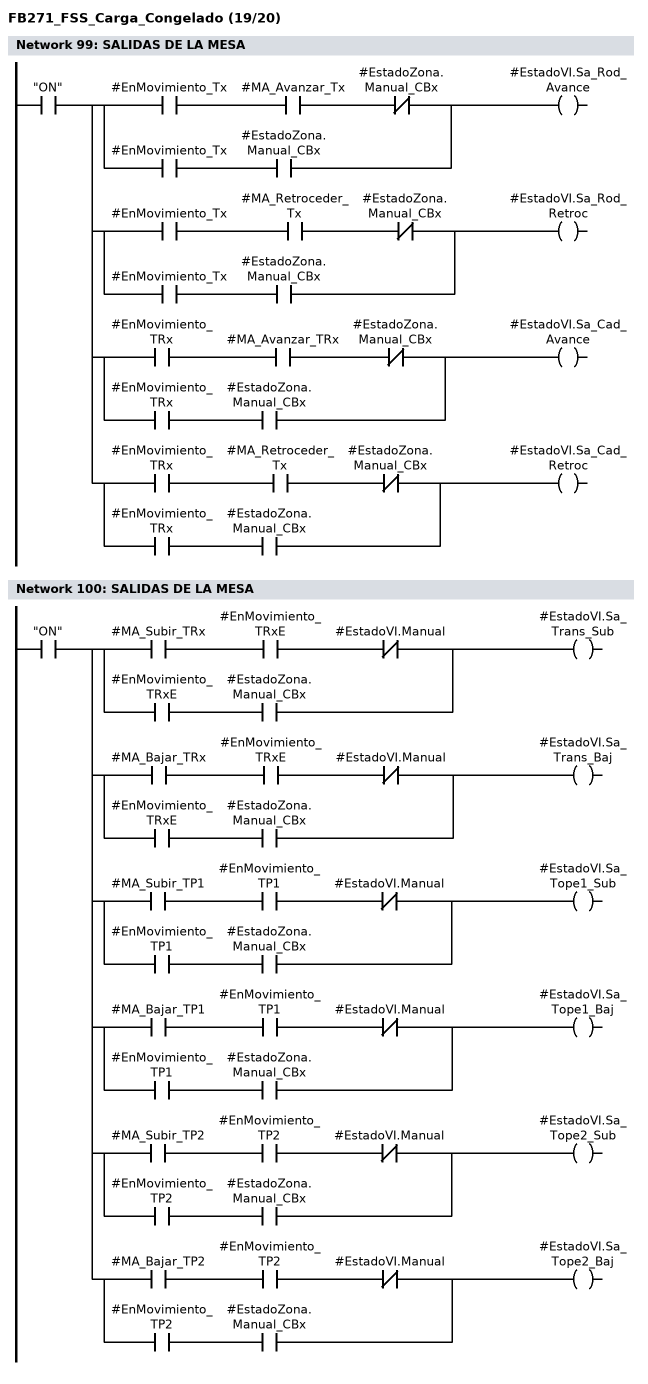
   RUNG wire#powerrail
      Contact( "ON" )
      wire#w1
      Contact( #EnMovimiento_Tx )
      Contact( #MA_Avanzar_Tx )
      I_Contact( #EstadoZona.Manual_CBx )
      wire#w2
      Coil( #EstadoVI.Sa_Rod_Avance )
   END_RUNG
   RUNG wire#w1
      Contact( #EnMovimiento_Tx )
      Contact( #EstadoZona.Manual_CBx )
   END_RUNG wire#w2
   RUNG wire#w1
      Contact( #EnMovimiento_Tx )
      Contact( #MA_Retroceder_Tx )
      I_Contact( #EstadoZona.Manual_CBx )
      wire#w3
      Coil( #EstadoVI.Sa_Rod_Retroc )
   END_RUNG
   RUNG wire#w1
      Contact( #EnMovimiento_Tx )
      Contact( #EstadoZona.Manual_CBx )
   END_RUNG wire#w3
   RUNG wire#w1
      Contact( #EnMovimiento_TRx )
      Contact( #MA_Avanzar_TRx )
      I_Contact( #EstadoZona.Manual_CBx )
      wire#w4
      Coil( #EstadoVI.Sa_Cad_Avance )
   END_RUNG
   RUNG wire#w1
      Contact( #EnMovimiento_TRx )
      Contact( #EstadoZona.Manual_CBx )
   END_RUNG wire#w4
   RUNG wire#w1
      Contact( #EnMovimiento_TRx )
      Contact( #MA_Retroceder_Tx )
      I_Contact( #EstadoZona.Manual_CBx )
      wire#w5
      Coil( #EstadoVI.Sa_Cad_Retroc )
   END_RUNG
   RUNG wire#w1
      Contact( #EnMovimiento_TRx )
      Contact( #EstadoZona.Manual_CBx )
   END_RUNG wire#w5
   // the same network as SCL:
   #EstadoVI.Sa_Rod_Avance := "ON" AND ((#EnMovimiento_Tx AND #MA_Avanzar_Tx AND NOT #EstadoZona.Manual_CBx) OR (#EnMovimiento_Tx AND #EstadoZona.Manual_CBx));
   #EstadoVI.Sa_Rod_Retroc := "ON" AND ((#EnMovimiento_Tx AND #MA_Retroceder_Tx AND NOT #EstadoZona.Manual_CBx) OR (#EnMovimiento_Tx AND #EstadoZona.Manual_CBx));
   #EstadoVI.Sa_Cad_Avance := "ON" AND ((#EnMovimiento_TRx AND #MA_Avanzar_TRx AND NOT #EstadoZona.Manual_CBx) OR (#EnMovimiento_TRx AND #EstadoZona.Manual_CBx));
   #EstadoVI.Sa_Cad_Retroc := "ON" AND ((#EnMovimiento_TRx AND #MA_Retroceder_Tx AND NOT #EstadoZona.Manual_CBx) OR (#EnMovimiento_TRx AND #EstadoZona.Manual_CBx));
END_REGION

REGION Network 100: SALIDAS DE LA MESA
   RUNG wire#powerrail
      Contact( "ON" )
      wire#w1
      Contact( #MA_Subir_TRx )
      Contact( #EnMovimiento_TRxE )
      I_Contact( #EstadoVI.Manual )
      wire#w2
      Coil( #EstadoVI.Sa_Trans_Sub )
   END_RUNG
   RUNG wire#w1
      Contact( #EnMovimiento_TRxE )
      Contact( #EstadoZona.Manual_CBx )
   END_RUNG wire#w2
   RUNG wire#w1
      Contact( #MA_Bajar_TRx )
      Contact( #EnMovimiento_TRxE )
      I_Contact( #EstadoVI.Manual )
      wire#w3
      Coil( #EstadoVI.Sa_Trans_Baj )
   END_RUNG
   RUNG wire#w1
      Contact( #EnMovimiento_TRxE )
      Contact( #EstadoZona.Manual_CBx )
   END_RUNG wire#w3
   RUNG wire#w1
      Contact( #MA_Subir_TP1 )
      Contact( #EnMovimiento_TP1 )
      I_Contact( #EstadoVI.Manual )
      wire#w4
      Coil( #EstadoVI.Sa_Tope1_Sub )
   END_RUNG
   RUNG wire#w1
      Contact( #EnMovimiento_TP1 )
      Contact( #EstadoZona.Manual_CBx )
   END_RUNG wire#w4
   RUNG wire#w1
      Contact( #MA_Bajar_TP1 )
      Contact( #EnMovimiento_TP1 )
      I_Contact( #EstadoVI.Manual )
      wire#w5
      Coil( #EstadoVI.Sa_Tope1_Baj )
   END_RUNG
   RUNG wire#w1
      Contact( #EnMovimiento_TP1 )
      Contact( #EstadoZona.Manual_CBx )
   END_RUNG wire#w5
   RUNG wire#w1
      Contact( #MA_Subir_TP2 )
      Contact( #EnMovimiento_TP2 )
      I_Contact( #EstadoVI.Manual )
      wire#w6
      Coil( #EstadoVI.Sa_Tope2_Sub )
   END_RUNG
   RUNG wire#w1
      Contact( #EnMovimiento_TP2 )
      Contact( #EstadoZona.Manual_CBx )
   END_RUNG wire#w6
   RUNG wire#w1
      Contact( #MA_Bajar_TP2 )
      Contact( #EnMovimiento_TP2 )
      I_Contact( #EstadoVI.Manual )
      wire#w7
      Coil( #EstadoVI.Sa_Tope2_Baj )
   END_RUNG
   RUNG wire#w1
      Contact( #EnMovimiento_TP2 )
      Contact( #EstadoZona.Manual_CBx )
   END_RUNG wire#w7
   // the same network as SCL:
   #EstadoVI.Sa_Trans_Sub := "ON" AND ((#MA_Subir_TRx AND #EnMovimiento_TRxE AND NOT #EstadoVI.Manual) OR (#EnMovimiento_TRxE AND #EstadoZona.Manual_CBx));
   #EstadoVI.Sa_Trans_Baj := "ON" AND ((#MA_Bajar_TRx AND #EnMovimiento_TRxE AND NOT #EstadoVI.Manual) OR (#EnMovimiento_TRxE AND #EstadoZona.Manual_CBx));
   #EstadoVI.Sa_Tope1_Sub := "ON" AND ((#MA_Subir_TP1 AND #EnMovimiento_TP1 AND NOT #EstadoVI.Manual) OR (#EnMovimiento_TP1 AND #EstadoZona.Manual_CBx));
   #EstadoVI.Sa_Tope1_Baj := "ON" AND ((#MA_Bajar_TP1 AND #EnMovimiento_TP1 AND NOT #EstadoVI.Manual) OR (#EnMovimiento_TP1 AND #EstadoZona.Manual_CBx));
   #EstadoVI.Sa_Tope2_Sub := "ON" AND ((#MA_Subir_TP2 AND #EnMovimiento_TP2 AND NOT #EstadoVI.Manual) OR (#EnMovimiento_TP2 AND #EstadoZona.Manual_CBx));
   #EstadoVI.Sa_Tope2_Baj := "ON" AND ((#MA_Bajar_TP2 AND #EnMovimiento_TP2 AND NOT #EstadoVI.Manual) OR (#EnMovimiento_TP2 AND #EstadoZona.Manual_CBx));
END_REGION

REGION Network 101: SALIDAS DE LA MESA
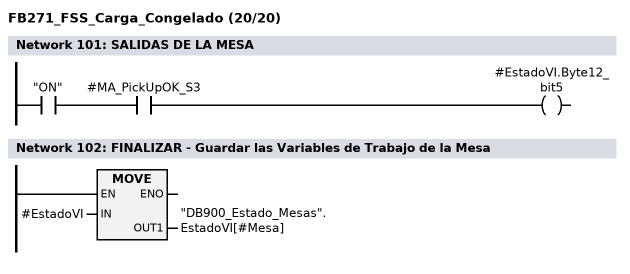
   RUNG wire#powerrail
      Contact( "ON" )
      Contact( #MA_PickUpOK_S3 )
      Coil( #EstadoVI.Byte12_bit5 )
   END_RUNG
   // the same network as SCL:
   #EstadoVI.Byte12_bit5 := "ON" AND #MA_PickUpOK_S3;
END_REGION

REGION Network 102: FINALIZAR - Guardar las Variables de Trabajo de la Mesa
   RUNG wire#powerrail
      Move(in := #EstadoVI, out1 => "DB900_Estado_Mesas".EstadoVI[#Mesa])
   END_RUNG
   // the same network as SCL:
   "DB900_Estado_Mesas".EstadoVI[#Mesa] := #EstadoVI;
END_REGION
END_FUNCTION_BLOCK
